REGION Network 2: PREMIXING VESSEL BOTTOM STERROR RUN
   RUNG wire#powerrail
      I_Contact( "AlwaysTRUE" )
      { S7_Templates := "SrcType := Int" } EQ_Contact(in1 := "MODE SELECTION DB"."MODE BUFF", in2 := 2)
      I_Contact( "RECIRCULATION DB".PREMIXING.PAUSE )
      Coil( "TRANSFER DB".OUTPUT."PREMIXING VESSEL BOTTOM STERROR RUN" )
   END_RUNG
   // the same network as SCL:
   "TRANSFER DB".OUTPUT."PREMIXING VESSEL BOTTOM STERROR RUN" := NOT "AlwaysTRUE" AND ("MODE SELECTION DB"."MODE BUFF" = 2) AND NOT "RECIRCULATION DB".PREMIXING.PAUSE;
END_REGION

REGION Network 3: INLINE 1 HOMOGENIZER MOTOR1 RUN
   RUNG wire#powerrail
      Contact( "AlwaysTRUE" )
      wire#w1
      { S7_Templates := "SrcType := Int" } NE_Contact(in1 := "MODE SELECTION DB"."MODE BUFF", in2 := 0)
      wire#w2
      Contact( "TRANSFER DB".BIT."MFG TO STORAGE-1 WITH INLINE HOMO"."INLINE 1 HOMOGENIZER MOTOR1 RUN" )
      wire#w3
      Contact( "DO MAPING"."PAV-56 INLINE HOMO. SEAL COOLING INLET" )
      { S7_Templates := "time_type := Time" } "IEC_Timer_0_DB_80".TON(pt := T#3S, et =>)
      Coil( "TRANSFER DB".OUTPUT."INLINE 1 HOMOGENIZER MOTOR1 RUN" )
   END_RUNG
   RUNG wire#w2
      Contact( "TRANSFER DB".BIT."MFG TO STORAGE-2 WITH INLINE HOMO"."INLINE 1 HOMOGENIZER MOTOR1 RUN" )
   END_RUNG wire#w3
   RUNG wire#w2
      Contact( "TRANSFER DB".BIT."MFG TO STORAGE-3 WITH INLINE HOMO"."INLINE 1 HOMOGENIZER MOTOR1 RUN" )
   END_RUNG wire#w3
   RUNG wire#w1
      { S7_Templates := "SrcType := Int" } EQ_Contact(in1 := "MODE SELECTION DB"."MODE BUFF", in2 := 2)
      { S7_Templates := "SrcType := Int" } EQ_Contact(in1 := "RECIRCULATION DB".MFG.BUFF, in2 := 2)
      I_Contact( "RECIRCULATION DB".MFG.PAUSE )
   END_RUNG wire#w3
   // the same network as SCL:
   "IEC_Timer_0_DB_80".TON(IN := "AlwaysTRUE" AND ((("MODE SELECTION DB"."MODE BUFF" <> 0) AND ("TRANSFER DB".BIT."MFG TO STORAGE-1 WITH INLINE HOMO"."INLINE 1 HOMOGENIZER MOTOR1 RUN" OR "TRANSFER DB".BIT."MFG TO STORAGE-2 WITH INLINE HOMO"."INLINE 1 HOMOGENIZER MOTOR1 RUN" OR "TRANSFER DB".BIT."MFG TO STORAGE-3 WITH INLINE HOMO"."INLINE 1 HOMOGENIZER MOTOR1 RUN")) OR (("MODE SELECTION DB"."MODE BUFF" = 2) AND ("RECIRCULATION DB".MFG.BUFF = 2) AND NOT "RECIRCULATION DB".MFG.PAUSE)) AND "DO MAPING"."PAV-56 INLINE HOMO. SEAL COOLING INLET",
                           PT := T#3S);
   "TRANSFER DB".OUTPUT."INLINE 1 HOMOGENIZER MOTOR1 RUN" := "IEC_Timer_0_DB_80".Q;
END_REGION

REGION Network 4: INLINE 2 HOMOGENIZER MOTOR 2 RUN
   RUNG wire#powerrail
      Contact( "AlwaysTRUE" )
      wire#w1
      { S7_Templates := "SrcType := Int" } NE_Contact(in1 := "MODE SELECTION DB"."MODE BUFF", in2 := 0)
      wire#w2
      Contact( "TRANSFER DB".BIT."PREMIXING TO MFG WITH INLINE HOMO"."INLINE 2 HOMOGENIZER MOTOR 2 RUN" )
      wire#w3
      Contact( "DO MAPING"."PAV-99 INLINE HOMOGENIZER SEAL COOLING" )
      { S7_Templates := "time_type := Time" } "IEC_Timer_0_DB_65".TON(pt := T#3S, et =>)
      Coil( "TRANSFER DB".OUTPUT."INLINE 2 HOMOGENIZER MOTOR 2 RUN" )
   END_RUNG
   RUNG wire#w2
      Contact( "TRANSFER DB".BIT."PREMIXING TO STORAGE-4 WITH INLINE HOMO"."INLINE 2 HOMOGENIZER MOTOR 2 RUN" )
   END_RUNG wire#w3
   RUNG wire#w1
      { S7_Templates := "SrcType := Int" } EQ_Contact(in1 := "MODE SELECTION DB"."MODE BUFF", in2 := 2)
      { S7_Templates := "SrcType := Int" } EQ_Contact(in1 := "RECIRCULATION DB".PREMIXING.BUFF, in2 := 2)
      I_Contact( "RECIRCULATION DB".PREMIXING.PAUSE )
   END_RUNG wire#w3
   // the same network as SCL:
   "IEC_Timer_0_DB_65".TON(IN := "AlwaysTRUE" AND ((("MODE SELECTION DB"."MODE BUFF" <> 0) AND ("TRANSFER DB".BIT."PREMIXING TO MFG WITH INLINE HOMO"."INLINE 2 HOMOGENIZER MOTOR 2 RUN" OR "TRANSFER DB".BIT."PREMIXING TO STORAGE-4 WITH INLINE HOMO"."INLINE 2 HOMOGENIZER MOTOR 2 RUN")) OR (("MODE SELECTION DB"."MODE BUFF" = 2) AND ("RECIRCULATION DB".PREMIXING.BUFF = 2) AND NOT "RECIRCULATION DB".PREMIXING.PAUSE)) AND "DO MAPING"."PAV-99 INLINE HOMOGENIZER SEAL COOLING",
                           PT := T#3S);
   "TRANSFER DB".OUTPUT."INLINE 2 HOMOGENIZER MOTOR 2 RUN" := "IEC_Timer_0_DB_65".Q;
END_REGION

REGION Network 5: FILTER PRESS MOTOR 1 RUN
   RUNG wire#powerrail
      Contact( "AlwaysTRUE" )
      { S7_Templates := "SrcType := Int" } NE_Contact(in1 := "MODE SELECTION DB"."MODE BUFF", in2 := 0)
      wire#w1
      Contact( "TRANSFER DB".BIT."MFG TO STORAGE-1 WITH INLINE FILTER PRES"."FILTER PRESS MOTOR 1 RUN" )
      wire#w2
      Coil( "TRANSFER DB".OUTPUT."FILTER PRESS MOTOR 1 RUN" )
   END_RUNG
   RUNG wire#w1
      Contact( "TRANSFER DB".BIT."MFG TO STORAGE-2 WITH INLINE FILTER PRES"."FILTER PRESS MOTOR 1 RUN" )
   END_RUNG wire#w2
   RUNG wire#w1
      Contact( "TRANSFER DB".BIT."MFG TO STORAGE-3 WITH INLINE FILTER PRES"."FILTER PRESS MOTOR 1 RUN" )
   END_RUNG wire#w2
   // the same network as SCL:
   "TRANSFER DB".OUTPUT."FILTER PRESS MOTOR 1 RUN" := "AlwaysTRUE" AND ("MODE SELECTION DB"."MODE BUFF" <> 0) AND ("TRANSFER DB".BIT."MFG TO STORAGE-1 WITH INLINE FILTER PRES"."FILTER PRESS MOTOR 1 RUN" OR "TRANSFER DB".BIT."MFG TO STORAGE-2 WITH INLINE FILTER PRES"."FILTER PRESS MOTOR 1 RUN" OR "TRANSFER DB".BIT."MFG TO STORAGE-3 WITH INLINE FILTER PRES"."FILTER PRESS MOTOR 1 RUN");
END_REGION

REGION Network 6: FILTER PRESS MOTOR 2 RUN
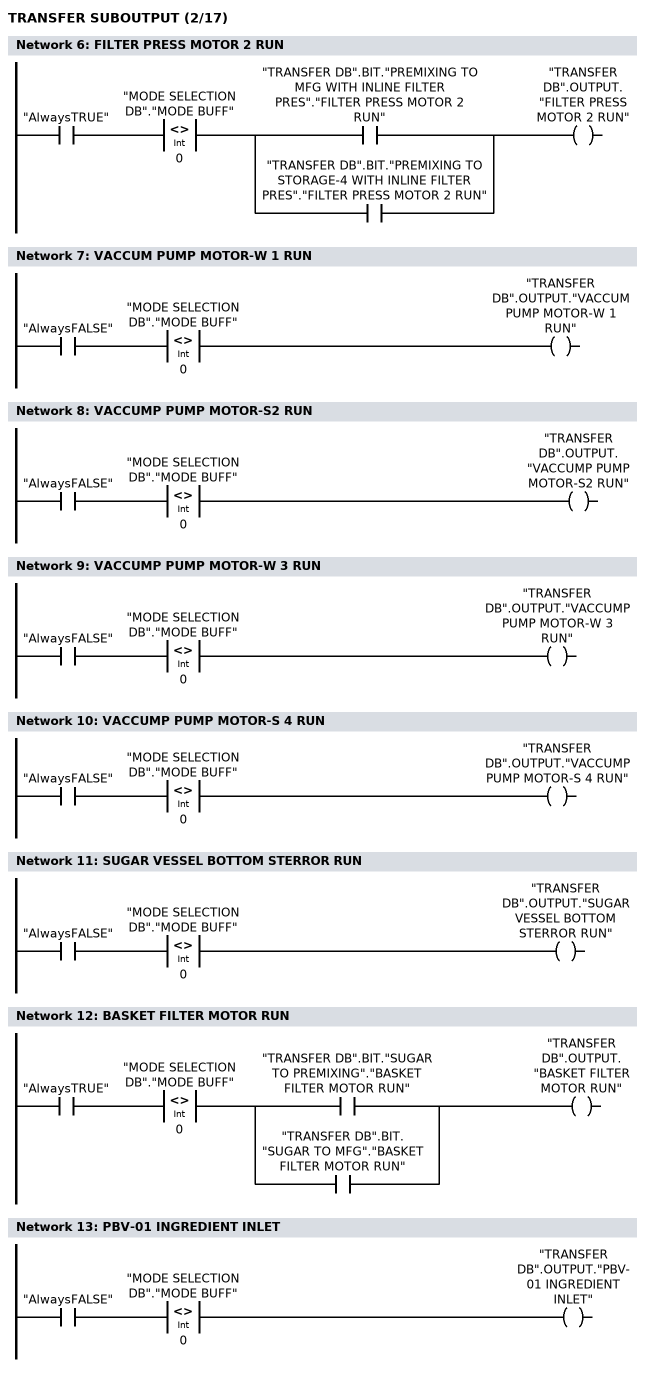
   RUNG wire#powerrail
      Contact( "AlwaysTRUE" )
      { S7_Templates := "SrcType := Int" } NE_Contact(in1 := "MODE SELECTION DB"."MODE BUFF", in2 := 0)
      wire#w1
      Contact( "TRANSFER DB".BIT."PREMIXING TO MFG WITH INLINE FILTER PRES"."FILTER PRESS MOTOR 2 RUN" )
      wire#w2
      Coil( "TRANSFER DB".OUTPUT."FILTER PRESS MOTOR 2 RUN" )
   END_RUNG
   RUNG wire#w1
      Contact( "TRANSFER DB".BIT."PREMIXING TO STORAGE-4 WITH INLINE FILTER PRES"."FILTER PRESS MOTOR 2 RUN" )
   END_RUNG wire#w2
   // the same network as SCL:
   "TRANSFER DB".OUTPUT."FILTER PRESS MOTOR 2 RUN" := "AlwaysTRUE" AND ("MODE SELECTION DB"."MODE BUFF" <> 0) AND ("TRANSFER DB".BIT."PREMIXING TO MFG WITH INLINE FILTER PRES"."FILTER PRESS MOTOR 2 RUN" OR "TRANSFER DB".BIT."PREMIXING TO STORAGE-4 WITH INLINE FILTER PRES"."FILTER PRESS MOTOR 2 RUN");
END_REGION

REGION Network 7: VACCUM PUMP MOTOR-W 1 RUN
   RUNG wire#powerrail
      Contact( "AlwaysFALSE" )
      { S7_Templates := "SrcType := Int" } NE_Contact(in1 := "MODE SELECTION DB"."MODE BUFF", in2 := 0)
      Coil( "TRANSFER DB".OUTPUT."VACCUM PUMP MOTOR-W 1 RUN" )
   END_RUNG
   // the same network as SCL:
   "TRANSFER DB".OUTPUT."VACCUM PUMP MOTOR-W 1 RUN" := "AlwaysFALSE" AND ("MODE SELECTION DB"."MODE BUFF" <> 0);
END_REGION

REGION Network 8: VACCUMP PUMP MOTOR-S2 RUN
   RUNG wire#powerrail
      Contact( "AlwaysFALSE" )
      { S7_Templates := "SrcType := Int" } NE_Contact(in1 := "MODE SELECTION DB"."MODE BUFF", in2 := 0)
      Coil( "TRANSFER DB".OUTPUT."VACCUMP PUMP MOTOR-S2 RUN" )
   END_RUNG
   // the same network as SCL:
   "TRANSFER DB".OUTPUT."VACCUMP PUMP MOTOR-S2 RUN" := "AlwaysFALSE" AND ("MODE SELECTION DB"."MODE BUFF" <> 0);
END_REGION

REGION Network 9: VACCUMP PUMP MOTOR-W 3 RUN
   RUNG wire#powerrail
      Contact( "AlwaysFALSE" )
      { S7_Templates := "SrcType := Int" } NE_Contact(in1 := "MODE SELECTION DB"."MODE BUFF", in2 := 0)
      Coil( "TRANSFER DB".OUTPUT."VACCUMP PUMP MOTOR-W 3 RUN" )
   END_RUNG
   // the same network as SCL:
   "TRANSFER DB".OUTPUT."VACCUMP PUMP MOTOR-W 3 RUN" := "AlwaysFALSE" AND ("MODE SELECTION DB"."MODE BUFF" <> 0);
END_REGION

REGION Network 10: VACCUMP PUMP MOTOR-S 4 RUN
   RUNG wire#powerrail
      Contact( "AlwaysFALSE" )
      { S7_Templates := "SrcType := Int" } NE_Contact(in1 := "MODE SELECTION DB"."MODE BUFF", in2 := 0)
      Coil( "TRANSFER DB".OUTPUT."VACCUMP PUMP MOTOR-S 4 RUN" )
   END_RUNG
   // the same network as SCL:
   "TRANSFER DB".OUTPUT."VACCUMP PUMP MOTOR-S 4 RUN" := "AlwaysFALSE" AND ("MODE SELECTION DB"."MODE BUFF" <> 0);
END_REGION

REGION Network 11: SUGAR VESSEL BOTTOM STERROR RUN
   RUNG wire#powerrail
      Contact( "AlwaysFALSE" )
      { S7_Templates := "SrcType := Int" } NE_Contact(in1 := "MODE SELECTION DB"."MODE BUFF", in2 := 0)
      Coil( "TRANSFER DB".OUTPUT."SUGAR VESSEL BOTTOM STERROR RUN" )
   END_RUNG
   // the same network as SCL:
   "TRANSFER DB".OUTPUT."SUGAR VESSEL BOTTOM STERROR RUN" := "AlwaysFALSE" AND ("MODE SELECTION DB"."MODE BUFF" <> 0);
END_REGION

REGION Network 12: BASKET FILTER MOTOR RUN
   RUNG wire#powerrail
      Contact( "AlwaysTRUE" )
      { S7_Templates := "SrcType := Int" } NE_Contact(in1 := "MODE SELECTION DB"."MODE BUFF", in2 := 0)
      wire#w1
      Contact( "TRANSFER DB".BIT."SUGAR TO PREMIXING"."BASKET FILTER MOTOR RUN" )
      wire#w2
      Coil( "TRANSFER DB".OUTPUT."BASKET FILTER MOTOR RUN" )
   END_RUNG
   RUNG wire#w1
      Contact( "TRANSFER DB".BIT."SUGAR TO MFG"."BASKET FILTER MOTOR RUN" )
   END_RUNG wire#w2
   // the same network as SCL:
   "TRANSFER DB".OUTPUT."BASKET FILTER MOTOR RUN" := "AlwaysTRUE" AND ("MODE SELECTION DB"."MODE BUFF" <> 0) AND ("TRANSFER DB".BIT."SUGAR TO PREMIXING"."BASKET FILTER MOTOR RUN" OR "TRANSFER DB".BIT."SUGAR TO MFG"."BASKET FILTER MOTOR RUN");
END_REGION

REGION Network 13: PBV-01 INGREDIENT INLET
   RUNG wire#powerrail
      Contact( "AlwaysFALSE" )
      { S7_Templates := "SrcType := Int" } NE_Contact(in1 := "MODE SELECTION DB"."MODE BUFF", in2 := 0)
      Coil( "TRANSFER DB".OUTPUT."PBV-01 INGREDIENT INLET" )
   END_RUNG
   // the same network as SCL:
   "TRANSFER DB".OUTPUT."PBV-01 INGREDIENT INLET" := "AlwaysFALSE" AND ("MODE SELECTION DB"."MODE BUFF" <> 0);
END_REGION

REGION Network 14: PBV-02 CIP INLET (SPRAY BALL)
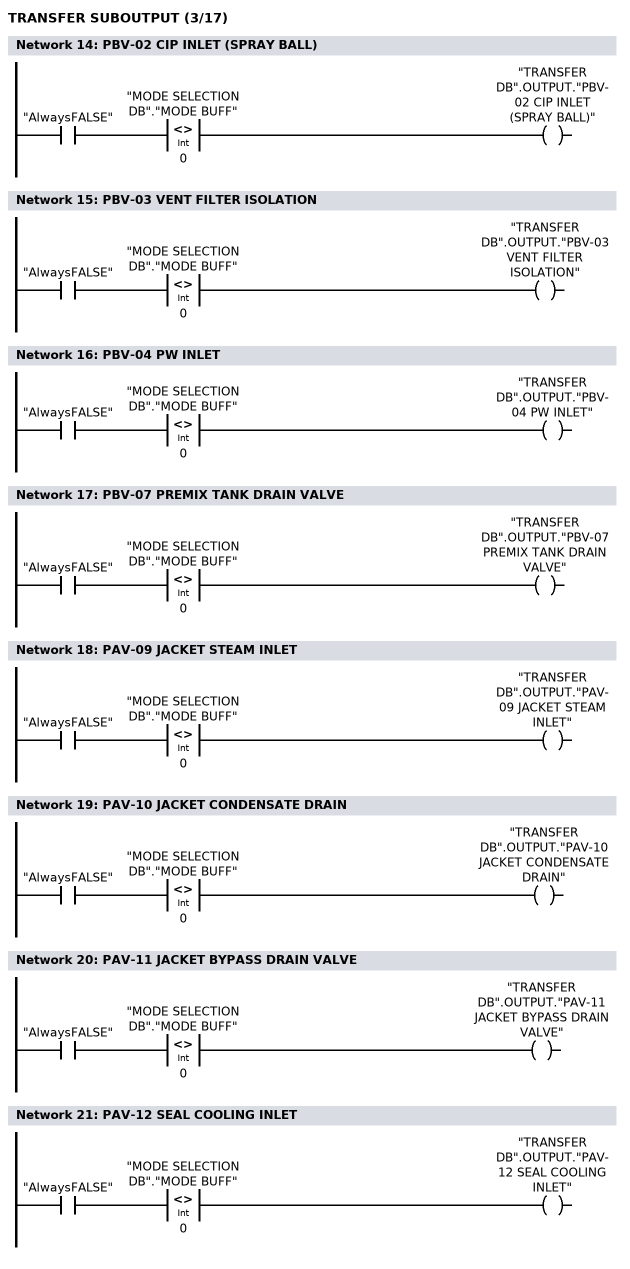
   RUNG wire#powerrail
      Contact( "AlwaysFALSE" )
      { S7_Templates := "SrcType := Int" } NE_Contact(in1 := "MODE SELECTION DB"."MODE BUFF", in2 := 0)
      Coil( "TRANSFER DB".OUTPUT."PBV-02 CIP INLET (SPRAY BALL)" )
   END_RUNG
   // the same network as SCL:
   "TRANSFER DB".OUTPUT."PBV-02 CIP INLET (SPRAY BALL)" := "AlwaysFALSE" AND ("MODE SELECTION DB"."MODE BUFF" <> 0);
END_REGION

REGION Network 15: PBV-03 VENT FILTER ISOLATION
   RUNG wire#powerrail
      Contact( "AlwaysFALSE" )
      { S7_Templates := "SrcType := Int" } NE_Contact(in1 := "MODE SELECTION DB"."MODE BUFF", in2 := 0)
      Coil( "TRANSFER DB".OUTPUT."PBV-03 VENT FILTER ISOLATION" )
   END_RUNG
   // the same network as SCL:
   "TRANSFER DB".OUTPUT."PBV-03 VENT FILTER ISOLATION" := "AlwaysFALSE" AND ("MODE SELECTION DB"."MODE BUFF" <> 0);
END_REGION

REGION Network 16: PBV-04 PW INLET
   RUNG wire#powerrail
      Contact( "AlwaysFALSE" )
      { S7_Templates := "SrcType := Int" } NE_Contact(in1 := "MODE SELECTION DB"."MODE BUFF", in2 := 0)
      Coil( "TRANSFER DB".OUTPUT."PBV-04 PW INLET" )
   END_RUNG
   // the same network as SCL:
   "TRANSFER DB".OUTPUT."PBV-04 PW INLET" := "AlwaysFALSE" AND ("MODE SELECTION DB"."MODE BUFF" <> 0);
END_REGION

REGION Network 17: PBV-07 PREMIX TANK DRAIN VALVE
   RUNG wire#powerrail
      Contact( "AlwaysFALSE" )
      { S7_Templates := "SrcType := Int" } NE_Contact(in1 := "MODE SELECTION DB"."MODE BUFF", in2 := 0)
      Coil( "TRANSFER DB".OUTPUT."PBV-07 PREMIX TANK DRAIN VALVE" )
   END_RUNG
   // the same network as SCL:
   "TRANSFER DB".OUTPUT."PBV-07 PREMIX TANK DRAIN VALVE" := "AlwaysFALSE" AND ("MODE SELECTION DB"."MODE BUFF" <> 0);
END_REGION

REGION Network 18: PAV-09 JACKET STEAM INLET
   RUNG wire#powerrail
      Contact( "AlwaysFALSE" )
      { S7_Templates := "SrcType := Int" } NE_Contact(in1 := "MODE SELECTION DB"."MODE BUFF", in2 := 0)
      Coil( "TRANSFER DB".OUTPUT."PAV-09 JACKET STEAM INLET" )
   END_RUNG
   // the same network as SCL:
   "TRANSFER DB".OUTPUT."PAV-09 JACKET STEAM INLET" := "AlwaysFALSE" AND ("MODE SELECTION DB"."MODE BUFF" <> 0);
END_REGION

REGION Network 19: PAV-10 JACKET CONDENSATE DRAIN
   RUNG wire#powerrail
      Contact( "AlwaysFALSE" )
      { S7_Templates := "SrcType := Int" } NE_Contact(in1 := "MODE SELECTION DB"."MODE BUFF", in2 := 0)
      Coil( "TRANSFER DB".OUTPUT."PAV-10 JACKET CONDENSATE DRAIN" )
   END_RUNG
   // the same network as SCL:
   "TRANSFER DB".OUTPUT."PAV-10 JACKET CONDENSATE DRAIN" := "AlwaysFALSE" AND ("MODE SELECTION DB"."MODE BUFF" <> 0);
END_REGION

REGION Network 20: PAV-11 JACKET BYPASS DRAIN VALVE
   RUNG wire#powerrail
      Contact( "AlwaysFALSE" )
      { S7_Templates := "SrcType := Int" } NE_Contact(in1 := "MODE SELECTION DB"."MODE BUFF", in2 := 0)
      Coil( "TRANSFER DB".OUTPUT."PAV-11 JACKET BYPASS DRAIN VALVE" )
   END_RUNG
   // the same network as SCL:
   "TRANSFER DB".OUTPUT."PAV-11 JACKET BYPASS DRAIN VALVE" := "AlwaysFALSE" AND ("MODE SELECTION DB"."MODE BUFF" <> 0);
END_REGION

REGION Network 21: PAV-12 SEAL COOLING INLET
   RUNG wire#powerrail
      Contact( "AlwaysFALSE" )
      { S7_Templates := "SrcType := Int" } NE_Contact(in1 := "MODE SELECTION DB"."MODE BUFF", in2 := 0)
      Coil( "TRANSFER DB".OUTPUT."PAV-12 SEAL COOLING INLET" )
   END_RUNG
   // the same network as SCL:
   "TRANSFER DB".OUTPUT."PAV-12 SEAL COOLING INLET" := "AlwaysFALSE" AND ("MODE SELECTION DB"."MODE BUFF" <> 0);
END_REGION

REGION Network 22: PAV-13 WATER COOLING INLET
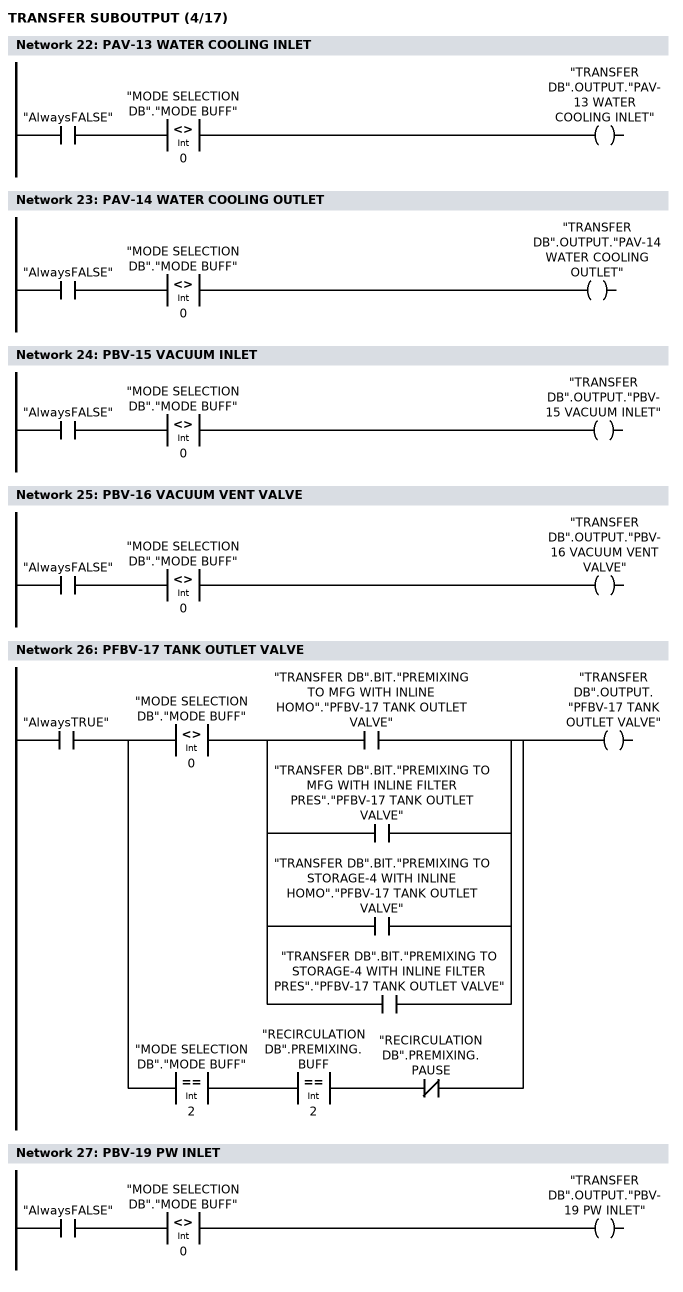
   RUNG wire#powerrail
      Contact( "AlwaysFALSE" )
      { S7_Templates := "SrcType := Int" } NE_Contact(in1 := "MODE SELECTION DB"."MODE BUFF", in2 := 0)
      Coil( "TRANSFER DB".OUTPUT."PAV-13 WATER COOLING INLET" )
   END_RUNG
   // the same network as SCL:
   "TRANSFER DB".OUTPUT."PAV-13 WATER COOLING INLET" := "AlwaysFALSE" AND ("MODE SELECTION DB"."MODE BUFF" <> 0);
END_REGION

REGION Network 23: PAV-14 WATER COOLING OUTLET
   RUNG wire#powerrail
      Contact( "AlwaysFALSE" )
      { S7_Templates := "SrcType := Int" } NE_Contact(in1 := "MODE SELECTION DB"."MODE BUFF", in2 := 0)
      Coil( "TRANSFER DB".OUTPUT."PAV-14 WATER COOLING OUTLET" )
   END_RUNG
   // the same network as SCL:
   "TRANSFER DB".OUTPUT."PAV-14 WATER COOLING OUTLET" := "AlwaysFALSE" AND ("MODE SELECTION DB"."MODE BUFF" <> 0);
END_REGION

REGION Network 24: PBV-15 VACUUM INLET
   RUNG wire#powerrail
      Contact( "AlwaysFALSE" )
      { S7_Templates := "SrcType := Int" } NE_Contact(in1 := "MODE SELECTION DB"."MODE BUFF", in2 := 0)
      Coil( "TRANSFER DB".OUTPUT."PBV-15 VACUUM INLET" )
   END_RUNG
   // the same network as SCL:
   "TRANSFER DB".OUTPUT."PBV-15 VACUUM INLET" := "AlwaysFALSE" AND ("MODE SELECTION DB"."MODE BUFF" <> 0);
END_REGION

REGION Network 25: PBV-16 VACUUM VENT VALVE
   RUNG wire#powerrail
      Contact( "AlwaysFALSE" )
      { S7_Templates := "SrcType := Int" } NE_Contact(in1 := "MODE SELECTION DB"."MODE BUFF", in2 := 0)
      Coil( "TRANSFER DB".OUTPUT."PBV-16 VACUUM VENT VALVE" )
   END_RUNG
   // the same network as SCL:
   "TRANSFER DB".OUTPUT."PBV-16 VACUUM VENT VALVE" := "AlwaysFALSE" AND ("MODE SELECTION DB"."MODE BUFF" <> 0);
END_REGION

REGION Network 26: PFBV-17 TANK OUTLET VALVE
   RUNG wire#powerrail
      Contact( "AlwaysTRUE" )
      wire#w1
      { S7_Templates := "SrcType := Int" } NE_Contact(in1 := "MODE SELECTION DB"."MODE BUFF", in2 := 0)
      wire#w2
      Contact( "TRANSFER DB".BIT."PREMIXING TO MFG WITH INLINE HOMO"."PFBV-17 TANK OUTLET VALVE" )
      wire#w3
      Coil( "TRANSFER DB".OUTPUT."PFBV-17 TANK OUTLET VALVE" )
   END_RUNG
   RUNG wire#w2
      Contact( "TRANSFER DB".BIT."PREMIXING TO MFG WITH INLINE FILTER PRES"."PFBV-17 TANK OUTLET VALVE" )
   END_RUNG wire#w3
   RUNG wire#w2
      Contact( "TRANSFER DB".BIT."PREMIXING TO STORAGE-4 WITH INLINE HOMO"."PFBV-17 TANK OUTLET VALVE" )
   END_RUNG wire#w3
   RUNG wire#w2
      Contact( "TRANSFER DB".BIT."PREMIXING TO STORAGE-4 WITH INLINE FILTER PRES"."PFBV-17 TANK OUTLET VALVE" )
   END_RUNG wire#w3
   RUNG wire#w1
      { S7_Templates := "SrcType := Int" } EQ_Contact(in1 := "MODE SELECTION DB"."MODE BUFF", in2 := 2)
      { S7_Templates := "SrcType := Int" } EQ_Contact(in1 := "RECIRCULATION DB".PREMIXING.BUFF, in2 := 2)
      I_Contact( "RECIRCULATION DB".PREMIXING.PAUSE )
   END_RUNG wire#w3
   // the same network as SCL:
   "TRANSFER DB".OUTPUT."PFBV-17 TANK OUTLET VALVE" := "AlwaysTRUE" AND ((("MODE SELECTION DB"."MODE BUFF" <> 0) AND ("TRANSFER DB".BIT."PREMIXING TO MFG WITH INLINE HOMO"."PFBV-17 TANK OUTLET VALVE" OR "TRANSFER DB".BIT."PREMIXING TO MFG WITH INLINE FILTER PRES"."PFBV-17 TANK OUTLET VALVE" OR "TRANSFER DB".BIT."PREMIXING TO STORAGE-4 WITH INLINE HOMO"."PFBV-17 TANK OUTLET VALVE" OR "TRANSFER DB".BIT."PREMIXING TO STORAGE-4 WITH INLINE FILTER PRES"."PFBV-17 TANK OUTLET VALVE")) OR (("MODE SELECTION DB"."MODE BUFF" = 2) AND ("RECIRCULATION DB".PREMIXING.BUFF = 2) AND NOT "RECIRCULATION DB".PREMIXING.PAUSE));
END_REGION

REGION Network 27: PBV-19 PW INLET
   RUNG wire#powerrail
      Contact( "AlwaysFALSE" )
      { S7_Templates := "SrcType := Int" } NE_Contact(in1 := "MODE SELECTION DB"."MODE BUFF", in2 := 0)
      Coil( "TRANSFER DB".OUTPUT."PBV-19 PW INLET" )
   END_RUNG
   // the same network as SCL:
   "TRANSFER DB".OUTPUT."PBV-19 PW INLET" := "AlwaysFALSE" AND ("MODE SELECTION DB"."MODE BUFF" <> 0);
END_REGION

REGION Network 28: PBV-20 CIP INLET (SPRAY BALL)
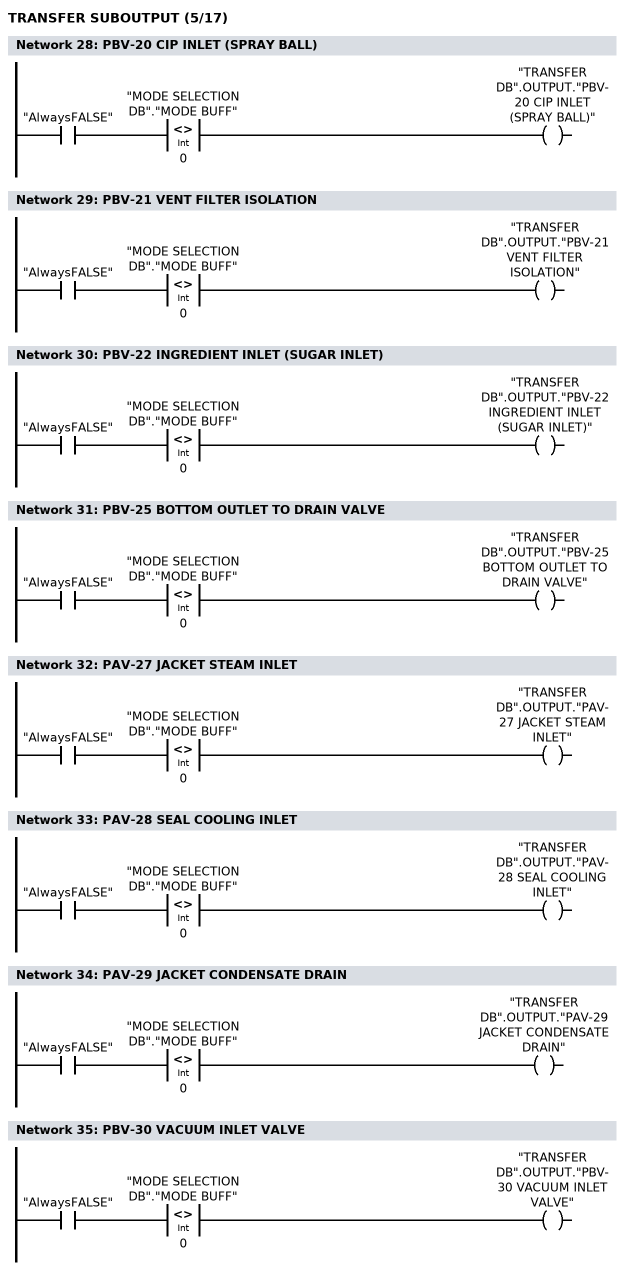
   RUNG wire#powerrail
      Contact( "AlwaysFALSE" )
      { S7_Templates := "SrcType := Int" } NE_Contact(in1 := "MODE SELECTION DB"."MODE BUFF", in2 := 0)
      Coil( "TRANSFER DB".OUTPUT."PBV-20 CIP INLET (SPRAY BALL)" )
   END_RUNG
   // the same network as SCL:
   "TRANSFER DB".OUTPUT."PBV-20 CIP INLET (SPRAY BALL)" := "AlwaysFALSE" AND ("MODE SELECTION DB"."MODE BUFF" <> 0);
END_REGION

REGION Network 29: PBV-21 VENT FILTER ISOLATION
   RUNG wire#powerrail
      Contact( "AlwaysFALSE" )
      { S7_Templates := "SrcType := Int" } NE_Contact(in1 := "MODE SELECTION DB"."MODE BUFF", in2 := 0)
      Coil( "TRANSFER DB".OUTPUT."PBV-21 VENT FILTER ISOLATION" )
   END_RUNG
   // the same network as SCL:
   "TRANSFER DB".OUTPUT."PBV-21 VENT FILTER ISOLATION" := "AlwaysFALSE" AND ("MODE SELECTION DB"."MODE BUFF" <> 0);
END_REGION

REGION Network 30: PBV-22 INGREDIENT INLET (SUGAR INLET)
   RUNG wire#powerrail
      Contact( "AlwaysFALSE" )
      { S7_Templates := "SrcType := Int" } NE_Contact(in1 := "MODE SELECTION DB"."MODE BUFF", in2 := 0)
      Coil( "TRANSFER DB".OUTPUT."PBV-22 INGREDIENT INLET (SUGAR INLET)" )
   END_RUNG
   // the same network as SCL:
   "TRANSFER DB".OUTPUT."PBV-22 INGREDIENT INLET (SUGAR INLET)" := "AlwaysFALSE" AND ("MODE SELECTION DB"."MODE BUFF" <> 0);
END_REGION

REGION Network 31: PBV-25 BOTTOM OUTLET TO DRAIN VALVE
   RUNG wire#powerrail
      Contact( "AlwaysFALSE" )
      { S7_Templates := "SrcType := Int" } NE_Contact(in1 := "MODE SELECTION DB"."MODE BUFF", in2 := 0)
      Coil( "TRANSFER DB".OUTPUT."PBV-25 BOTTOM OUTLET TO DRAIN VALVE" )
   END_RUNG
   // the same network as SCL:
   "TRANSFER DB".OUTPUT."PBV-25 BOTTOM OUTLET TO DRAIN VALVE" := "AlwaysFALSE" AND ("MODE SELECTION DB"."MODE BUFF" <> 0);
END_REGION

REGION Network 32: PAV-27 JACKET STEAM INLET
   RUNG wire#powerrail
      Contact( "AlwaysFALSE" )
      { S7_Templates := "SrcType := Int" } NE_Contact(in1 := "MODE SELECTION DB"."MODE BUFF", in2 := 0)
      Coil( "TRANSFER DB".OUTPUT."PAV-27 JACKET STEAM INLET" )
   END_RUNG
   // the same network as SCL:
   "TRANSFER DB".OUTPUT."PAV-27 JACKET STEAM INLET" := "AlwaysFALSE" AND ("MODE SELECTION DB"."MODE BUFF" <> 0);
END_REGION

REGION Network 33: PAV-28 SEAL COOLING INLET
   RUNG wire#powerrail
      Contact( "AlwaysFALSE" )
      { S7_Templates := "SrcType := Int" } NE_Contact(in1 := "MODE SELECTION DB"."MODE BUFF", in2 := 0)
      Coil( "TRANSFER DB".OUTPUT."PAV-28 SEAL COOLING INLET" )
   END_RUNG
   // the same network as SCL:
   "TRANSFER DB".OUTPUT."PAV-28 SEAL COOLING INLET" := "AlwaysFALSE" AND ("MODE SELECTION DB"."MODE BUFF" <> 0);
END_REGION

REGION Network 34: PAV-29 JACKET CONDENSATE DRAIN
   RUNG wire#powerrail
      Contact( "AlwaysFALSE" )
      { S7_Templates := "SrcType := Int" } NE_Contact(in1 := "MODE SELECTION DB"."MODE BUFF", in2 := 0)
      Coil( "TRANSFER DB".OUTPUT."PAV-29 JACKET CONDENSATE DRAIN" )
   END_RUNG
   // the same network as SCL:
   "TRANSFER DB".OUTPUT."PAV-29 JACKET CONDENSATE DRAIN" := "AlwaysFALSE" AND ("MODE SELECTION DB"."MODE BUFF" <> 0);
END_REGION

REGION Network 35: PBV-30 VACUUM INLET VALVE
   RUNG wire#powerrail
      Contact( "AlwaysFALSE" )
      { S7_Templates := "SrcType := Int" } NE_Contact(in1 := "MODE SELECTION DB"."MODE BUFF", in2 := 0)
      Coil( "TRANSFER DB".OUTPUT."PBV-30 VACUUM INLET VALVE" )
   END_RUNG
   // the same network as SCL:
   "TRANSFER DB".OUTPUT."PBV-30 VACUUM INLET VALVE" := "AlwaysFALSE" AND ("MODE SELECTION DB"."MODE BUFF" <> 0);
END_REGION

REGION Network 36: PBV-31 VACUUM VENT VALVE
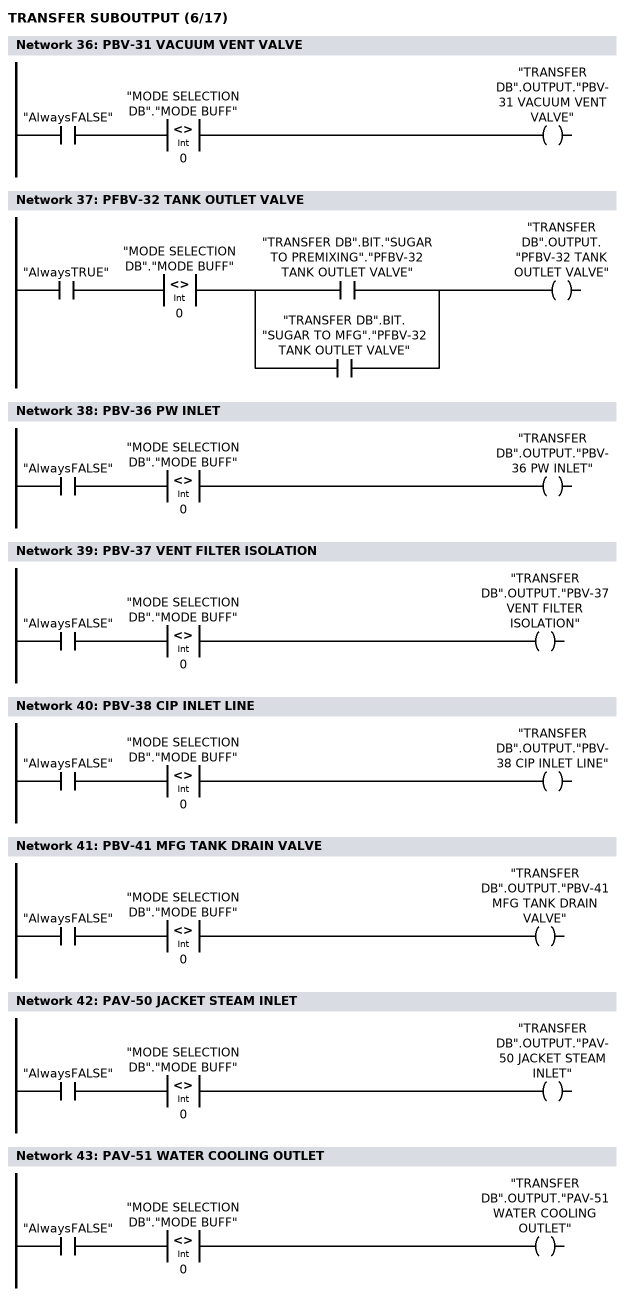
   RUNG wire#powerrail
      Contact( "AlwaysFALSE" )
      { S7_Templates := "SrcType := Int" } NE_Contact(in1 := "MODE SELECTION DB"."MODE BUFF", in2 := 0)
      Coil( "TRANSFER DB".OUTPUT."PBV-31 VACUUM VENT VALVE" )
   END_RUNG
   // the same network as SCL:
   "TRANSFER DB".OUTPUT."PBV-31 VACUUM VENT VALVE" := "AlwaysFALSE" AND ("MODE SELECTION DB"."MODE BUFF" <> 0);
END_REGION

REGION Network 37: PFBV-32 TANK OUTLET VALVE
   RUNG wire#powerrail
      Contact( "AlwaysTRUE" )
      { S7_Templates := "SrcType := Int" } NE_Contact(in1 := "MODE SELECTION DB"."MODE BUFF", in2 := 0)
      wire#w1
      Contact( "TRANSFER DB".BIT."SUGAR TO PREMIXING"."PFBV-32 TANK OUTLET VALVE" )
      wire#w2
      Coil( "TRANSFER DB".OUTPUT."PFBV-32 TANK OUTLET VALVE" )
   END_RUNG
   RUNG wire#w1
      Contact( "TRANSFER DB".BIT."SUGAR TO MFG"."PFBV-32 TANK OUTLET VALVE" )
   END_RUNG wire#w2
   // the same network as SCL:
   "TRANSFER DB".OUTPUT."PFBV-32 TANK OUTLET VALVE" := "AlwaysTRUE" AND ("MODE SELECTION DB"."MODE BUFF" <> 0) AND ("TRANSFER DB".BIT."SUGAR TO PREMIXING"."PFBV-32 TANK OUTLET VALVE" OR "TRANSFER DB".BIT."SUGAR TO MFG"."PFBV-32 TANK OUTLET VALVE");
END_REGION

REGION Network 38: PBV-36 PW INLET
   RUNG wire#powerrail
      Contact( "AlwaysFALSE" )
      { S7_Templates := "SrcType := Int" } NE_Contact(in1 := "MODE SELECTION DB"."MODE BUFF", in2 := 0)
      Coil( "TRANSFER DB".OUTPUT."PBV-36 PW INLET" )
   END_RUNG
   // the same network as SCL:
   "TRANSFER DB".OUTPUT."PBV-36 PW INLET" := "AlwaysFALSE" AND ("MODE SELECTION DB"."MODE BUFF" <> 0);
END_REGION

REGION Network 39: PBV-37 VENT FILTER ISOLATION
   RUNG wire#powerrail
      Contact( "AlwaysFALSE" )
      { S7_Templates := "SrcType := Int" } NE_Contact(in1 := "MODE SELECTION DB"."MODE BUFF", in2 := 0)
      Coil( "TRANSFER DB".OUTPUT."PBV-37 VENT FILTER ISOLATION" )
   END_RUNG
   // the same network as SCL:
   "TRANSFER DB".OUTPUT."PBV-37 VENT FILTER ISOLATION" := "AlwaysFALSE" AND ("MODE SELECTION DB"."MODE BUFF" <> 0);
END_REGION

REGION Network 40: PBV-38 CIP INLET LINE
   RUNG wire#powerrail
      Contact( "AlwaysFALSE" )
      { S7_Templates := "SrcType := Int" } NE_Contact(in1 := "MODE SELECTION DB"."MODE BUFF", in2 := 0)
      Coil( "TRANSFER DB".OUTPUT."PBV-38 CIP INLET LINE" )
   END_RUNG
   // the same network as SCL:
   "TRANSFER DB".OUTPUT."PBV-38 CIP INLET LINE" := "AlwaysFALSE" AND ("MODE SELECTION DB"."MODE BUFF" <> 0);
END_REGION

REGION Network 41: PBV-41 MFG TANK DRAIN VALVE
   RUNG wire#powerrail
      Contact( "AlwaysFALSE" )
      { S7_Templates := "SrcType := Int" } NE_Contact(in1 := "MODE SELECTION DB"."MODE BUFF", in2 := 0)
      Coil( "TRANSFER DB".OUTPUT."PBV-41 MFG TANK DRAIN VALVE" )
   END_RUNG
   // the same network as SCL:
   "TRANSFER DB".OUTPUT."PBV-41 MFG TANK DRAIN VALVE" := "AlwaysFALSE" AND ("MODE SELECTION DB"."MODE BUFF" <> 0);
END_REGION

REGION Network 42: PAV-50 JACKET STEAM INLET
   RUNG wire#powerrail
      Contact( "AlwaysFALSE" )
      { S7_Templates := "SrcType := Int" } NE_Contact(in1 := "MODE SELECTION DB"."MODE BUFF", in2 := 0)
      Coil( "TRANSFER DB".OUTPUT."PAV-50 JACKET STEAM INLET" )
   END_RUNG
   // the same network as SCL:
   "TRANSFER DB".OUTPUT."PAV-50 JACKET STEAM INLET" := "AlwaysFALSE" AND ("MODE SELECTION DB"."MODE BUFF" <> 0);
END_REGION

REGION Network 43: PAV-51 WATER COOLING OUTLET
   RUNG wire#powerrail
      Contact( "AlwaysFALSE" )
      { S7_Templates := "SrcType := Int" } NE_Contact(in1 := "MODE SELECTION DB"."MODE BUFF", in2 := 0)
      Coil( "TRANSFER DB".OUTPUT."PAV-51 WATER COOLING OUTLET" )
   END_RUNG
   // the same network as SCL:
   "TRANSFER DB".OUTPUT."PAV-51 WATER COOLING OUTLET" := "AlwaysFALSE" AND ("MODE SELECTION DB"."MODE BUFF" <> 0);
END_REGION

REGION Network 44: PAV-52 WATER COOLING INLET
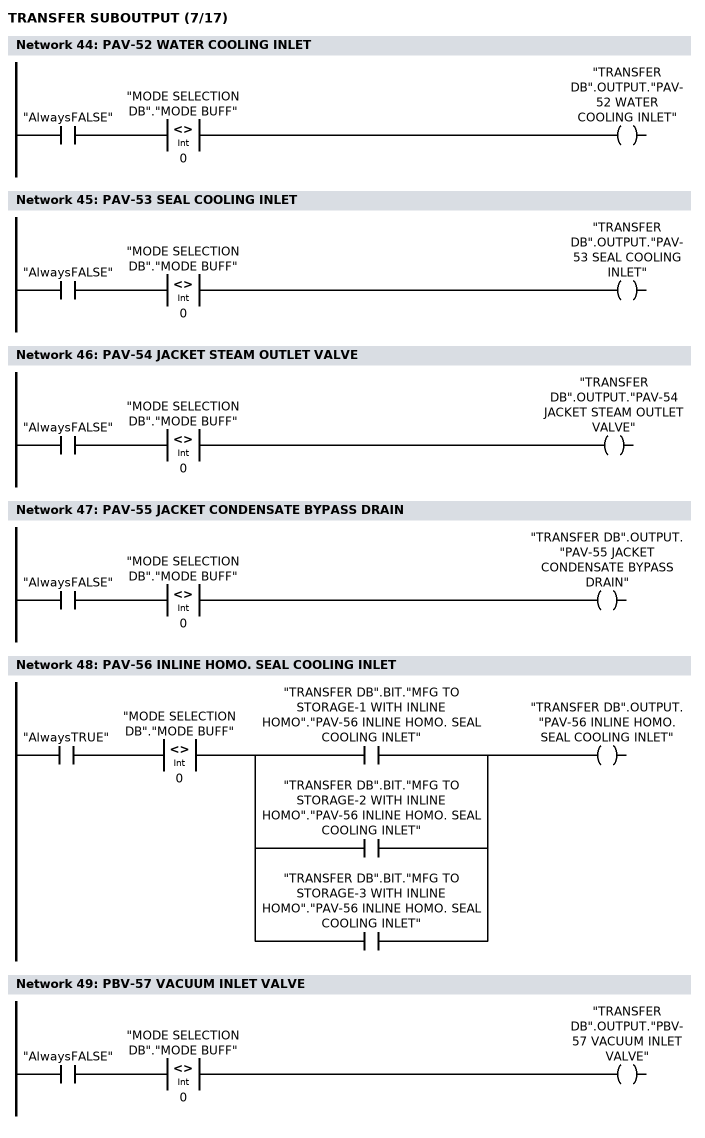
   RUNG wire#powerrail
      Contact( "AlwaysFALSE" )
      { S7_Templates := "SrcType := Int" } NE_Contact(in1 := "MODE SELECTION DB"."MODE BUFF", in2 := 0)
      Coil( "TRANSFER DB".OUTPUT."PAV-52 WATER COOLING INLET" )
   END_RUNG
   // the same network as SCL:
   "TRANSFER DB".OUTPUT."PAV-52 WATER COOLING INLET" := "AlwaysFALSE" AND ("MODE SELECTION DB"."MODE BUFF" <> 0);
END_REGION

REGION Network 45: PAV-53 SEAL COOLING INLET
   RUNG wire#powerrail
      Contact( "AlwaysFALSE" )
      { S7_Templates := "SrcType := Int" } NE_Contact(in1 := "MODE SELECTION DB"."MODE BUFF", in2 := 0)
      Coil( "TRANSFER DB".OUTPUT."PAV-53 SEAL COOLING INLET" )
   END_RUNG
   // the same network as SCL:
   "TRANSFER DB".OUTPUT."PAV-53 SEAL COOLING INLET" := "AlwaysFALSE" AND ("MODE SELECTION DB"."MODE BUFF" <> 0);
END_REGION

REGION Network 46: PAV-54 JACKET STEAM OUTLET VALVE
   RUNG wire#powerrail
      Contact( "AlwaysFALSE" )
      { S7_Templates := "SrcType := Int" } NE_Contact(in1 := "MODE SELECTION DB"."MODE BUFF", in2 := 0)
      Coil( "TRANSFER DB".OUTPUT."PAV-54 JACKET STEAM OUTLET VALVE" )
   END_RUNG
   // the same network as SCL:
   "TRANSFER DB".OUTPUT."PAV-54 JACKET STEAM OUTLET VALVE" := "AlwaysFALSE" AND ("MODE SELECTION DB"."MODE BUFF" <> 0);
END_REGION

REGION Network 47: PAV-55 JACKET CONDENSATE BYPASS DRAIN
   RUNG wire#powerrail
      Contact( "AlwaysFALSE" )
      { S7_Templates := "SrcType := Int" } NE_Contact(in1 := "MODE SELECTION DB"."MODE BUFF", in2 := 0)
      Coil( "TRANSFER DB".OUTPUT."PAV-55 JACKET CONDENSATE BYPASS DRAIN" )
   END_RUNG
   // the same network as SCL:
   "TRANSFER DB".OUTPUT."PAV-55 JACKET CONDENSATE BYPASS DRAIN" := "AlwaysFALSE" AND ("MODE SELECTION DB"."MODE BUFF" <> 0);
END_REGION

REGION Network 48: PAV-56 INLINE HOMO. SEAL COOLING INLET
   RUNG wire#powerrail
      Contact( "AlwaysTRUE" )
      { S7_Templates := "SrcType := Int" } NE_Contact(in1 := "MODE SELECTION DB"."MODE BUFF", in2 := 0)
      wire#w1
      Contact( "TRANSFER DB".BIT."MFG TO STORAGE-1 WITH INLINE HOMO"."PAV-56 INLINE HOMO. SEAL COOLING INLET" )
      wire#w2
      Coil( "TRANSFER DB".OUTPUT."PAV-56 INLINE HOMO. SEAL COOLING INLET" )
   END_RUNG
   RUNG wire#w1
      Contact( "TRANSFER DB".BIT."MFG TO STORAGE-2 WITH INLINE HOMO"."PAV-56 INLINE HOMO. SEAL COOLING INLET" )
   END_RUNG wire#w2
   RUNG wire#w1
      Contact( "TRANSFER DB".BIT."MFG TO STORAGE-3 WITH INLINE HOMO"."PAV-56 INLINE HOMO. SEAL COOLING INLET" )
   END_RUNG wire#w2
   // the same network as SCL:
   "TRANSFER DB".OUTPUT."PAV-56 INLINE HOMO. SEAL COOLING INLET" := "AlwaysTRUE" AND ("MODE SELECTION DB"."MODE BUFF" <> 0) AND ("TRANSFER DB".BIT."MFG TO STORAGE-1 WITH INLINE HOMO"."PAV-56 INLINE HOMO. SEAL COOLING INLET" OR "TRANSFER DB".BIT."MFG TO STORAGE-2 WITH INLINE HOMO"."PAV-56 INLINE HOMO. SEAL COOLING INLET" OR "TRANSFER DB".BIT."MFG TO STORAGE-3 WITH INLINE HOMO"."PAV-56 INLINE HOMO. SEAL COOLING INLET");
END_REGION

REGION Network 49: PBV-57 VACUUM INLET VALVE
   RUNG wire#powerrail
      Contact( "AlwaysFALSE" )
      { S7_Templates := "SrcType := Int" } NE_Contact(in1 := "MODE SELECTION DB"."MODE BUFF", in2 := 0)
      Coil( "TRANSFER DB".OUTPUT."PBV-57 VACUUM INLET VALVE" )
   END_RUNG
   // the same network as SCL:
   "TRANSFER DB".OUTPUT."PBV-57 VACUUM INLET VALVE" := "AlwaysFALSE" AND ("MODE SELECTION DB"."MODE BUFF" <> 0);
END_REGION

REGION Network 50: PFBV-59 TANK OUTLET VALVE
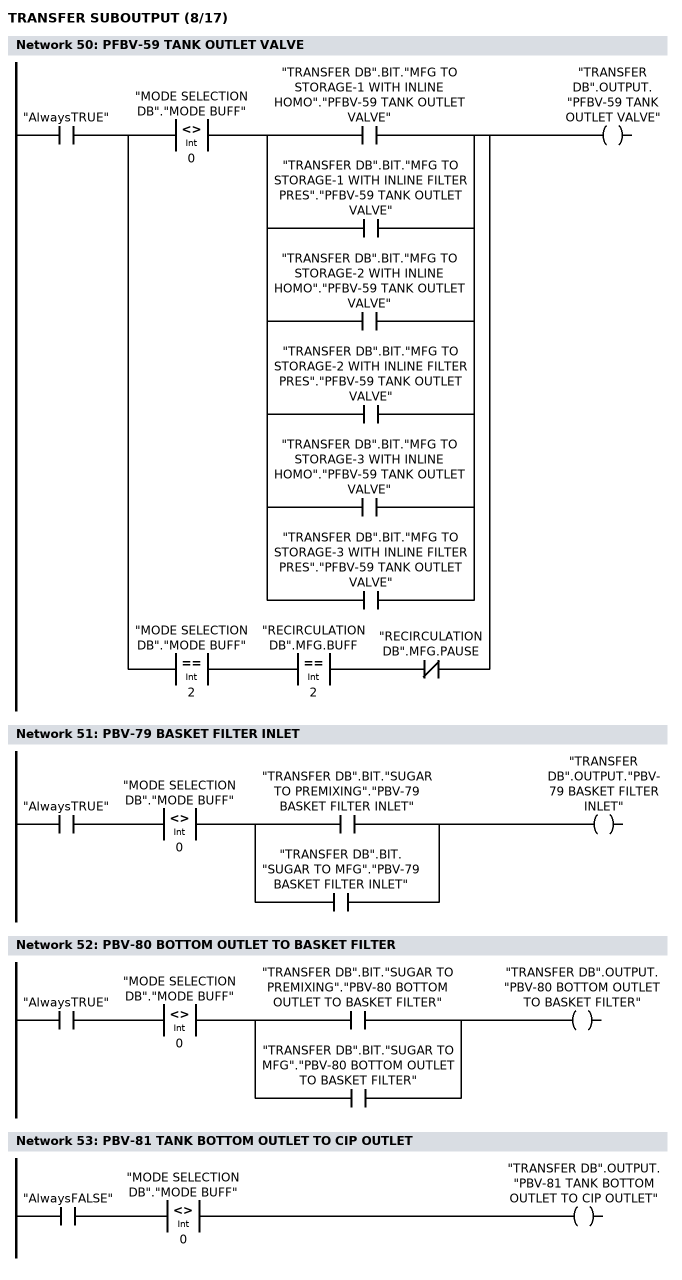
   RUNG wire#powerrail
      Contact( "AlwaysTRUE" )
      wire#w1
      { S7_Templates := "SrcType := Int" } NE_Contact(in1 := "MODE SELECTION DB"."MODE BUFF", in2 := 0)
      wire#w2
      Contact( "TRANSFER DB".BIT."MFG TO STORAGE-1 WITH INLINE HOMO"."PFBV-59 TANK OUTLET VALVE" )
      wire#w3
      Coil( "TRANSFER DB".OUTPUT."PFBV-59 TANK OUTLET VALVE" )
   END_RUNG
   RUNG wire#w2
      Contact( "TRANSFER DB".BIT."MFG TO STORAGE-1 WITH INLINE FILTER PRES"."PFBV-59 TANK OUTLET VALVE" )
   END_RUNG wire#w3
   RUNG wire#w2
      Contact( "TRANSFER DB".BIT."MFG TO STORAGE-2 WITH INLINE HOMO"."PFBV-59 TANK OUTLET VALVE" )
   END_RUNG wire#w3
   RUNG wire#w2
      Contact( "TRANSFER DB".BIT."MFG TO STORAGE-2 WITH INLINE FILTER PRES"."PFBV-59 TANK OUTLET VALVE" )
   END_RUNG wire#w3
   RUNG wire#w2
      Contact( "TRANSFER DB".BIT."MFG TO STORAGE-3 WITH INLINE HOMO"."PFBV-59 TANK OUTLET VALVE" )
   END_RUNG wire#w3
   RUNG wire#w2
      Contact( "TRANSFER DB".BIT."MFG TO STORAGE-3 WITH INLINE FILTER PRES"."PFBV-59 TANK OUTLET VALVE" )
   END_RUNG wire#w3
   RUNG wire#w1
      { S7_Templates := "SrcType := Int" } EQ_Contact(in1 := "MODE SELECTION DB"."MODE BUFF", in2 := 2)
      { S7_Templates := "SrcType := Int" } EQ_Contact(in1 := "RECIRCULATION DB".MFG.BUFF, in2 := 2)
      I_Contact( "RECIRCULATION DB".MFG.PAUSE )
   END_RUNG wire#w3
   // the same network as SCL:
   "TRANSFER DB".OUTPUT."PFBV-59 TANK OUTLET VALVE" := "AlwaysTRUE" AND ((("MODE SELECTION DB"."MODE BUFF" <> 0) AND ("TRANSFER DB".BIT."MFG TO STORAGE-1 WITH INLINE HOMO"."PFBV-59 TANK OUTLET VALVE" OR "TRANSFER DB".BIT."MFG TO STORAGE-1 WITH INLINE FILTER PRES"."PFBV-59 TANK OUTLET VALVE" OR "TRANSFER DB".BIT."MFG TO STORAGE-2 WITH INLINE HOMO"."PFBV-59 TANK OUTLET VALVE" OR "TRANSFER DB".BIT."MFG TO STORAGE-2 WITH INLINE FILTER PRES"."PFBV-59 TANK OUTLET VALVE" OR "TRANSFER DB".BIT."MFG TO STORAGE-3 WITH INLINE HOMO"."PFBV-59 TANK OUTLET VALVE" OR "TRANSFER DB".BIT."MFG TO STORAGE-3 WITH INLINE FILTER PRES"."PFBV-59 TANK OUTLET VALVE")) OR (("MODE SELECTION DB"."MODE BUFF" = 2) AND ("RECIRCULATION DB".MFG.BUFF = 2) AND NOT "RECIRCULATION DB".MFG.PAUSE));
END_REGION

REGION Network 51: PBV-79 BASKET FILTER INLET
   RUNG wire#powerrail
      Contact( "AlwaysTRUE" )
      { S7_Templates := "SrcType := Int" } NE_Contact(in1 := "MODE SELECTION DB"."MODE BUFF", in2 := 0)
      wire#w1
      Contact( "TRANSFER DB".BIT."SUGAR TO PREMIXING"."PBV-79 BASKET FILTER INLET" )
      wire#w2
      Coil( "TRANSFER DB".OUTPUT."PBV-79 BASKET FILTER INLET" )
   END_RUNG
   RUNG wire#w1
      Contact( "TRANSFER DB".BIT."SUGAR TO MFG"."PBV-79 BASKET FILTER INLET" )
   END_RUNG wire#w2
   // the same network as SCL:
   "TRANSFER DB".OUTPUT."PBV-79 BASKET FILTER INLET" := "AlwaysTRUE" AND ("MODE SELECTION DB"."MODE BUFF" <> 0) AND ("TRANSFER DB".BIT."SUGAR TO PREMIXING"."PBV-79 BASKET FILTER INLET" OR "TRANSFER DB".BIT."SUGAR TO MFG"."PBV-79 BASKET FILTER INLET");
END_REGION

REGION Network 52: PBV-80 BOTTOM OUTLET TO BASKET FILTER
   RUNG wire#powerrail
      Contact( "AlwaysTRUE" )
      { S7_Templates := "SrcType := Int" } NE_Contact(in1 := "MODE SELECTION DB"."MODE BUFF", in2 := 0)
      wire#w1
      Contact( "TRANSFER DB".BIT."SUGAR TO PREMIXING"."PBV-80 BOTTOM OUTLET TO BASKET FILTER" )
      wire#w2
      Coil( "TRANSFER DB".OUTPUT."PBV-80 BOTTOM OUTLET TO BASKET FILTER" )
   END_RUNG
   RUNG wire#w1
      Contact( "TRANSFER DB".BIT."SUGAR TO MFG"."PBV-80 BOTTOM OUTLET TO BASKET FILTER" )
   END_RUNG wire#w2
   // the same network as SCL:
   "TRANSFER DB".OUTPUT."PBV-80 BOTTOM OUTLET TO BASKET FILTER" := "AlwaysTRUE" AND ("MODE SELECTION DB"."MODE BUFF" <> 0) AND ("TRANSFER DB".BIT."SUGAR TO PREMIXING"."PBV-80 BOTTOM OUTLET TO BASKET FILTER" OR "TRANSFER DB".BIT."SUGAR TO MFG"."PBV-80 BOTTOM OUTLET TO BASKET FILTER");
END_REGION

REGION Network 53: PBV-81 TANK BOTTOM OUTLET TO CIP OUTLET
   RUNG wire#powerrail
      Contact( "AlwaysFALSE" )
      { S7_Templates := "SrcType := Int" } NE_Contact(in1 := "MODE SELECTION DB"."MODE BUFF", in2 := 0)
      Coil( "TRANSFER DB".OUTPUT."PBV-81 TANK BOTTOM OUTLET TO CIP OUTLET" )
   END_RUNG
   // the same network as SCL:
   "TRANSFER DB".OUTPUT."PBV-81 TANK BOTTOM OUTLET TO CIP OUTLET" := "AlwaysFALSE" AND ("MODE SELECTION DB"."MODE BUFF" <> 0);
END_REGION

REGION Network 54: PBV-82 CIP ISOLATION
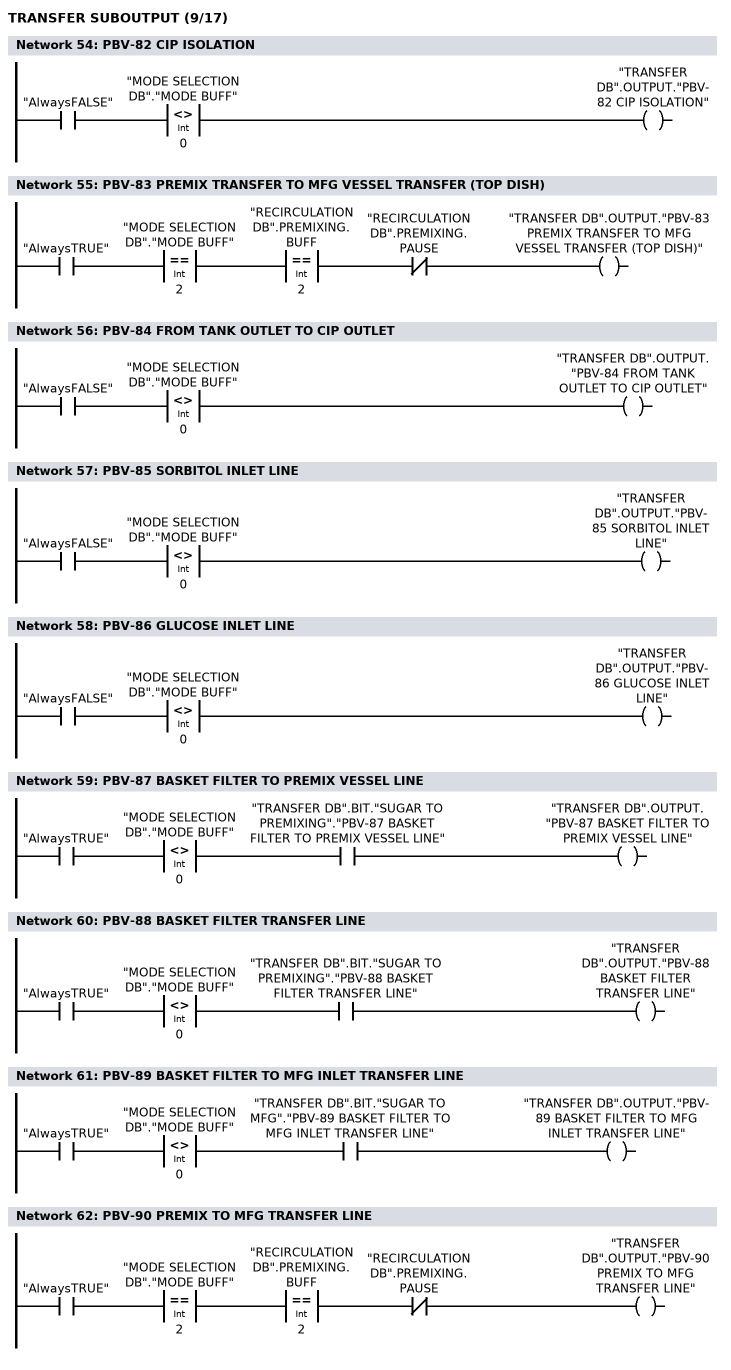
   RUNG wire#powerrail
      Contact( "AlwaysFALSE" )
      { S7_Templates := "SrcType := Int" } NE_Contact(in1 := "MODE SELECTION DB"."MODE BUFF", in2 := 0)
      Coil( "TRANSFER DB".OUTPUT."PBV-82 CIP ISOLATION" )
   END_RUNG
   // the same network as SCL:
   "TRANSFER DB".OUTPUT."PBV-82 CIP ISOLATION" := "AlwaysFALSE" AND ("MODE SELECTION DB"."MODE BUFF" <> 0);
END_REGION

REGION Network 55: PBV-83 PREMIX TRANSFER TO MFG VESSEL TRANSFER (TOP DISH)
   RUNG wire#powerrail
      Contact( "AlwaysTRUE" )
      { S7_Templates := "SrcType := Int" } EQ_Contact(in1 := "MODE SELECTION DB"."MODE BUFF", in2 := 2)
      { S7_Templates := "SrcType := Int" } EQ_Contact(in1 := "RECIRCULATION DB".PREMIXING.BUFF, in2 := 2)
      I_Contact( "RECIRCULATION DB".PREMIXING.PAUSE )
      Coil( "TRANSFER DB".OUTPUT."PBV-83 PREMIX TRANSFER TO MFG VESSEL TRANSFER (TOP DISH)" )
   END_RUNG
   // the same network as SCL:
   "TRANSFER DB".OUTPUT."PBV-83 PREMIX TRANSFER TO MFG VESSEL TRANSFER (TOP DISH)" := "AlwaysTRUE" AND ("MODE SELECTION DB"."MODE BUFF" = 2) AND ("RECIRCULATION DB".PREMIXING.BUFF = 2) AND NOT "RECIRCULATION DB".PREMIXING.PAUSE;
END_REGION

REGION Network 56: PBV-84 FROM TANK OUTLET TO CIP OUTLET
   RUNG wire#powerrail
      Contact( "AlwaysFALSE" )
      { S7_Templates := "SrcType := Int" } NE_Contact(in1 := "MODE SELECTION DB"."MODE BUFF", in2 := 0)
      Coil( "TRANSFER DB".OUTPUT."PBV-84 FROM TANK OUTLET TO CIP OUTLET" )
   END_RUNG
   // the same network as SCL:
   "TRANSFER DB".OUTPUT."PBV-84 FROM TANK OUTLET TO CIP OUTLET" := "AlwaysFALSE" AND ("MODE SELECTION DB"."MODE BUFF" <> 0);
END_REGION

REGION Network 57: PBV-85 SORBITOL INLET LINE
   RUNG wire#powerrail
      Contact( "AlwaysFALSE" )
      { S7_Templates := "SrcType := Int" } NE_Contact(in1 := "MODE SELECTION DB"."MODE BUFF", in2 := 0)
      Coil( "TRANSFER DB".OUTPUT."PBV-85 SORBITOL INLET LINE" )
   END_RUNG
   // the same network as SCL:
   "TRANSFER DB".OUTPUT."PBV-85 SORBITOL INLET LINE" := "AlwaysFALSE" AND ("MODE SELECTION DB"."MODE BUFF" <> 0);
END_REGION

REGION Network 58: PBV-86 GLUCOSE INLET LINE
   RUNG wire#powerrail
      Contact( "AlwaysFALSE" )
      { S7_Templates := "SrcType := Int" } NE_Contact(in1 := "MODE SELECTION DB"."MODE BUFF", in2 := 0)
      Coil( "TRANSFER DB".OUTPUT."PBV-86 GLUCOSE INLET LINE" )
   END_RUNG
   // the same network as SCL:
   "TRANSFER DB".OUTPUT."PBV-86 GLUCOSE INLET LINE" := "AlwaysFALSE" AND ("MODE SELECTION DB"."MODE BUFF" <> 0);
END_REGION

REGION Network 59: PBV-87 BASKET FILTER TO PREMIX VESSEL LINE
   RUNG wire#powerrail
      Contact( "AlwaysTRUE" )
      { S7_Templates := "SrcType := Int" } NE_Contact(in1 := "MODE SELECTION DB"."MODE BUFF", in2 := 0)
      Contact( "TRANSFER DB".BIT."SUGAR TO PREMIXING"."PBV-87 BASKET FILTER TO PREMIX VESSEL LINE" )
      Coil( "TRANSFER DB".OUTPUT."PBV-87 BASKET FILTER TO PREMIX VESSEL LINE" )
   END_RUNG
   // the same network as SCL:
   "TRANSFER DB".OUTPUT."PBV-87 BASKET FILTER TO PREMIX VESSEL LINE" := "AlwaysTRUE" AND ("MODE SELECTION DB"."MODE BUFF" <> 0) AND "TRANSFER DB".BIT."SUGAR TO PREMIXING"."PBV-87 BASKET FILTER TO PREMIX VESSEL LINE";
END_REGION

REGION Network 60: PBV-88 BASKET FILTER TRANSFER LINE
   RUNG wire#powerrail
      Contact( "AlwaysTRUE" )
      { S7_Templates := "SrcType := Int" } NE_Contact(in1 := "MODE SELECTION DB"."MODE BUFF", in2 := 0)
      Contact( "TRANSFER DB".BIT."SUGAR TO PREMIXING"."PBV-88 BASKET FILTER TRANSFER LINE" )
      Coil( "TRANSFER DB".OUTPUT."PBV-88 BASKET FILTER TRANSFER LINE" )
   END_RUNG
   // the same network as SCL:
   "TRANSFER DB".OUTPUT."PBV-88 BASKET FILTER TRANSFER LINE" := "AlwaysTRUE" AND ("MODE SELECTION DB"."MODE BUFF" <> 0) AND "TRANSFER DB".BIT."SUGAR TO PREMIXING"."PBV-88 BASKET FILTER TRANSFER LINE";
END_REGION

REGION Network 61: PBV-89 BASKET FILTER TO MFG INLET TRANSFER LINE
   RUNG wire#powerrail
      Contact( "AlwaysTRUE" )
      { S7_Templates := "SrcType := Int" } NE_Contact(in1 := "MODE SELECTION DB"."MODE BUFF", in2 := 0)
      Contact( "TRANSFER DB".BIT."SUGAR TO MFG"."PBV-89 BASKET FILTER TO MFG INLET TRANSFER LINE" )
      Coil( "TRANSFER DB".OUTPUT."PBV-89 BASKET FILTER TO MFG INLET TRANSFER LINE" )
   END_RUNG
   // the same network as SCL:
   "TRANSFER DB".OUTPUT."PBV-89 BASKET FILTER TO MFG INLET TRANSFER LINE" := "AlwaysTRUE" AND ("MODE SELECTION DB"."MODE BUFF" <> 0) AND "TRANSFER DB".BIT."SUGAR TO MFG"."PBV-89 BASKET FILTER TO MFG INLET TRANSFER LINE";
END_REGION

REGION Network 62: PBV-90 PREMIX TO MFG TRANSFER LINE
   RUNG wire#powerrail
      Contact( "AlwaysTRUE" )
      { S7_Templates := "SrcType := Int" } EQ_Contact(in1 := "MODE SELECTION DB"."MODE BUFF", in2 := 2)
      { S7_Templates := "SrcType := Int" } EQ_Contact(in1 := "RECIRCULATION DB".PREMIXING.BUFF, in2 := 2)
      I_Contact( "RECIRCULATION DB".PREMIXING.PAUSE )
      Coil( "TRANSFER DB".OUTPUT."PBV-90 PREMIX TO MFG TRANSFER LINE" )
   END_RUNG
   // the same network as SCL:
   "TRANSFER DB".OUTPUT."PBV-90 PREMIX TO MFG TRANSFER LINE" := "AlwaysTRUE" AND ("MODE SELECTION DB"."MODE BUFF" = 2) AND ("RECIRCULATION DB".PREMIXING.BUFF = 2) AND NOT "RECIRCULATION DB".PREMIXING.PAUSE;
END_REGION

REGION Network 63: PBV-91 PREMIX TO MFG TRANSFER LINE
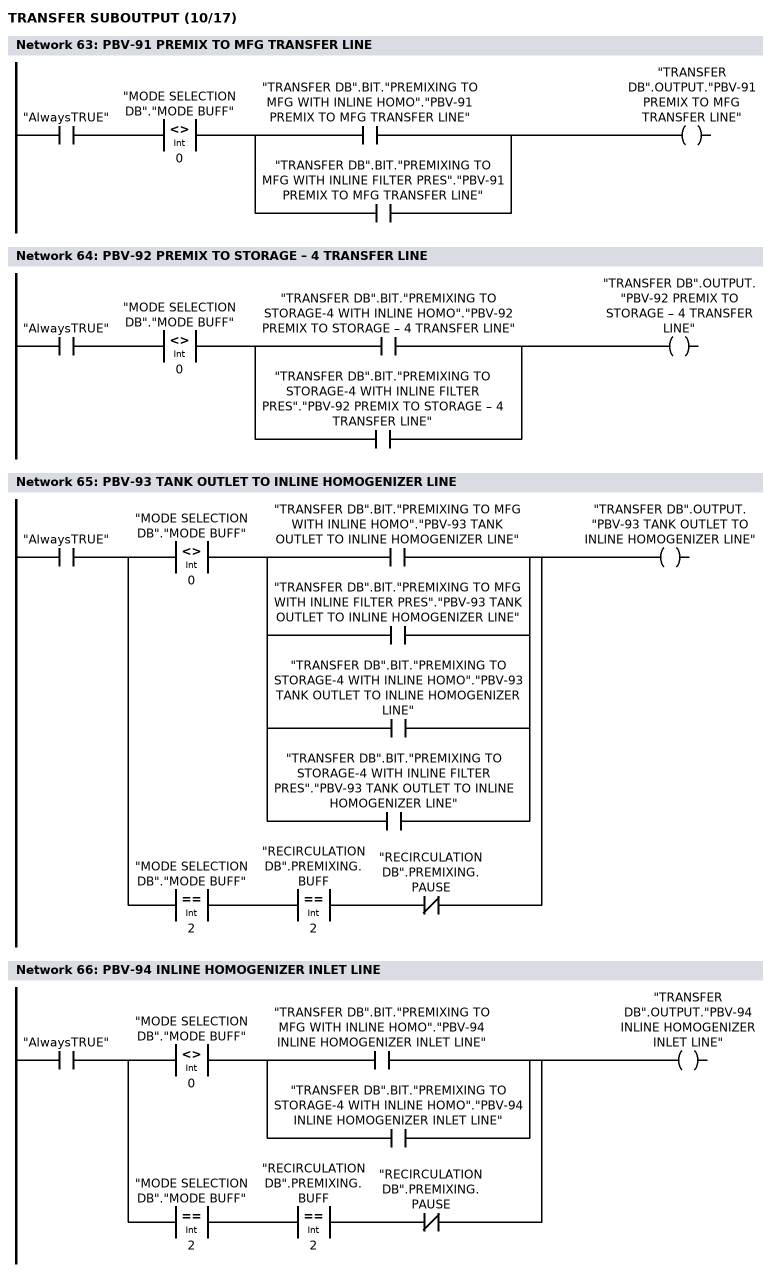
   RUNG wire#powerrail
      Contact( "AlwaysTRUE" )
      { S7_Templates := "SrcType := Int" } NE_Contact(in1 := "MODE SELECTION DB"."MODE BUFF", in2 := 0)
      wire#w1
      Contact( "TRANSFER DB".BIT."PREMIXING TO MFG WITH INLINE HOMO"."PBV-91 PREMIX TO MFG TRANSFER LINE" )
      wire#w2
      Coil( "TRANSFER DB".OUTPUT."PBV-91 PREMIX TO MFG TRANSFER LINE" )
   END_RUNG
   RUNG wire#w1
      Contact( "TRANSFER DB".BIT."PREMIXING TO MFG WITH INLINE FILTER PRES"."PBV-91 PREMIX TO MFG TRANSFER LINE" )
   END_RUNG wire#w2
   // the same network as SCL:
   "TRANSFER DB".OUTPUT."PBV-91 PREMIX TO MFG TRANSFER LINE" := "AlwaysTRUE" AND ("MODE SELECTION DB"."MODE BUFF" <> 0) AND ("TRANSFER DB".BIT."PREMIXING TO MFG WITH INLINE HOMO"."PBV-91 PREMIX TO MFG TRANSFER LINE" OR "TRANSFER DB".BIT."PREMIXING TO MFG WITH INLINE FILTER PRES"."PBV-91 PREMIX TO MFG TRANSFER LINE");
END_REGION

REGION Network 64: PBV-92 PREMIX TO STORAGE – 4 TRANSFER LINE
   RUNG wire#powerrail
      Contact( "AlwaysTRUE" )
      { S7_Templates := "SrcType := Int" } NE_Contact(in1 := "MODE SELECTION DB"."MODE BUFF", in2 := 0)
      wire#w1
      Contact( "TRANSFER DB".BIT."PREMIXING TO STORAGE-4 WITH INLINE HOMO"."PBV-92 PREMIX TO STORAGE – 4 TRANSFER LINE" )
      wire#w2
      Coil( "TRANSFER DB".OUTPUT."PBV-92 PREMIX TO STORAGE – 4 TRANSFER LINE" )
   END_RUNG
   RUNG wire#w1
      Contact( "TRANSFER DB".BIT."PREMIXING TO STORAGE-4 WITH INLINE FILTER PRES"."PBV-92 PREMIX TO STORAGE – 4 TRANSFER LINE" )
   END_RUNG wire#w2
   // the same network as SCL:
   "TRANSFER DB".OUTPUT."PBV-92 PREMIX TO STORAGE – 4 TRANSFER LINE" := "AlwaysTRUE" AND ("MODE SELECTION DB"."MODE BUFF" <> 0) AND ("TRANSFER DB".BIT."PREMIXING TO STORAGE-4 WITH INLINE HOMO"."PBV-92 PREMIX TO STORAGE – 4 TRANSFER LINE" OR "TRANSFER DB".BIT."PREMIXING TO STORAGE-4 WITH INLINE FILTER PRES"."PBV-92 PREMIX TO STORAGE – 4 TRANSFER LINE");
END_REGION

REGION Network 65: PBV-93 TANK OUTLET TO INLINE HOMOGENIZER LINE
   RUNG wire#powerrail
      Contact( "AlwaysTRUE" )
      wire#w1
      { S7_Templates := "SrcType := Int" } NE_Contact(in1 := "MODE SELECTION DB"."MODE BUFF", in2 := 0)
      wire#w2
      Contact( "TRANSFER DB".BIT."PREMIXING TO MFG WITH INLINE HOMO"."PBV-93 TANK OUTLET TO INLINE HOMOGENIZER LINE" )
      wire#w3
      Coil( "TRANSFER DB".OUTPUT."PBV-93 TANK OUTLET TO INLINE HOMOGENIZER LINE" )
   END_RUNG
   RUNG wire#w2
      Contact( "TRANSFER DB".BIT."PREMIXING TO MFG WITH INLINE FILTER PRES"."PBV-93 TANK OUTLET TO INLINE HOMOGENIZER LINE" )
   END_RUNG wire#w3
   RUNG wire#w2
      Contact( "TRANSFER DB".BIT."PREMIXING TO STORAGE-4 WITH INLINE HOMO"."PBV-93 TANK OUTLET TO INLINE HOMOGENIZER LINE" )
   END_RUNG wire#w3
   RUNG wire#w2
      Contact( "TRANSFER DB".BIT."PREMIXING TO STORAGE-4 WITH INLINE FILTER PRES"."PBV-93 TANK OUTLET TO INLINE HOMOGENIZER LINE" )
   END_RUNG wire#w3
   RUNG wire#w1
      { S7_Templates := "SrcType := Int" } EQ_Contact(in1 := "MODE SELECTION DB"."MODE BUFF", in2 := 2)
      { S7_Templates := "SrcType := Int" } EQ_Contact(in1 := "RECIRCULATION DB".PREMIXING.BUFF, in2 := 2)
      I_Contact( "RECIRCULATION DB".PREMIXING.PAUSE )
   END_RUNG wire#w3
   // the same network as SCL:
   "TRANSFER DB".OUTPUT."PBV-93 TANK OUTLET TO INLINE HOMOGENIZER LINE" := "AlwaysTRUE" AND ((("MODE SELECTION DB"."MODE BUFF" <> 0) AND ("TRANSFER DB".BIT."PREMIXING TO MFG WITH INLINE HOMO"."PBV-93 TANK OUTLET TO INLINE HOMOGENIZER LINE" OR "TRANSFER DB".BIT."PREMIXING TO MFG WITH INLINE FILTER PRES"."PBV-93 TANK OUTLET TO INLINE HOMOGENIZER LINE" OR "TRANSFER DB".BIT."PREMIXING TO STORAGE-4 WITH INLINE HOMO"."PBV-93 TANK OUTLET TO INLINE HOMOGENIZER LINE" OR "TRANSFER DB".BIT."PREMIXING TO STORAGE-4 WITH INLINE FILTER PRES"."PBV-93 TANK OUTLET TO INLINE HOMOGENIZER LINE")) OR (("MODE SELECTION DB"."MODE BUFF" = 2) AND ("RECIRCULATION DB".PREMIXING.BUFF = 2) AND NOT "RECIRCULATION DB".PREMIXING.PAUSE));
END_REGION

REGION Network 66: PBV-94 INLINE HOMOGENIZER INLET LINE
   RUNG wire#powerrail
      Contact( "AlwaysTRUE" )
      wire#w1
      { S7_Templates := "SrcType := Int" } NE_Contact(in1 := "MODE SELECTION DB"."MODE BUFF", in2 := 0)
      wire#w2
      Contact( "TRANSFER DB".BIT."PREMIXING TO MFG WITH INLINE HOMO"."PBV-94 INLINE HOMOGENIZER INLET LINE" )
      wire#w3
      Coil( "TRANSFER DB".OUTPUT."PBV-94 INLINE HOMOGENIZER INLET LINE" )
   END_RUNG
   RUNG wire#w2
      Contact( "TRANSFER DB".BIT."PREMIXING TO STORAGE-4 WITH INLINE HOMO"."PBV-94 INLINE HOMOGENIZER INLET LINE" )
   END_RUNG wire#w3
   RUNG wire#w1
      { S7_Templates := "SrcType := Int" } EQ_Contact(in1 := "MODE SELECTION DB"."MODE BUFF", in2 := 2)
      { S7_Templates := "SrcType := Int" } EQ_Contact(in1 := "RECIRCULATION DB".PREMIXING.BUFF, in2 := 2)
      I_Contact( "RECIRCULATION DB".PREMIXING.PAUSE )
   END_RUNG wire#w3
   // the same network as SCL:
   "TRANSFER DB".OUTPUT."PBV-94 INLINE HOMOGENIZER INLET LINE" := "AlwaysTRUE" AND ((("MODE SELECTION DB"."MODE BUFF" <> 0) AND ("TRANSFER DB".BIT."PREMIXING TO MFG WITH INLINE HOMO"."PBV-94 INLINE HOMOGENIZER INLET LINE" OR "TRANSFER DB".BIT."PREMIXING TO STORAGE-4 WITH INLINE HOMO"."PBV-94 INLINE HOMOGENIZER INLET LINE")) OR (("MODE SELECTION DB"."MODE BUFF" = 2) AND ("RECIRCULATION DB".PREMIXING.BUFF = 2) AND NOT "RECIRCULATION DB".PREMIXING.PAUSE));
END_REGION

REGION Network 67: PBV-95 TANK OUTLET TO FILTER PRESS LINE
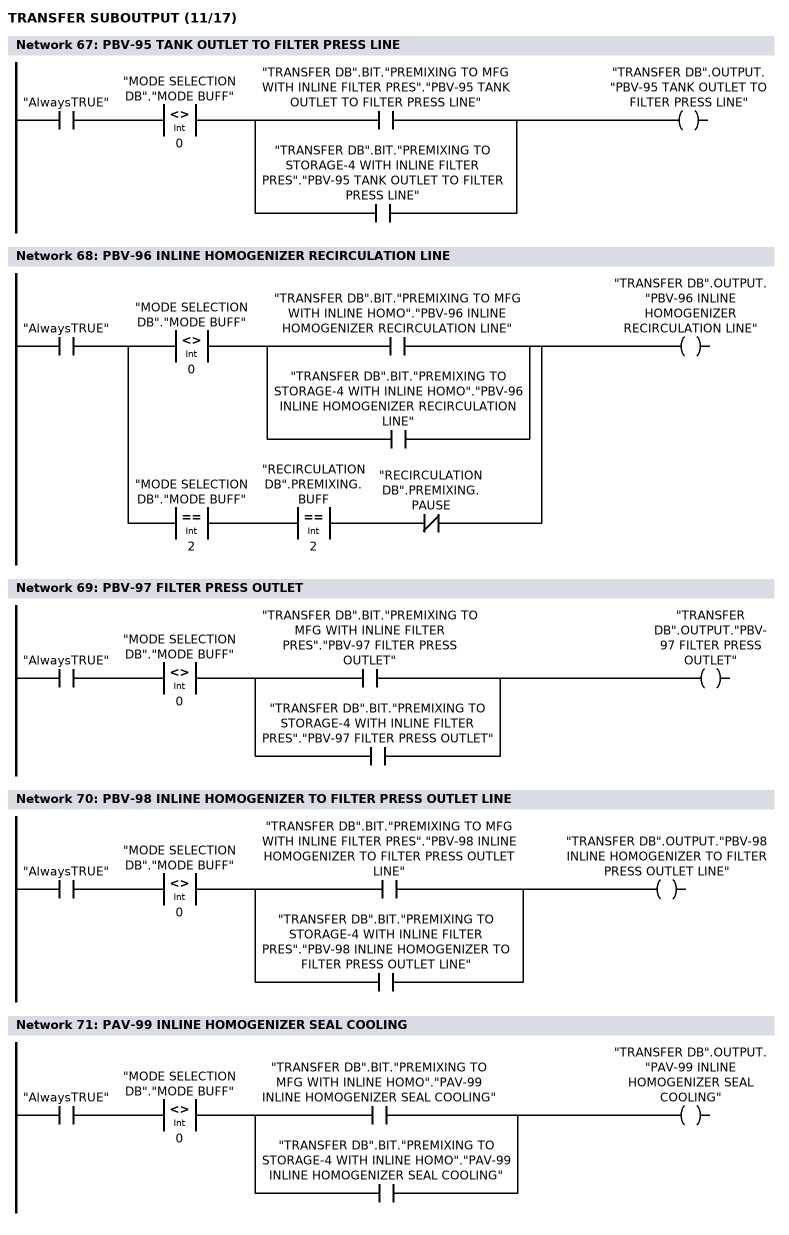
   RUNG wire#powerrail
      Contact( "AlwaysTRUE" )
      { S7_Templates := "SrcType := Int" } NE_Contact(in1 := "MODE SELECTION DB"."MODE BUFF", in2 := 0)
      wire#w1
      Contact( "TRANSFER DB".BIT."PREMIXING TO MFG WITH INLINE FILTER PRES"."PBV-95 TANK OUTLET TO FILTER PRESS LINE" )
      wire#w2
      Coil( "TRANSFER DB".OUTPUT."PBV-95 TANK OUTLET TO FILTER PRESS LINE" )
   END_RUNG
   RUNG wire#w1
      Contact( "TRANSFER DB".BIT."PREMIXING TO STORAGE-4 WITH INLINE FILTER PRES"."PBV-95 TANK OUTLET TO FILTER PRESS LINE" )
   END_RUNG wire#w2
   // the same network as SCL:
   "TRANSFER DB".OUTPUT."PBV-95 TANK OUTLET TO FILTER PRESS LINE" := "AlwaysTRUE" AND ("MODE SELECTION DB"."MODE BUFF" <> 0) AND ("TRANSFER DB".BIT."PREMIXING TO MFG WITH INLINE FILTER PRES"."PBV-95 TANK OUTLET TO FILTER PRESS LINE" OR "TRANSFER DB".BIT."PREMIXING TO STORAGE-4 WITH INLINE FILTER PRES"."PBV-95 TANK OUTLET TO FILTER PRESS LINE");
END_REGION

REGION Network 68: PBV-96 INLINE HOMOGENIZER RECIRCULATION LINE
   RUNG wire#powerrail
      Contact( "AlwaysTRUE" )
      wire#w1
      { S7_Templates := "SrcType := Int" } NE_Contact(in1 := "MODE SELECTION DB"."MODE BUFF", in2 := 0)
      wire#w2
      Contact( "TRANSFER DB".BIT."PREMIXING TO MFG WITH INLINE HOMO"."PBV-96 INLINE HOMOGENIZER RECIRCULATION LINE" )
      wire#w3
      Coil( "TRANSFER DB".OUTPUT."PBV-96 INLINE HOMOGENIZER RECIRCULATION LINE" )
   END_RUNG
   RUNG wire#w2
      Contact( "TRANSFER DB".BIT."PREMIXING TO STORAGE-4 WITH INLINE HOMO"."PBV-96 INLINE HOMOGENIZER RECIRCULATION LINE" )
   END_RUNG wire#w3
   RUNG wire#w1
      { S7_Templates := "SrcType := Int" } EQ_Contact(in1 := "MODE SELECTION DB"."MODE BUFF", in2 := 2)
      { S7_Templates := "SrcType := Int" } EQ_Contact(in1 := "RECIRCULATION DB".PREMIXING.BUFF, in2 := 2)
      I_Contact( "RECIRCULATION DB".PREMIXING.PAUSE )
   END_RUNG wire#w3
   // the same network as SCL:
   "TRANSFER DB".OUTPUT."PBV-96 INLINE HOMOGENIZER RECIRCULATION LINE" := "AlwaysTRUE" AND ((("MODE SELECTION DB"."MODE BUFF" <> 0) AND ("TRANSFER DB".BIT."PREMIXING TO MFG WITH INLINE HOMO"."PBV-96 INLINE HOMOGENIZER RECIRCULATION LINE" OR "TRANSFER DB".BIT."PREMIXING TO STORAGE-4 WITH INLINE HOMO"."PBV-96 INLINE HOMOGENIZER RECIRCULATION LINE")) OR (("MODE SELECTION DB"."MODE BUFF" = 2) AND ("RECIRCULATION DB".PREMIXING.BUFF = 2) AND NOT "RECIRCULATION DB".PREMIXING.PAUSE));
END_REGION

REGION Network 69: PBV-97 FILTER PRESS OUTLET
   RUNG wire#powerrail
      Contact( "AlwaysTRUE" )
      { S7_Templates := "SrcType := Int" } NE_Contact(in1 := "MODE SELECTION DB"."MODE BUFF", in2 := 0)
      wire#w1
      Contact( "TRANSFER DB".BIT."PREMIXING TO MFG WITH INLINE FILTER PRES"."PBV-97 FILTER PRESS OUTLET" )
      wire#w2
      Coil( "TRANSFER DB".OUTPUT."PBV-97 FILTER PRESS OUTLET" )
   END_RUNG
   RUNG wire#w1
      Contact( "TRANSFER DB".BIT."PREMIXING TO STORAGE-4 WITH INLINE FILTER PRES"."PBV-97 FILTER PRESS OUTLET" )
   END_RUNG wire#w2
   // the same network as SCL:
   "TRANSFER DB".OUTPUT."PBV-97 FILTER PRESS OUTLET" := "AlwaysTRUE" AND ("MODE SELECTION DB"."MODE BUFF" <> 0) AND ("TRANSFER DB".BIT."PREMIXING TO MFG WITH INLINE FILTER PRES"."PBV-97 FILTER PRESS OUTLET" OR "TRANSFER DB".BIT."PREMIXING TO STORAGE-4 WITH INLINE FILTER PRES"."PBV-97 FILTER PRESS OUTLET");
END_REGION

REGION Network 70: PBV-98 INLINE HOMOGENIZER TO FILTER PRESS OUTLET LINE
   RUNG wire#powerrail
      Contact( "AlwaysTRUE" )
      { S7_Templates := "SrcType := Int" } NE_Contact(in1 := "MODE SELECTION DB"."MODE BUFF", in2 := 0)
      wire#w1
      Contact( "TRANSFER DB".BIT."PREMIXING TO MFG WITH INLINE FILTER PRES"."PBV-98 INLINE HOMOGENIZER TO FILTER PRESS OUTLET LINE" )
      wire#w2
      Coil( "TRANSFER DB".OUTPUT."PBV-98 INLINE HOMOGENIZER TO FILTER PRESS OUTLET LINE" )
   END_RUNG
   RUNG wire#w1
      Contact( "TRANSFER DB".BIT."PREMIXING TO STORAGE-4 WITH INLINE FILTER PRES"."PBV-98 INLINE HOMOGENIZER TO FILTER PRESS OUTLET LINE" )
   END_RUNG wire#w2
   // the same network as SCL:
   "TRANSFER DB".OUTPUT."PBV-98 INLINE HOMOGENIZER TO FILTER PRESS OUTLET LINE" := "AlwaysTRUE" AND ("MODE SELECTION DB"."MODE BUFF" <> 0) AND ("TRANSFER DB".BIT."PREMIXING TO MFG WITH INLINE FILTER PRES"."PBV-98 INLINE HOMOGENIZER TO FILTER PRESS OUTLET LINE" OR "TRANSFER DB".BIT."PREMIXING TO STORAGE-4 WITH INLINE FILTER PRES"."PBV-98 INLINE HOMOGENIZER TO FILTER PRESS OUTLET LINE");
END_REGION

REGION Network 71: PAV-99 INLINE HOMOGENIZER SEAL COOLING
   RUNG wire#powerrail
      Contact( "AlwaysTRUE" )
      { S7_Templates := "SrcType := Int" } NE_Contact(in1 := "MODE SELECTION DB"."MODE BUFF", in2 := 0)
      wire#w1
      Contact( "TRANSFER DB".BIT."PREMIXING TO MFG WITH INLINE HOMO"."PAV-99 INLINE HOMOGENIZER SEAL COOLING" )
      wire#w2
      Coil( "TRANSFER DB".OUTPUT."PAV-99 INLINE HOMOGENIZER SEAL COOLING" )
   END_RUNG
   RUNG wire#w1
      Contact( "TRANSFER DB".BIT."PREMIXING TO STORAGE-4 WITH INLINE HOMO"."PAV-99 INLINE HOMOGENIZER SEAL COOLING" )
   END_RUNG wire#w2
   // the same network as SCL:
   "TRANSFER DB".OUTPUT."PAV-99 INLINE HOMOGENIZER SEAL COOLING" := "AlwaysTRUE" AND ("MODE SELECTION DB"."MODE BUFF" <> 0) AND ("TRANSFER DB".BIT."PREMIXING TO MFG WITH INLINE HOMO"."PAV-99 INLINE HOMOGENIZER SEAL COOLING" OR "TRANSFER DB".BIT."PREMIXING TO STORAGE-4 WITH INLINE HOMO"."PAV-99 INLINE HOMOGENIZER SEAL COOLING");
END_REGION

REGION Network 72: PBV-100 FILTER PRESS INLET
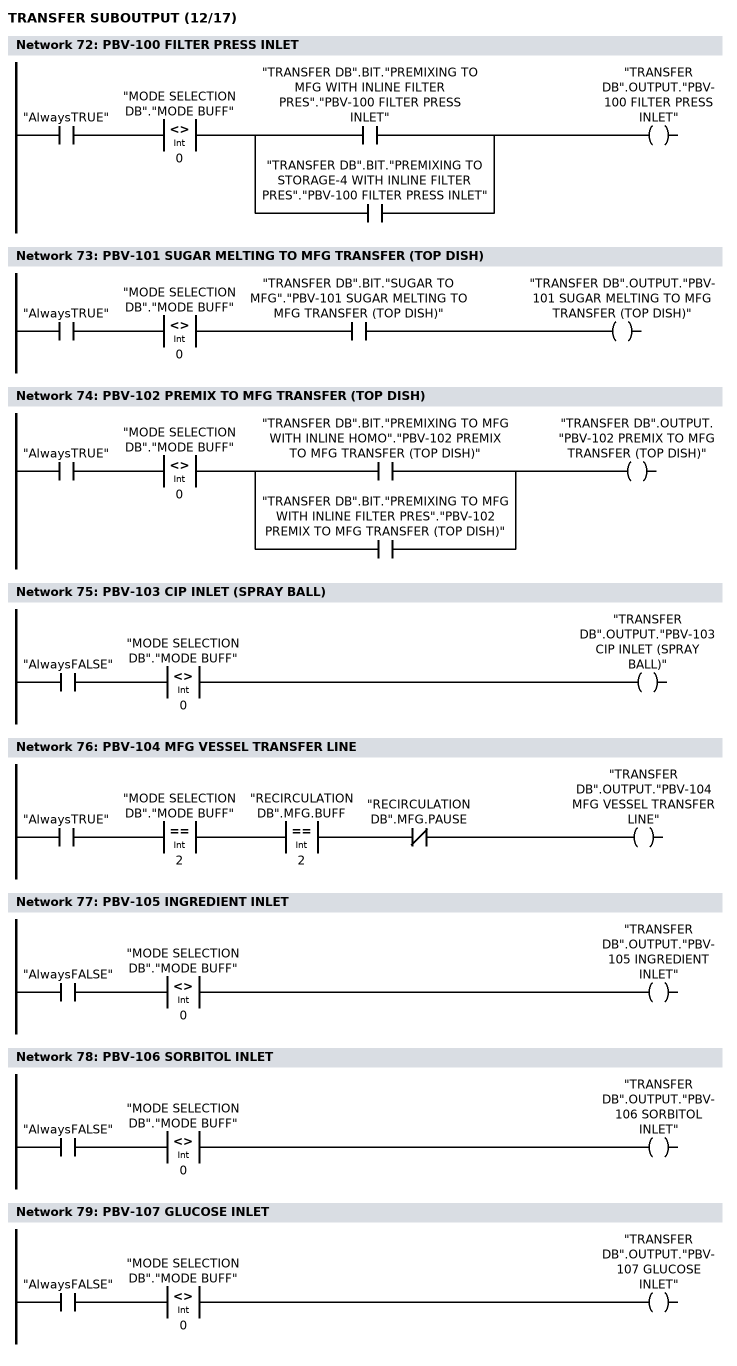
   RUNG wire#powerrail
      Contact( "AlwaysTRUE" )
      { S7_Templates := "SrcType := Int" } NE_Contact(in1 := "MODE SELECTION DB"."MODE BUFF", in2 := 0)
      wire#w1
      Contact( "TRANSFER DB".BIT."PREMIXING TO MFG WITH INLINE FILTER PRES"."PBV-100 FILTER PRESS INLET" )
      wire#w2
      Coil( "TRANSFER DB".OUTPUT."PBV-100 FILTER PRESS INLET" )
   END_RUNG
   RUNG wire#w1
      Contact( "TRANSFER DB".BIT."PREMIXING TO STORAGE-4 WITH INLINE FILTER PRES"."PBV-100 FILTER PRESS INLET" )
   END_RUNG wire#w2
   // the same network as SCL:
   "TRANSFER DB".OUTPUT."PBV-100 FILTER PRESS INLET" := "AlwaysTRUE" AND ("MODE SELECTION DB"."MODE BUFF" <> 0) AND ("TRANSFER DB".BIT."PREMIXING TO MFG WITH INLINE FILTER PRES"."PBV-100 FILTER PRESS INLET" OR "TRANSFER DB".BIT."PREMIXING TO STORAGE-4 WITH INLINE FILTER PRES"."PBV-100 FILTER PRESS INLET");
END_REGION

REGION Network 73: PBV-101 SUGAR MELTING TO MFG TRANSFER (TOP DISH)
   RUNG wire#powerrail
      Contact( "AlwaysTRUE" )
      { S7_Templates := "SrcType := Int" } NE_Contact(in1 := "MODE SELECTION DB"."MODE BUFF", in2 := 0)
      Contact( "TRANSFER DB".BIT."SUGAR TO MFG"."PBV-101 SUGAR MELTING TO MFG TRANSFER (TOP DISH)" )
      Coil( "TRANSFER DB".OUTPUT."PBV-101 SUGAR MELTING TO MFG TRANSFER (TOP DISH)" )
   END_RUNG
   // the same network as SCL:
   "TRANSFER DB".OUTPUT."PBV-101 SUGAR MELTING TO MFG TRANSFER (TOP DISH)" := "AlwaysTRUE" AND ("MODE SELECTION DB"."MODE BUFF" <> 0) AND "TRANSFER DB".BIT."SUGAR TO MFG"."PBV-101 SUGAR MELTING TO MFG TRANSFER (TOP DISH)";
END_REGION

REGION Network 74: PBV-102 PREMIX TO MFG TRANSFER (TOP DISH)
   RUNG wire#powerrail
      Contact( "AlwaysTRUE" )
      { S7_Templates := "SrcType := Int" } NE_Contact(in1 := "MODE SELECTION DB"."MODE BUFF", in2 := 0)
      wire#w1
      Contact( "TRANSFER DB".BIT."PREMIXING TO MFG WITH INLINE HOMO"."PBV-102 PREMIX TO MFG TRANSFER (TOP DISH)" )
      wire#w2
      Coil( "TRANSFER DB".OUTPUT."PBV-102 PREMIX TO MFG TRANSFER (TOP DISH)" )
   END_RUNG
   RUNG wire#w1
      Contact( "TRANSFER DB".BIT."PREMIXING TO MFG WITH INLINE FILTER PRES"."PBV-102 PREMIX TO MFG TRANSFER (TOP DISH)" )
   END_RUNG wire#w2
   // the same network as SCL:
   "TRANSFER DB".OUTPUT."PBV-102 PREMIX TO MFG TRANSFER (TOP DISH)" := "AlwaysTRUE" AND ("MODE SELECTION DB"."MODE BUFF" <> 0) AND ("TRANSFER DB".BIT."PREMIXING TO MFG WITH INLINE HOMO"."PBV-102 PREMIX TO MFG TRANSFER (TOP DISH)" OR "TRANSFER DB".BIT."PREMIXING TO MFG WITH INLINE FILTER PRES"."PBV-102 PREMIX TO MFG TRANSFER (TOP DISH)");
END_REGION

REGION Network 75: PBV-103 CIP INLET (SPRAY BALL)
   RUNG wire#powerrail
      Contact( "AlwaysFALSE" )
      { S7_Templates := "SrcType := Int" } NE_Contact(in1 := "MODE SELECTION DB"."MODE BUFF", in2 := 0)
      Coil( "TRANSFER DB".OUTPUT."PBV-103 CIP INLET (SPRAY BALL)" )
   END_RUNG
   // the same network as SCL:
   "TRANSFER DB".OUTPUT."PBV-103 CIP INLET (SPRAY BALL)" := "AlwaysFALSE" AND ("MODE SELECTION DB"."MODE BUFF" <> 0);
END_REGION

REGION Network 76: PBV-104 MFG VESSEL TRANSFER LINE
   RUNG wire#powerrail
      Contact( "AlwaysTRUE" )
      { S7_Templates := "SrcType := Int" } EQ_Contact(in1 := "MODE SELECTION DB"."MODE BUFF", in2 := 2)
      { S7_Templates := "SrcType := Int" } EQ_Contact(in1 := "RECIRCULATION DB".MFG.BUFF, in2 := 2)
      I_Contact( "RECIRCULATION DB".MFG.PAUSE )
      Coil( "TRANSFER DB".OUTPUT."PBV-104 MFG VESSEL TRANSFER LINE" )
   END_RUNG
   // the same network as SCL:
   "TRANSFER DB".OUTPUT."PBV-104 MFG VESSEL TRANSFER LINE" := "AlwaysTRUE" AND ("MODE SELECTION DB"."MODE BUFF" = 2) AND ("RECIRCULATION DB".MFG.BUFF = 2) AND NOT "RECIRCULATION DB".MFG.PAUSE;
END_REGION

REGION Network 77: PBV-105 INGREDIENT INLET
   RUNG wire#powerrail
      Contact( "AlwaysFALSE" )
      { S7_Templates := "SrcType := Int" } NE_Contact(in1 := "MODE SELECTION DB"."MODE BUFF", in2 := 0)
      Coil( "TRANSFER DB".OUTPUT."PBV-105 INGREDIENT INLET" )
   END_RUNG
   // the same network as SCL:
   "TRANSFER DB".OUTPUT."PBV-105 INGREDIENT INLET" := "AlwaysFALSE" AND ("MODE SELECTION DB"."MODE BUFF" <> 0);
END_REGION

REGION Network 78: PBV-106 SORBITOL INLET
   RUNG wire#powerrail
      Contact( "AlwaysFALSE" )
      { S7_Templates := "SrcType := Int" } NE_Contact(in1 := "MODE SELECTION DB"."MODE BUFF", in2 := 0)
      Coil( "TRANSFER DB".OUTPUT."PBV-106 SORBITOL INLET" )
   END_RUNG
   // the same network as SCL:
   "TRANSFER DB".OUTPUT."PBV-106 SORBITOL INLET" := "AlwaysFALSE" AND ("MODE SELECTION DB"."MODE BUFF" <> 0);
END_REGION

REGION Network 79: PBV-107 GLUCOSE INLET
   RUNG wire#powerrail
      Contact( "AlwaysFALSE" )
      { S7_Templates := "SrcType := Int" } NE_Contact(in1 := "MODE SELECTION DB"."MODE BUFF", in2 := 0)
      Coil( "TRANSFER DB".OUTPUT."PBV-107 GLUCOSE INLET" )
   END_RUNG
   // the same network as SCL:
   "TRANSFER DB".OUTPUT."PBV-107 GLUCOSE INLET" := "AlwaysFALSE" AND ("MODE SELECTION DB"."MODE BUFF" <> 0);
END_REGION

REGION Network 80: PBV-108 INLINE HOMOGENIZER TO FILTER PRESS INLET LINE
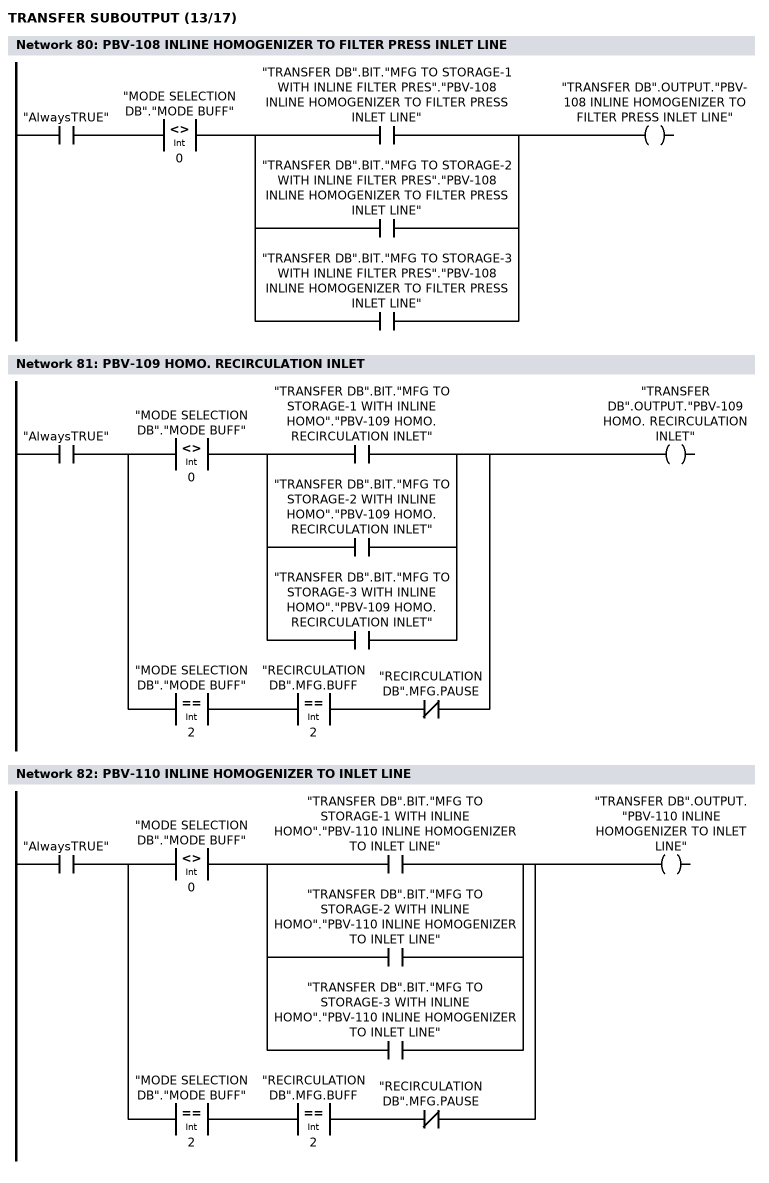
   RUNG wire#powerrail
      Contact( "AlwaysTRUE" )
      { S7_Templates := "SrcType := Int" } NE_Contact(in1 := "MODE SELECTION DB"."MODE BUFF", in2 := 0)
      wire#w1
      Contact( "TRANSFER DB".BIT."MFG TO STORAGE-1 WITH INLINE FILTER PRES"."PBV-108 INLINE HOMOGENIZER TO FILTER PRESS INLET LINE" )
      wire#w2
      Coil( "TRANSFER DB".OUTPUT."PBV-108 INLINE HOMOGENIZER TO FILTER PRESS INLET LINE" )
   END_RUNG
   RUNG wire#w1
      Contact( "TRANSFER DB".BIT."MFG TO STORAGE-2 WITH INLINE FILTER PRES"."PBV-108 INLINE HOMOGENIZER TO FILTER PRESS INLET LINE" )
   END_RUNG wire#w2
   RUNG wire#w1
      Contact( "TRANSFER DB".BIT."MFG TO STORAGE-3 WITH INLINE FILTER PRES"."PBV-108 INLINE HOMOGENIZER TO FILTER PRESS INLET LINE" )
   END_RUNG wire#w2
   // the same network as SCL:
   "TRANSFER DB".OUTPUT."PBV-108 INLINE HOMOGENIZER TO FILTER PRESS INLET LINE" := "AlwaysTRUE" AND ("MODE SELECTION DB"."MODE BUFF" <> 0) AND ("TRANSFER DB".BIT."MFG TO STORAGE-1 WITH INLINE FILTER PRES"."PBV-108 INLINE HOMOGENIZER TO FILTER PRESS INLET LINE" OR "TRANSFER DB".BIT."MFG TO STORAGE-2 WITH INLINE FILTER PRES"."PBV-108 INLINE HOMOGENIZER TO FILTER PRESS INLET LINE" OR "TRANSFER DB".BIT."MFG TO STORAGE-3 WITH INLINE FILTER PRES"."PBV-108 INLINE HOMOGENIZER TO FILTER PRESS INLET LINE");
END_REGION

REGION Network 81: PBV-109 HOMO. RECIRCULATION INLET
   RUNG wire#powerrail
      Contact( "AlwaysTRUE" )
      wire#w1
      { S7_Templates := "SrcType := Int" } NE_Contact(in1 := "MODE SELECTION DB"."MODE BUFF", in2 := 0)
      wire#w2
      Contact( "TRANSFER DB".BIT."MFG TO STORAGE-1 WITH INLINE HOMO"."PBV-109 HOMO. RECIRCULATION INLET" )
      wire#w3
      Coil( "TRANSFER DB".OUTPUT."PBV-109 HOMO. RECIRCULATION INLET" )
   END_RUNG
   RUNG wire#w2
      Contact( "TRANSFER DB".BIT."MFG TO STORAGE-2 WITH INLINE HOMO"."PBV-109 HOMO. RECIRCULATION INLET" )
   END_RUNG wire#w3
   RUNG wire#w2
      Contact( "TRANSFER DB".BIT."MFG TO STORAGE-3 WITH INLINE HOMO"."PBV-109 HOMO. RECIRCULATION INLET" )
   END_RUNG wire#w3
   RUNG wire#w1
      { S7_Templates := "SrcType := Int" } EQ_Contact(in1 := "MODE SELECTION DB"."MODE BUFF", in2 := 2)
      { S7_Templates := "SrcType := Int" } EQ_Contact(in1 := "RECIRCULATION DB".MFG.BUFF, in2 := 2)
      I_Contact( "RECIRCULATION DB".MFG.PAUSE )
   END_RUNG wire#w3
   // the same network as SCL:
   "TRANSFER DB".OUTPUT."PBV-109 HOMO. RECIRCULATION INLET" := "AlwaysTRUE" AND ((("MODE SELECTION DB"."MODE BUFF" <> 0) AND ("TRANSFER DB".BIT."MFG TO STORAGE-1 WITH INLINE HOMO"."PBV-109 HOMO. RECIRCULATION INLET" OR "TRANSFER DB".BIT."MFG TO STORAGE-2 WITH INLINE HOMO"."PBV-109 HOMO. RECIRCULATION INLET" OR "TRANSFER DB".BIT."MFG TO STORAGE-3 WITH INLINE HOMO"."PBV-109 HOMO. RECIRCULATION INLET")) OR (("MODE SELECTION DB"."MODE BUFF" = 2) AND ("RECIRCULATION DB".MFG.BUFF = 2) AND NOT "RECIRCULATION DB".MFG.PAUSE));
END_REGION

REGION Network 82: PBV-110 INLINE HOMOGENIZER TO INLET LINE
   RUNG wire#powerrail
      Contact( "AlwaysTRUE" )
      wire#w1
      { S7_Templates := "SrcType := Int" } NE_Contact(in1 := "MODE SELECTION DB"."MODE BUFF", in2 := 0)
      wire#w2
      Contact( "TRANSFER DB".BIT."MFG TO STORAGE-1 WITH INLINE HOMO"."PBV-110 INLINE HOMOGENIZER TO INLET LINE" )
      wire#w3
      Coil( "TRANSFER DB".OUTPUT."PBV-110 INLINE HOMOGENIZER TO INLET LINE" )
   END_RUNG
   RUNG wire#w2
      Contact( "TRANSFER DB".BIT."MFG TO STORAGE-2 WITH INLINE HOMO"."PBV-110 INLINE HOMOGENIZER TO INLET LINE" )
   END_RUNG wire#w3
   RUNG wire#w2
      Contact( "TRANSFER DB".BIT."MFG TO STORAGE-3 WITH INLINE HOMO"."PBV-110 INLINE HOMOGENIZER TO INLET LINE" )
   END_RUNG wire#w3
   RUNG wire#w1
      { S7_Templates := "SrcType := Int" } EQ_Contact(in1 := "MODE SELECTION DB"."MODE BUFF", in2 := 2)
      { S7_Templates := "SrcType := Int" } EQ_Contact(in1 := "RECIRCULATION DB".MFG.BUFF, in2 := 2)
      I_Contact( "RECIRCULATION DB".MFG.PAUSE )
   END_RUNG wire#w3
   // the same network as SCL:
   "TRANSFER DB".OUTPUT."PBV-110 INLINE HOMOGENIZER TO INLET LINE" := "AlwaysTRUE" AND ((("MODE SELECTION DB"."MODE BUFF" <> 0) AND ("TRANSFER DB".BIT."MFG TO STORAGE-1 WITH INLINE HOMO"."PBV-110 INLINE HOMOGENIZER TO INLET LINE" OR "TRANSFER DB".BIT."MFG TO STORAGE-2 WITH INLINE HOMO"."PBV-110 INLINE HOMOGENIZER TO INLET LINE" OR "TRANSFER DB".BIT."MFG TO STORAGE-3 WITH INLINE HOMO"."PBV-110 INLINE HOMOGENIZER TO INLET LINE")) OR (("MODE SELECTION DB"."MODE BUFF" = 2) AND ("RECIRCULATION DB".MFG.BUFF = 2) AND NOT "RECIRCULATION DB".MFG.PAUSE));
END_REGION

REGION Network 83: PBV-111 FILTER PRESS OUTLER VALVE
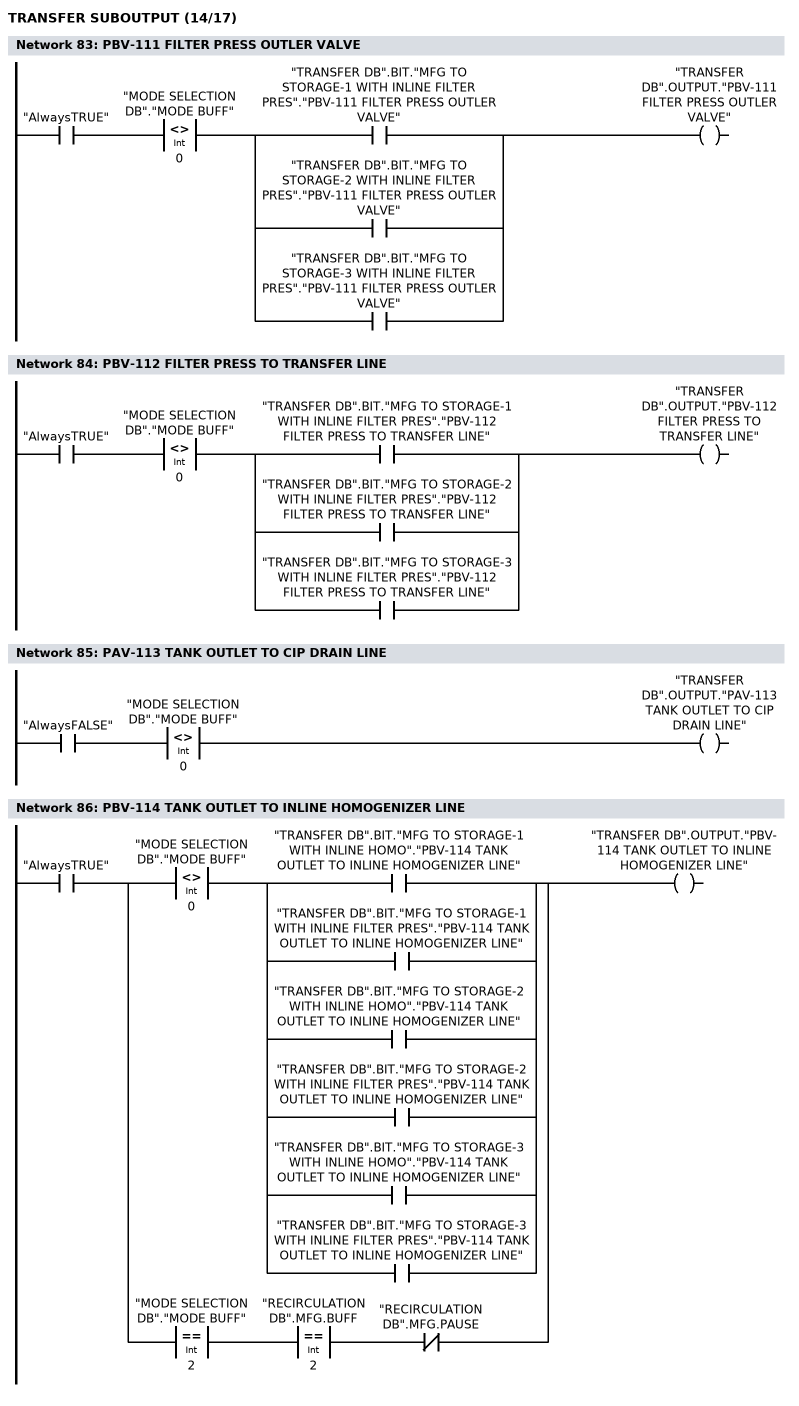
   RUNG wire#powerrail
      Contact( "AlwaysTRUE" )
      { S7_Templates := "SrcType := Int" } NE_Contact(in1 := "MODE SELECTION DB"."MODE BUFF", in2 := 0)
      wire#w1
      Contact( "TRANSFER DB".BIT."MFG TO STORAGE-1 WITH INLINE FILTER PRES"."PBV-111 FILTER PRESS OUTLER VALVE" )
      wire#w2
      Coil( "TRANSFER DB".OUTPUT."PBV-111 FILTER PRESS OUTLER VALVE" )
   END_RUNG
   RUNG wire#w1
      Contact( "TRANSFER DB".BIT."MFG TO STORAGE-2 WITH INLINE FILTER PRES"."PBV-111 FILTER PRESS OUTLER VALVE" )
   END_RUNG wire#w2
   RUNG wire#w1
      Contact( "TRANSFER DB".BIT."MFG TO STORAGE-3 WITH INLINE FILTER PRES"."PBV-111 FILTER PRESS OUTLER VALVE" )
   END_RUNG wire#w2
   // the same network as SCL:
   "TRANSFER DB".OUTPUT."PBV-111 FILTER PRESS OUTLER VALVE" := "AlwaysTRUE" AND ("MODE SELECTION DB"."MODE BUFF" <> 0) AND ("TRANSFER DB".BIT."MFG TO STORAGE-1 WITH INLINE FILTER PRES"."PBV-111 FILTER PRESS OUTLER VALVE" OR "TRANSFER DB".BIT."MFG TO STORAGE-2 WITH INLINE FILTER PRES"."PBV-111 FILTER PRESS OUTLER VALVE" OR "TRANSFER DB".BIT."MFG TO STORAGE-3 WITH INLINE FILTER PRES"."PBV-111 FILTER PRESS OUTLER VALVE");
END_REGION

REGION Network 84: PBV-112 FILTER PRESS TO TRANSFER LINE
   RUNG wire#powerrail
      Contact( "AlwaysTRUE" )
      { S7_Templates := "SrcType := Int" } NE_Contact(in1 := "MODE SELECTION DB"."MODE BUFF", in2 := 0)
      wire#w1
      Contact( "TRANSFER DB".BIT."MFG TO STORAGE-1 WITH INLINE FILTER PRES"."PBV-112 FILTER PRESS TO TRANSFER LINE" )
      wire#w2
      Coil( "TRANSFER DB".OUTPUT."PBV-112 FILTER PRESS TO TRANSFER LINE" )
   END_RUNG
   RUNG wire#w1
      Contact( "TRANSFER DB".BIT."MFG TO STORAGE-2 WITH INLINE FILTER PRES"."PBV-112 FILTER PRESS TO TRANSFER LINE" )
   END_RUNG wire#w2
   RUNG wire#w1
      Contact( "TRANSFER DB".BIT."MFG TO STORAGE-3 WITH INLINE FILTER PRES"."PBV-112 FILTER PRESS TO TRANSFER LINE" )
   END_RUNG wire#w2
   // the same network as SCL:
   "TRANSFER DB".OUTPUT."PBV-112 FILTER PRESS TO TRANSFER LINE" := "AlwaysTRUE" AND ("MODE SELECTION DB"."MODE BUFF" <> 0) AND ("TRANSFER DB".BIT."MFG TO STORAGE-1 WITH INLINE FILTER PRES"."PBV-112 FILTER PRESS TO TRANSFER LINE" OR "TRANSFER DB".BIT."MFG TO STORAGE-2 WITH INLINE FILTER PRES"."PBV-112 FILTER PRESS TO TRANSFER LINE" OR "TRANSFER DB".BIT."MFG TO STORAGE-3 WITH INLINE FILTER PRES"."PBV-112 FILTER PRESS TO TRANSFER LINE");
END_REGION

REGION Network 85: PAV-113 TANK OUTLET TO CIP DRAIN LINE
   RUNG wire#powerrail
      Contact( "AlwaysFALSE" )
      { S7_Templates := "SrcType := Int" } NE_Contact(in1 := "MODE SELECTION DB"."MODE BUFF", in2 := 0)
      Coil( "TRANSFER DB".OUTPUT."PAV-113 TANK OUTLET TO CIP DRAIN LINE" )
   END_RUNG
   // the same network as SCL:
   "TRANSFER DB".OUTPUT."PAV-113 TANK OUTLET TO CIP DRAIN LINE" := "AlwaysFALSE" AND ("MODE SELECTION DB"."MODE BUFF" <> 0);
END_REGION

REGION Network 86: PBV-114 TANK OUTLET TO INLINE HOMOGENIZER LINE
   RUNG wire#powerrail
      Contact( "AlwaysTRUE" )
      wire#w1
      { S7_Templates := "SrcType := Int" } NE_Contact(in1 := "MODE SELECTION DB"."MODE BUFF", in2 := 0)
      wire#w2
      Contact( "TRANSFER DB".BIT."MFG TO STORAGE-1 WITH INLINE HOMO"."PBV-114 TANK OUTLET TO INLINE HOMOGENIZER LINE" )
      wire#w3
      Coil( "TRANSFER DB".OUTPUT."PBV-114 TANK OUTLET TO INLINE HOMOGENIZER LINE" )
   END_RUNG
   RUNG wire#w2
      Contact( "TRANSFER DB".BIT."MFG TO STORAGE-1 WITH INLINE FILTER PRES"."PBV-114 TANK OUTLET TO INLINE HOMOGENIZER LINE" )
   END_RUNG wire#w3
   RUNG wire#w2
      Contact( "TRANSFER DB".BIT."MFG TO STORAGE-2 WITH INLINE HOMO"."PBV-114 TANK OUTLET TO INLINE HOMOGENIZER LINE" )
   END_RUNG wire#w3
   RUNG wire#w2
      Contact( "TRANSFER DB".BIT."MFG TO STORAGE-2 WITH INLINE FILTER PRES"."PBV-114 TANK OUTLET TO INLINE HOMOGENIZER LINE" )
   END_RUNG wire#w3
   RUNG wire#w2
      Contact( "TRANSFER DB".BIT."MFG TO STORAGE-3 WITH INLINE HOMO"."PBV-114 TANK OUTLET TO INLINE HOMOGENIZER LINE" )
   END_RUNG wire#w3
   RUNG wire#w2
      Contact( "TRANSFER DB".BIT."MFG TO STORAGE-3 WITH INLINE FILTER PRES"."PBV-114 TANK OUTLET TO INLINE HOMOGENIZER LINE" )
   END_RUNG wire#w3
   RUNG wire#w1
      { S7_Templates := "SrcType := Int" } EQ_Contact(in1 := "MODE SELECTION DB"."MODE BUFF", in2 := 2)
      { S7_Templates := "SrcType := Int" } EQ_Contact(in1 := "RECIRCULATION DB".MFG.BUFF, in2 := 2)
      I_Contact( "RECIRCULATION DB".MFG.PAUSE )
   END_RUNG wire#w3
   // the same network as SCL:
   "TRANSFER DB".OUTPUT."PBV-114 TANK OUTLET TO INLINE HOMOGENIZER LINE" := "AlwaysTRUE" AND ((("MODE SELECTION DB"."MODE BUFF" <> 0) AND ("TRANSFER DB".BIT."MFG TO STORAGE-1 WITH INLINE HOMO"."PBV-114 TANK OUTLET TO INLINE HOMOGENIZER LINE" OR "TRANSFER DB".BIT."MFG TO STORAGE-1 WITH INLINE FILTER PRES"."PBV-114 TANK OUTLET TO INLINE HOMOGENIZER LINE" OR "TRANSFER DB".BIT."MFG TO STORAGE-2 WITH INLINE HOMO"."PBV-114 TANK OUTLET TO INLINE HOMOGENIZER LINE" OR "TRANSFER DB".BIT."MFG TO STORAGE-2 WITH INLINE FILTER PRES"."PBV-114 TANK OUTLET TO INLINE HOMOGENIZER LINE" OR "TRANSFER DB".BIT."MFG TO STORAGE-3 WITH INLINE HOMO"."PBV-114 TANK OUTLET TO INLINE HOMOGENIZER LINE" OR "TRANSFER DB".BIT."MFG TO STORAGE-3 WITH INLINE FILTER PRES"."PBV-114 TANK OUTLET TO INLINE HOMOGENIZER LINE")) OR (("MODE SELECTION DB"."MODE BUFF" = 2) AND ("RECIRCULATION DB".MFG.BUFF = 2) AND NOT "RECIRCULATION DB".MFG.PAUSE));
END_REGION

REGION Network 87: PBV-115 MFG TO STORAGE – 1 TRANSFER LINE
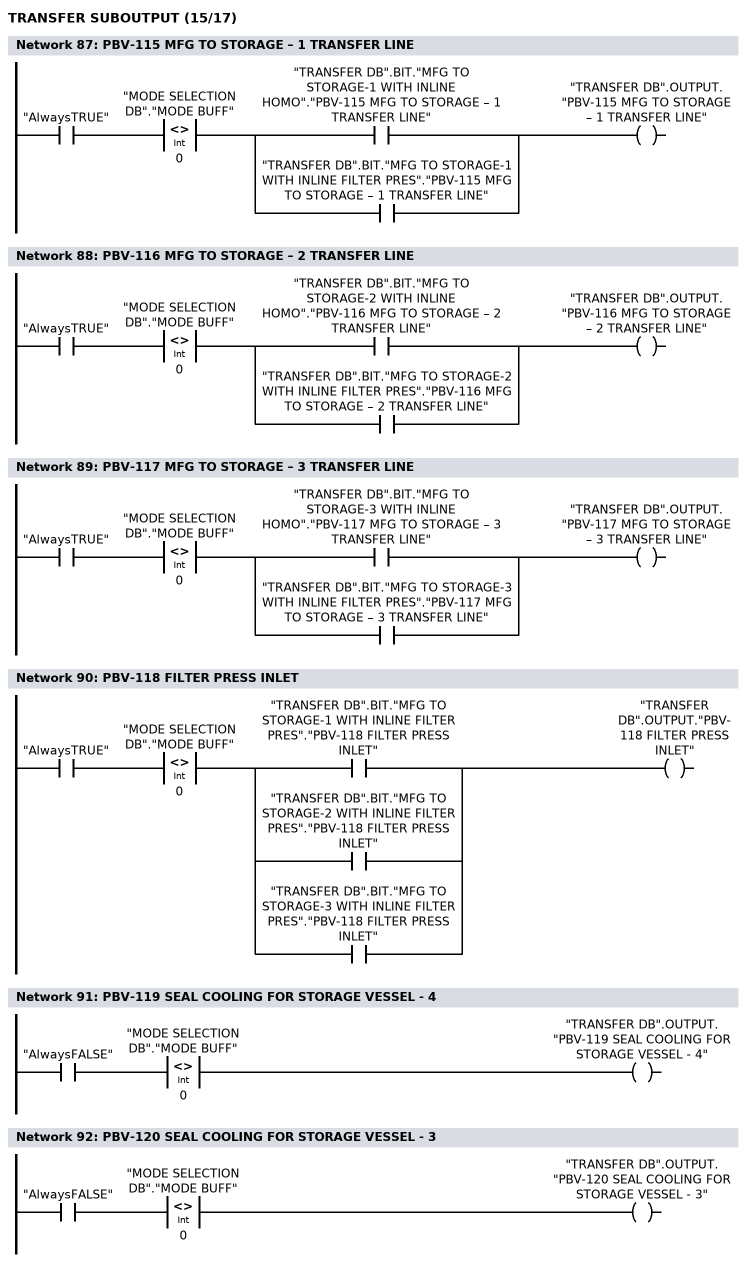
   RUNG wire#powerrail
      Contact( "AlwaysTRUE" )
      { S7_Templates := "SrcType := Int" } NE_Contact(in1 := "MODE SELECTION DB"."MODE BUFF", in2 := 0)
      wire#w1
      Contact( "TRANSFER DB".BIT."MFG TO STORAGE-1 WITH INLINE HOMO"."PBV-115 MFG TO STORAGE – 1 TRANSFER LINE" )
      wire#w2
      Coil( "TRANSFER DB".OUTPUT."PBV-115 MFG TO STORAGE – 1 TRANSFER LINE" )
   END_RUNG
   RUNG wire#w1
      Contact( "TRANSFER DB".BIT."MFG TO STORAGE-1 WITH INLINE FILTER PRES"."PBV-115 MFG TO STORAGE – 1 TRANSFER LINE" )
   END_RUNG wire#w2
   // the same network as SCL:
   "TRANSFER DB".OUTPUT."PBV-115 MFG TO STORAGE – 1 TRANSFER LINE" := "AlwaysTRUE" AND ("MODE SELECTION DB"."MODE BUFF" <> 0) AND ("TRANSFER DB".BIT."MFG TO STORAGE-1 WITH INLINE HOMO"."PBV-115 MFG TO STORAGE – 1 TRANSFER LINE" OR "TRANSFER DB".BIT."MFG TO STORAGE-1 WITH INLINE FILTER PRES"."PBV-115 MFG TO STORAGE – 1 TRANSFER LINE");
END_REGION

REGION Network 88: PBV-116 MFG TO STORAGE – 2 TRANSFER LINE
   RUNG wire#powerrail
      Contact( "AlwaysTRUE" )
      { S7_Templates := "SrcType := Int" } NE_Contact(in1 := "MODE SELECTION DB"."MODE BUFF", in2 := 0)
      wire#w1
      Contact( "TRANSFER DB".BIT."MFG TO STORAGE-2 WITH INLINE HOMO"."PBV-116 MFG TO STORAGE – 2 TRANSFER LINE" )
      wire#w2
      Coil( "TRANSFER DB".OUTPUT."PBV-116 MFG TO STORAGE – 2 TRANSFER LINE" )
   END_RUNG
   RUNG wire#w1
      Contact( "TRANSFER DB".BIT."MFG TO STORAGE-2 WITH INLINE FILTER PRES"."PBV-116 MFG TO STORAGE – 2 TRANSFER LINE" )
   END_RUNG wire#w2
   // the same network as SCL:
   "TRANSFER DB".OUTPUT."PBV-116 MFG TO STORAGE – 2 TRANSFER LINE" := "AlwaysTRUE" AND ("MODE SELECTION DB"."MODE BUFF" <> 0) AND ("TRANSFER DB".BIT."MFG TO STORAGE-2 WITH INLINE HOMO"."PBV-116 MFG TO STORAGE – 2 TRANSFER LINE" OR "TRANSFER DB".BIT."MFG TO STORAGE-2 WITH INLINE FILTER PRES"."PBV-116 MFG TO STORAGE – 2 TRANSFER LINE");
END_REGION

REGION Network 89: PBV-117 MFG TO STORAGE – 3 TRANSFER LINE
   RUNG wire#powerrail
      Contact( "AlwaysTRUE" )
      { S7_Templates := "SrcType := Int" } NE_Contact(in1 := "MODE SELECTION DB"."MODE BUFF", in2 := 0)
      wire#w1
      Contact( "TRANSFER DB".BIT."MFG TO STORAGE-3 WITH INLINE HOMO"."PBV-117 MFG TO STORAGE – 3 TRANSFER LINE" )
      wire#w2
      Coil( "TRANSFER DB".OUTPUT."PBV-117 MFG TO STORAGE – 3 TRANSFER LINE" )
   END_RUNG
   RUNG wire#w1
      Contact( "TRANSFER DB".BIT."MFG TO STORAGE-3 WITH INLINE FILTER PRES"."PBV-117 MFG TO STORAGE – 3 TRANSFER LINE" )
   END_RUNG wire#w2
   // the same network as SCL:
   "TRANSFER DB".OUTPUT."PBV-117 MFG TO STORAGE – 3 TRANSFER LINE" := "AlwaysTRUE" AND ("MODE SELECTION DB"."MODE BUFF" <> 0) AND ("TRANSFER DB".BIT."MFG TO STORAGE-3 WITH INLINE HOMO"."PBV-117 MFG TO STORAGE – 3 TRANSFER LINE" OR "TRANSFER DB".BIT."MFG TO STORAGE-3 WITH INLINE FILTER PRES"."PBV-117 MFG TO STORAGE – 3 TRANSFER LINE");
END_REGION

REGION Network 90: PBV-118 FILTER PRESS INLET
   RUNG wire#powerrail
      Contact( "AlwaysTRUE" )
      { S7_Templates := "SrcType := Int" } NE_Contact(in1 := "MODE SELECTION DB"."MODE BUFF", in2 := 0)
      wire#w1
      Contact( "TRANSFER DB".BIT."MFG TO STORAGE-1 WITH INLINE FILTER PRES"."PBV-118 FILTER PRESS INLET" )
      wire#w2
      Coil( "TRANSFER DB".OUTPUT."PBV-118 FILTER PRESS INLET" )
   END_RUNG
   RUNG wire#w1
      Contact( "TRANSFER DB".BIT."MFG TO STORAGE-2 WITH INLINE FILTER PRES"."PBV-118 FILTER PRESS INLET" )
   END_RUNG wire#w2
   RUNG wire#w1
      Contact( "TRANSFER DB".BIT."MFG TO STORAGE-3 WITH INLINE FILTER PRES"."PBV-118 FILTER PRESS INLET" )
   END_RUNG wire#w2
   // the same network as SCL:
   "TRANSFER DB".OUTPUT."PBV-118 FILTER PRESS INLET" := "AlwaysTRUE" AND ("MODE SELECTION DB"."MODE BUFF" <> 0) AND ("TRANSFER DB".BIT."MFG TO STORAGE-1 WITH INLINE FILTER PRES"."PBV-118 FILTER PRESS INLET" OR "TRANSFER DB".BIT."MFG TO STORAGE-2 WITH INLINE FILTER PRES"."PBV-118 FILTER PRESS INLET" OR "TRANSFER DB".BIT."MFG TO STORAGE-3 WITH INLINE FILTER PRES"."PBV-118 FILTER PRESS INLET");
END_REGION

REGION Network 91: PBV-119 SEAL COOLING FOR STORAGE VESSEL - 4
   RUNG wire#powerrail
      Contact( "AlwaysFALSE" )
      { S7_Templates := "SrcType := Int" } NE_Contact(in1 := "MODE SELECTION DB"."MODE BUFF", in2 := 0)
      Coil( "TRANSFER DB".OUTPUT."PBV-119 SEAL COOLING FOR STORAGE VESSEL - 4" )
   END_RUNG
   // the same network as SCL:
   "TRANSFER DB".OUTPUT."PBV-119 SEAL COOLING FOR STORAGE VESSEL - 4" := "AlwaysFALSE" AND ("MODE SELECTION DB"."MODE BUFF" <> 0);
END_REGION

REGION Network 92: PBV-120 SEAL COOLING FOR STORAGE VESSEL - 3
   RUNG wire#powerrail
      Contact( "AlwaysFALSE" )
      { S7_Templates := "SrcType := Int" } NE_Contact(in1 := "MODE SELECTION DB"."MODE BUFF", in2 := 0)
      Coil( "TRANSFER DB".OUTPUT."PBV-120 SEAL COOLING FOR STORAGE VESSEL - 3" )
   END_RUNG
   // the same network as SCL:
   "TRANSFER DB".OUTPUT."PBV-120 SEAL COOLING FOR STORAGE VESSEL - 3" := "AlwaysFALSE" AND ("MODE SELECTION DB"."MODE BUFF" <> 0);
END_REGION

REGION Network 93: PBV-121 SEAL COOLING FOR STORAGE VESSEL - 2
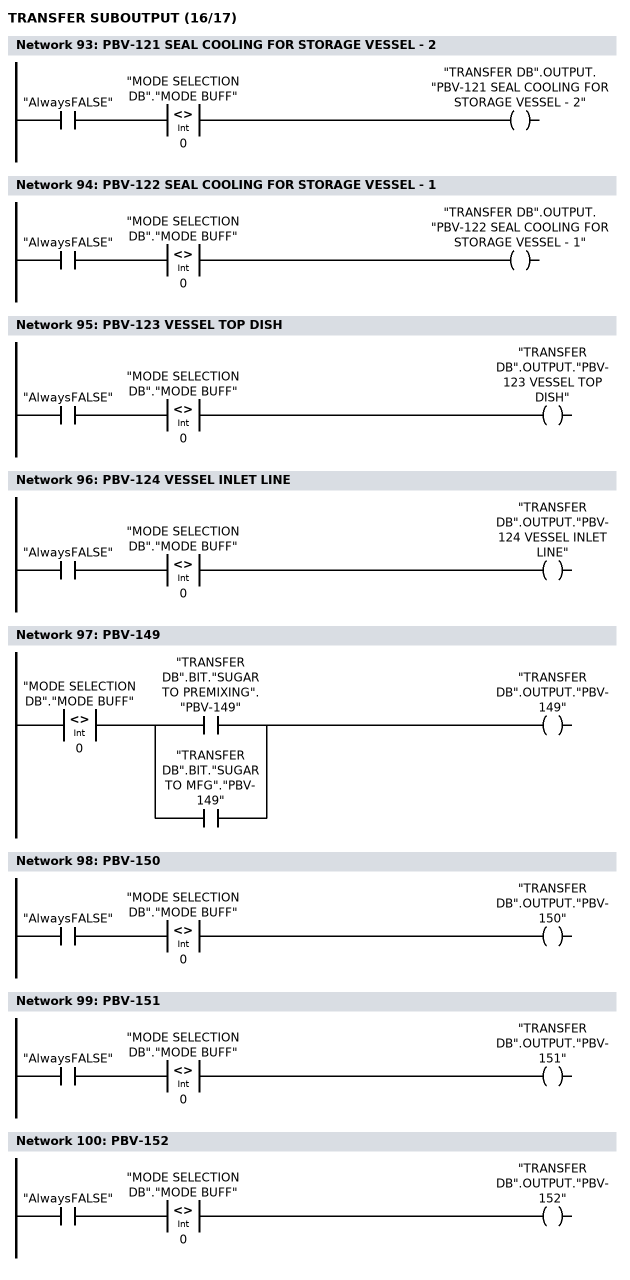
   RUNG wire#powerrail
      Contact( "AlwaysFALSE" )
      { S7_Templates := "SrcType := Int" } NE_Contact(in1 := "MODE SELECTION DB"."MODE BUFF", in2 := 0)
      Coil( "TRANSFER DB".OUTPUT."PBV-121 SEAL COOLING FOR STORAGE VESSEL - 2" )
   END_RUNG
   // the same network as SCL:
   "TRANSFER DB".OUTPUT."PBV-121 SEAL COOLING FOR STORAGE VESSEL - 2" := "AlwaysFALSE" AND ("MODE SELECTION DB"."MODE BUFF" <> 0);
END_REGION

REGION Network 94: PBV-122 SEAL COOLING FOR STORAGE VESSEL - 1
   RUNG wire#powerrail
      Contact( "AlwaysFALSE" )
      { S7_Templates := "SrcType := Int" } NE_Contact(in1 := "MODE SELECTION DB"."MODE BUFF", in2 := 0)
      Coil( "TRANSFER DB".OUTPUT."PBV-122 SEAL COOLING FOR STORAGE VESSEL - 1" )
   END_RUNG
   // the same network as SCL:
   "TRANSFER DB".OUTPUT."PBV-122 SEAL COOLING FOR STORAGE VESSEL - 1" := "AlwaysFALSE" AND ("MODE SELECTION DB"."MODE BUFF" <> 0);
END_REGION

REGION Network 95: PBV-123 VESSEL TOP DISH
   RUNG wire#powerrail
      Contact( "AlwaysFALSE" )
      { S7_Templates := "SrcType := Int" } NE_Contact(in1 := "MODE SELECTION DB"."MODE BUFF", in2 := 0)
      Coil( "TRANSFER DB".OUTPUT."PBV-123 VESSEL TOP DISH" )
   END_RUNG
   // the same network as SCL:
   "TRANSFER DB".OUTPUT."PBV-123 VESSEL TOP DISH" := "AlwaysFALSE" AND ("MODE SELECTION DB"."MODE BUFF" <> 0);
END_REGION

REGION Network 96: PBV-124 VESSEL INLET LINE
   RUNG wire#powerrail
      Contact( "AlwaysFALSE" )
      { S7_Templates := "SrcType := Int" } NE_Contact(in1 := "MODE SELECTION DB"."MODE BUFF", in2 := 0)
      Coil( "TRANSFER DB".OUTPUT."PBV-124 VESSEL INLET LINE" )
   END_RUNG
   // the same network as SCL:
   "TRANSFER DB".OUTPUT."PBV-124 VESSEL INLET LINE" := "AlwaysFALSE" AND ("MODE SELECTION DB"."MODE BUFF" <> 0);
END_REGION

REGION Network 97: PBV-149
   RUNG wire#powerrail
      { S7_Templates := "SrcType := Int" } NE_Contact(in1 := "MODE SELECTION DB"."MODE BUFF", in2 := 0)
      wire#w1
      Contact( "TRANSFER DB".BIT."SUGAR TO PREMIXING"."PBV-149" )
      wire#w2
      Coil( "TRANSFER DB".OUTPUT."PBV-149" )
   END_RUNG
   RUNG wire#w1
      Contact( "TRANSFER DB".BIT."SUGAR TO MFG"."PBV-149" )
   END_RUNG wire#w2
   // the same network as SCL:
   "TRANSFER DB".OUTPUT."PBV-149" := ("MODE SELECTION DB"."MODE BUFF" <> 0) AND ("TRANSFER DB".BIT."SUGAR TO PREMIXING"."PBV-149" OR "TRANSFER DB".BIT."SUGAR TO MFG"."PBV-149");
END_REGION

REGION Network 98: PBV-150
   RUNG wire#powerrail
      Contact( "AlwaysFALSE" )
      { S7_Templates := "SrcType := Int" } NE_Contact(in1 := "MODE SELECTION DB"."MODE BUFF", in2 := 0)
      Coil( "TRANSFER DB".OUTPUT."PBV-150" )
   END_RUNG
   // the same network as SCL:
   "TRANSFER DB".OUTPUT."PBV-150" := "AlwaysFALSE" AND ("MODE SELECTION DB"."MODE BUFF" <> 0);
END_REGION

REGION Network 99: PBV-151
   RUNG wire#powerrail
      Contact( "AlwaysFALSE" )
      { S7_Templates := "SrcType := Int" } NE_Contact(in1 := "MODE SELECTION DB"."MODE BUFF", in2 := 0)
      Coil( "TRANSFER DB".OUTPUT."PBV-151" )
   END_RUNG
   // the same network as SCL:
   "TRANSFER DB".OUTPUT."PBV-151" := "AlwaysFALSE" AND ("MODE SELECTION DB"."MODE BUFF" <> 0);
END_REGION

REGION Network 100: PBV-152
   RUNG wire#powerrail
      Contact( "AlwaysFALSE" )
      { S7_Templates := "SrcType := Int" } NE_Contact(in1 := "MODE SELECTION DB"."MODE BUFF", in2 := 0)
      Coil( "TRANSFER DB".OUTPUT."PBV-152" )
   END_RUNG
   // the same network as SCL:
   "TRANSFER DB".OUTPUT."PBV-152" := "AlwaysFALSE" AND ("MODE SELECTION DB"."MODE BUFF" <> 0);
END_REGION

REGION Network 101: PBV-153
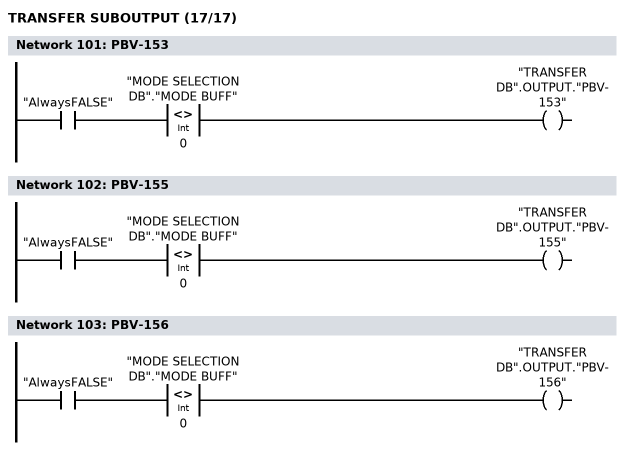
   RUNG wire#powerrail
      Contact( "AlwaysFALSE" )
      { S7_Templates := "SrcType := Int" } NE_Contact(in1 := "MODE SELECTION DB"."MODE BUFF", in2 := 0)
      Coil( "TRANSFER DB".OUTPUT."PBV-153" )
   END_RUNG
   // the same network as SCL:
   "TRANSFER DB".OUTPUT."PBV-153" := "AlwaysFALSE" AND ("MODE SELECTION DB"."MODE BUFF" <> 0);
END_REGION

REGION Network 102: PBV-155
   RUNG wire#powerrail
      Contact( "AlwaysFALSE" )
      { S7_Templates := "SrcType := Int" } NE_Contact(in1 := "MODE SELECTION DB"."MODE BUFF", in2 := 0)
      Coil( "TRANSFER DB".OUTPUT."PBV-155" )
   END_RUNG
   // the same network as SCL:
   "TRANSFER DB".OUTPUT."PBV-155" := "AlwaysFALSE" AND ("MODE SELECTION DB"."MODE BUFF" <> 0);
END_REGION

REGION Network 103: PBV-156
   RUNG wire#powerrail
      Contact( "AlwaysFALSE" )
      { S7_Templates := "SrcType := Int" } NE_Contact(in1 := "MODE SELECTION DB"."MODE BUFF", in2 := 0)
      Coil( "TRANSFER DB".OUTPUT."PBV-156" )
   END_RUNG
   // the same network as SCL:
   "TRANSFER DB".OUTPUT."PBV-156" := "AlwaysFALSE" AND ("MODE SELECTION DB"."MODE BUFF" <> 0);
END_REGION
END_FUNCTION

FUNCTION "MODE SELECTION" : Void   // FC2, LAD
{ S7_Optimized_Access := 'TRUE' }
// stored: SetENOAutomatically false
   VAR_TEMP   // added for the SCL form of the ladder/FBD networks
      _w1 : Bool;
   END_VAR
BEGIN

REGION Network 1: STANDBY
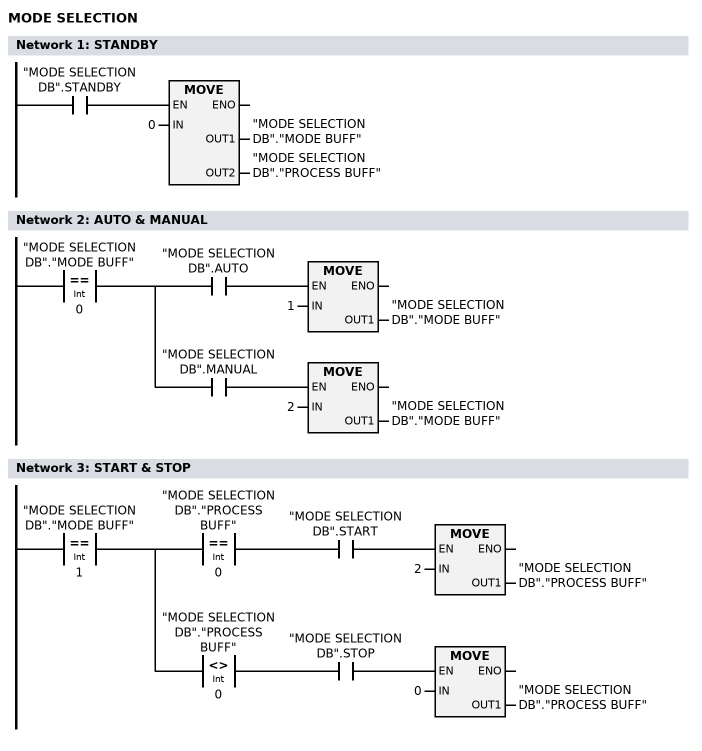
   RUNG wire#powerrail
      Contact( "MODE SELECTION DB".STANDBY )
      Move(in := 0, out1 => "MODE SELECTION DB"."MODE BUFF", out2 => "MODE SELECTION DB"."PROCESS BUFF")
   END_RUNG
   // the same network as SCL:
   IF "MODE SELECTION DB".STANDBY THEN
       "MODE SELECTION DB"."MODE BUFF" := 0;
       "MODE SELECTION DB"."PROCESS BUFF" := 0;
   END_IF;
END_REGION

REGION Network 2: AUTO & MANUAL
   RUNG wire#powerrail
      { S7_Templates := "SrcType := Int" } EQ_Contact(in1 := "MODE SELECTION DB"."MODE BUFF", in2 := 0)
      wire#w1
      Contact( "MODE SELECTION DB".AUTO )
      Move(in := 1, out1 => "MODE SELECTION DB"."MODE BUFF")
   END_RUNG
   RUNG wire#w1
      Contact( "MODE SELECTION DB".MANUAL )
      Move(in := 2, out1 => "MODE SELECTION DB"."MODE BUFF")
   END_RUNG
   // the same network as SCL:
   #_w1 := "MODE SELECTION DB"."MODE BUFF" = 0;
   IF #_w1 AND "MODE SELECTION DB".AUTO THEN "MODE SELECTION DB"."MODE BUFF" := 1; END_IF;
   IF #_w1 AND "MODE SELECTION DB".MANUAL THEN "MODE SELECTION DB"."MODE BUFF" := 2; END_IF;
END_REGION

REGION Network 3: START & STOP
   RUNG wire#powerrail
      { S7_Templates := "SrcType := Int" } EQ_Contact(in1 := "MODE SELECTION DB"."MODE BUFF", in2 := 1)
      wire#w1
      { S7_Templates := "SrcType := Int" } EQ_Contact(in1 := "MODE SELECTION DB"."PROCESS BUFF", in2 := 0)
      Contact( "MODE SELECTION DB".START )
      Move(in := 2, out1 => "MODE SELECTION DB"."PROCESS BUFF")
   END_RUNG
   RUNG wire#w1
      { S7_Templates := "SrcType := Int" } NE_Contact(in1 := "MODE SELECTION DB"."PROCESS BUFF", in2 := 0)
      Contact( "MODE SELECTION DB".STOP )
      Move(in := 0, out1 => "MODE SELECTION DB"."PROCESS BUFF")
   END_RUNG
   // the same network as SCL:
   #_w1 := "MODE SELECTION DB"."MODE BUFF" = 1;
   IF #_w1 AND ("MODE SELECTION DB"."PROCESS BUFF" = 0) AND "MODE SELECTION DB".START THEN
       "MODE SELECTION DB"."PROCESS BUFF" := 2;
   END_IF;
   IF #_w1 AND ("MODE SELECTION DB"."PROCESS BUFF" <> 0) AND "MODE SELECTION DB".STOP THEN
       "MODE SELECTION DB"."PROCESS BUFF" := 0;
   END_IF;
END_REGION
END_FUNCTION

FUNCTION "ALARM" : Void   // FC10, LAD
{ S7_Optimized_Access := 'TRUE' }
// stored: SetENOAutomatically false
   VAR_TEMP   // added for the SCL form of the ladder/FBD networks
      _w1 : Bool;
   END_VAR
BEGIN

REGION Network 1: HOOTER RESET
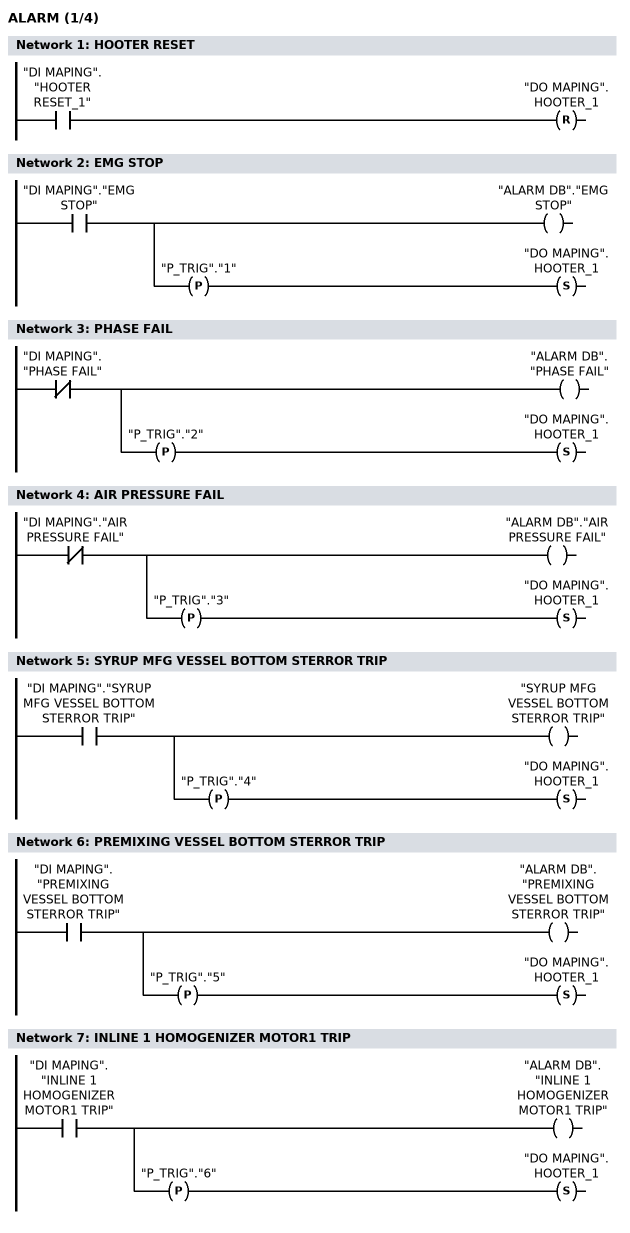
   RUNG wire#powerrail
      Contact( "DI MAPING"."HOOTER RESET_1" )
      R_Coil( "DO MAPING".HOOTER_1 )
   END_RUNG
   // the same network as SCL:
   IF "DI MAPING"."HOOTER RESET_1" THEN "DO MAPING".HOOTER_1 := FALSE; END_IF;
END_REGION

REGION Network 2: EMG STOP
   RUNG wire#powerrail
      Contact( "DI MAPING"."EMG STOP" )
      wire#w1
      Coil( "ALARM DB"."EMG STOP" )
   END_RUNG
   RUNG wire#w1
      P_Trig( "P_TRIG"."1" )
      S_Coil( "DO MAPING".HOOTER_1 )
   END_RUNG
   // the same network as SCL:
   "ALARM DB"."EMG STOP" := "DI MAPING"."EMG STOP";
   #_w1 := "DI MAPING"."EMG STOP" AND NOT "P_TRIG"."1";   // rising edge
   "P_TRIG"."1" := "DI MAPING"."EMG STOP";
   IF #_w1 THEN "DO MAPING".HOOTER_1 := TRUE; END_IF;
END_REGION

REGION Network 3: PHASE FAIL
   RUNG wire#powerrail
      I_Contact( "DI MAPING"."PHASE FAIL" )
      wire#w1
      Coil( "ALARM DB"."PHASE FAIL" )
   END_RUNG
   RUNG wire#w1
      P_Trig( "P_TRIG"."2" )
      S_Coil( "DO MAPING".HOOTER_1 )
   END_RUNG
   // the same network as SCL:
   "ALARM DB"."PHASE FAIL" := NOT "DI MAPING"."PHASE FAIL";
   #_w1 := NOT "DI MAPING"."PHASE FAIL" AND NOT "P_TRIG"."2";   // rising edge
   "P_TRIG"."2" := NOT "DI MAPING"."PHASE FAIL";
   IF #_w1 THEN "DO MAPING".HOOTER_1 := TRUE; END_IF;
END_REGION

REGION Network 4: AIR PRESSURE FAIL
   RUNG wire#powerrail
      I_Contact( "DI MAPING"."AIR PRESSURE FAIL" )
      wire#w1
      Coil( "ALARM DB"."AIR PRESSURE FAIL" )
   END_RUNG
   RUNG wire#w1
      P_Trig( "P_TRIG"."3" )
      S_Coil( "DO MAPING".HOOTER_1 )
   END_RUNG
   // the same network as SCL:
   "ALARM DB"."AIR PRESSURE FAIL" := NOT "DI MAPING"."AIR PRESSURE FAIL";
   #_w1 := NOT "DI MAPING"."AIR PRESSURE FAIL" AND NOT "P_TRIG"."3";   // rising edge
   "P_TRIG"."3" := NOT "DI MAPING"."AIR PRESSURE FAIL";
   IF #_w1 THEN "DO MAPING".HOOTER_1 := TRUE; END_IF;
END_REGION

REGION Network 5: SYRUP MFG VESSEL BOTTOM STERROR TRIP
   RUNG wire#powerrail
      Contact( "DI MAPING"."SYRUP MFG VESSEL BOTTOM STERROR TRIP" )
      wire#w1
      Coil( "SYRUP MFG VESSEL BOTTOM STERROR TRIP" )
   END_RUNG
   RUNG wire#w1
      P_Trig( "P_TRIG"."4" )
      S_Coil( "DO MAPING".HOOTER_1 )
   END_RUNG
   // the same network as SCL:
   "SYRUP MFG VESSEL BOTTOM STERROR TRIP" := "DI MAPING"."SYRUP MFG VESSEL BOTTOM STERROR TRIP";
   #_w1 := "DI MAPING"."SYRUP MFG VESSEL BOTTOM STERROR TRIP" AND NOT "P_TRIG"."4";   // rising edge
   "P_TRIG"."4" := "DI MAPING"."SYRUP MFG VESSEL BOTTOM STERROR TRIP";
   IF #_w1 THEN "DO MAPING".HOOTER_1 := TRUE; END_IF;
END_REGION

REGION Network 6: PREMIXING VESSEL BOTTOM STERROR TRIP
   RUNG wire#powerrail
      Contact( "DI MAPING"."PREMIXING VESSEL BOTTOM STERROR TRIP" )
      wire#w1
      Coil( "ALARM DB"."PREMIXING VESSEL BOTTOM STERROR TRIP" )
   END_RUNG
   RUNG wire#w1
      P_Trig( "P_TRIG"."5" )
      S_Coil( "DO MAPING".HOOTER_1 )
   END_RUNG
   // the same network as SCL:
   "ALARM DB"."PREMIXING VESSEL BOTTOM STERROR TRIP" := "DI MAPING"."PREMIXING VESSEL BOTTOM STERROR TRIP";
   #_w1 := "DI MAPING"."PREMIXING VESSEL BOTTOM STERROR TRIP" AND NOT "P_TRIG"."5";   // rising edge
   "P_TRIG"."5" := "DI MAPING"."PREMIXING VESSEL BOTTOM STERROR TRIP";
   IF #_w1 THEN "DO MAPING".HOOTER_1 := TRUE; END_IF;
END_REGION

REGION Network 7: INLINE 1 HOMOGENIZER MOTOR1 TRIP
   RUNG wire#powerrail
      Contact( "DI MAPING"."INLINE 1 HOMOGENIZER MOTOR1 TRIP" )
      wire#w1
      Coil( "ALARM DB"."INLINE 1 HOMOGENIZER MOTOR1 TRIP" )
   END_RUNG
   RUNG wire#w1
      P_Trig( "P_TRIG"."6" )
      S_Coil( "DO MAPING".HOOTER_1 )
   END_RUNG
   // the same network as SCL:
   "ALARM DB"."INLINE 1 HOMOGENIZER MOTOR1 TRIP" := "DI MAPING"."INLINE 1 HOMOGENIZER MOTOR1 TRIP";
   #_w1 := "DI MAPING"."INLINE 1 HOMOGENIZER MOTOR1 TRIP" AND NOT "P_TRIG"."6";   // rising edge
   "P_TRIG"."6" := "DI MAPING"."INLINE 1 HOMOGENIZER MOTOR1 TRIP";
   IF #_w1 THEN "DO MAPING".HOOTER_1 := TRUE; END_IF;
END_REGION

REGION Network 8: INLINE 2 HOMOGENIZER MOTOR 2 TRIP
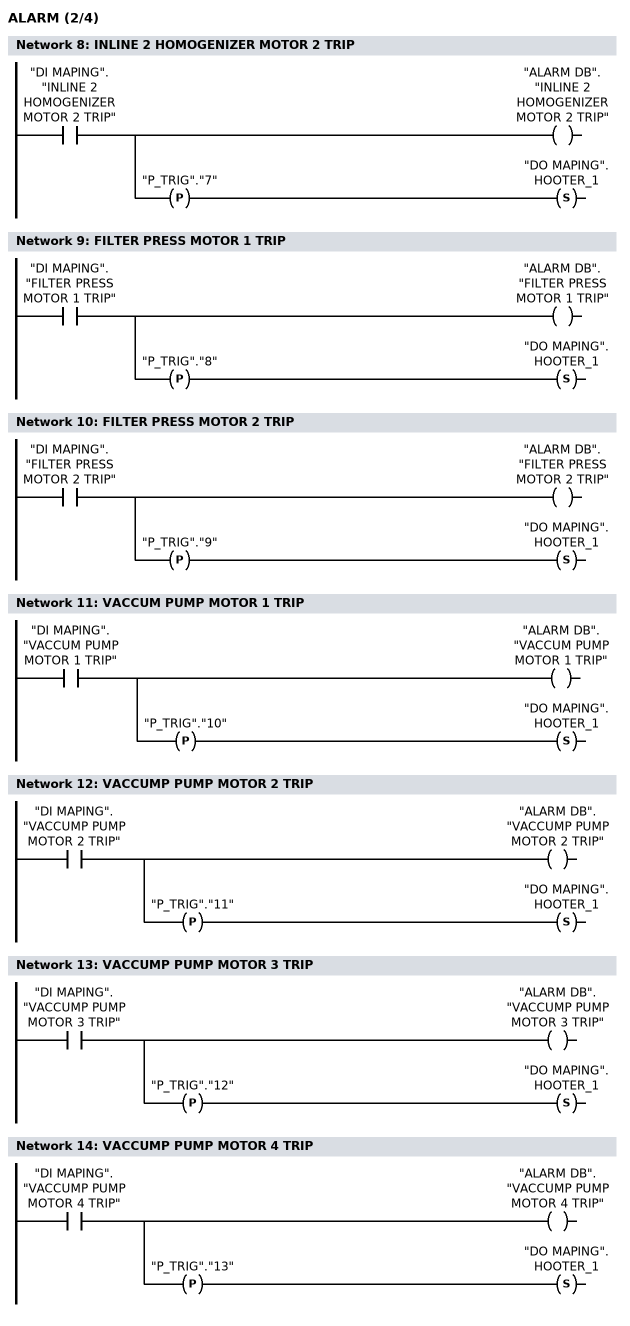
   RUNG wire#powerrail
      Contact( "DI MAPING"."INLINE 2 HOMOGENIZER MOTOR 2 TRIP" )
      wire#w1
      Coil( "ALARM DB"."INLINE 2 HOMOGENIZER MOTOR 2 TRIP" )
   END_RUNG
   RUNG wire#w1
      P_Trig( "P_TRIG"."7" )
      S_Coil( "DO MAPING".HOOTER_1 )
   END_RUNG
   // the same network as SCL:
   "ALARM DB"."INLINE 2 HOMOGENIZER MOTOR 2 TRIP" := "DI MAPING"."INLINE 2 HOMOGENIZER MOTOR 2 TRIP";
   #_w1 := "DI MAPING"."INLINE 2 HOMOGENIZER MOTOR 2 TRIP" AND NOT "P_TRIG"."7";   // rising edge
   "P_TRIG"."7" := "DI MAPING"."INLINE 2 HOMOGENIZER MOTOR 2 TRIP";
   IF #_w1 THEN "DO MAPING".HOOTER_1 := TRUE; END_IF;
END_REGION

REGION Network 9: FILTER PRESS MOTOR 1 TRIP
   RUNG wire#powerrail
      Contact( "DI MAPING"."FILTER PRESS MOTOR 1 TRIP" )
      wire#w1
      Coil( "ALARM DB"."FILTER PRESS MOTOR 1 TRIP" )
   END_RUNG
   RUNG wire#w1
      P_Trig( "P_TRIG"."8" )
      S_Coil( "DO MAPING".HOOTER_1 )
   END_RUNG
   // the same network as SCL:
   "ALARM DB"."FILTER PRESS MOTOR 1 TRIP" := "DI MAPING"."FILTER PRESS MOTOR 1 TRIP";
   #_w1 := "DI MAPING"."FILTER PRESS MOTOR 1 TRIP" AND NOT "P_TRIG"."8";   // rising edge
   "P_TRIG"."8" := "DI MAPING"."FILTER PRESS MOTOR 1 TRIP";
   IF #_w1 THEN "DO MAPING".HOOTER_1 := TRUE; END_IF;
END_REGION

REGION Network 10: FILTER PRESS MOTOR 2 TRIP
   RUNG wire#powerrail
      Contact( "DI MAPING"."FILTER PRESS MOTOR 2 TRIP" )
      wire#w1
      Coil( "ALARM DB"."FILTER PRESS MOTOR 2 TRIP" )
   END_RUNG
   RUNG wire#w1
      P_Trig( "P_TRIG"."9" )
      S_Coil( "DO MAPING".HOOTER_1 )
   END_RUNG
   // the same network as SCL:
   "ALARM DB"."FILTER PRESS MOTOR 2 TRIP" := "DI MAPING"."FILTER PRESS MOTOR 2 TRIP";
   #_w1 := "DI MAPING"."FILTER PRESS MOTOR 2 TRIP" AND NOT "P_TRIG"."9";   // rising edge
   "P_TRIG"."9" := "DI MAPING"."FILTER PRESS MOTOR 2 TRIP";
   IF #_w1 THEN "DO MAPING".HOOTER_1 := TRUE; END_IF;
END_REGION

REGION Network 11: VACCUM PUMP MOTOR 1 TRIP
   RUNG wire#powerrail
      Contact( "DI MAPING"."VACCUM PUMP MOTOR 1 TRIP" )
      wire#w1
      Coil( "ALARM DB"."VACCUM PUMP MOTOR 1 TRIP" )
   END_RUNG
   RUNG wire#w1
      P_Trig( "P_TRIG"."10" )
      S_Coil( "DO MAPING".HOOTER_1 )
   END_RUNG
   // the same network as SCL:
   "ALARM DB"."VACCUM PUMP MOTOR 1 TRIP" := "DI MAPING"."VACCUM PUMP MOTOR 1 TRIP";
   #_w1 := "DI MAPING"."VACCUM PUMP MOTOR 1 TRIP" AND NOT "P_TRIG"."10";   // rising edge
   "P_TRIG"."10" := "DI MAPING"."VACCUM PUMP MOTOR 1 TRIP";
   IF #_w1 THEN "DO MAPING".HOOTER_1 := TRUE; END_IF;
END_REGION

REGION Network 12: VACCUMP PUMP MOTOR 2 TRIP
   RUNG wire#powerrail
      Contact( "DI MAPING"."VACCUMP PUMP MOTOR 2 TRIP" )
      wire#w1
      Coil( "ALARM DB"."VACCUMP PUMP MOTOR 2 TRIP" )
   END_RUNG
   RUNG wire#w1
      P_Trig( "P_TRIG"."11" )
      S_Coil( "DO MAPING".HOOTER_1 )
   END_RUNG
   // the same network as SCL:
   "ALARM DB"."VACCUMP PUMP MOTOR 2 TRIP" := "DI MAPING"."VACCUMP PUMP MOTOR 2 TRIP";
   #_w1 := "DI MAPING"."VACCUMP PUMP MOTOR 2 TRIP" AND NOT "P_TRIG"."11";   // rising edge
   "P_TRIG"."11" := "DI MAPING"."VACCUMP PUMP MOTOR 2 TRIP";
   IF #_w1 THEN "DO MAPING".HOOTER_1 := TRUE; END_IF;
END_REGION

REGION Network 13: VACCUMP PUMP MOTOR 3 TRIP
   RUNG wire#powerrail
      Contact( "DI MAPING"."VACCUMP PUMP MOTOR 3 TRIP" )
      wire#w1
      Coil( "ALARM DB"."VACCUMP PUMP MOTOR 3 TRIP" )
   END_RUNG
   RUNG wire#w1
      P_Trig( "P_TRIG"."12" )
      S_Coil( "DO MAPING".HOOTER_1 )
   END_RUNG
   // the same network as SCL:
   "ALARM DB"."VACCUMP PUMP MOTOR 3 TRIP" := "DI MAPING"."VACCUMP PUMP MOTOR 3 TRIP";
   #_w1 := "DI MAPING"."VACCUMP PUMP MOTOR 3 TRIP" AND NOT "P_TRIG"."12";   // rising edge
   "P_TRIG"."12" := "DI MAPING"."VACCUMP PUMP MOTOR 3 TRIP";
   IF #_w1 THEN "DO MAPING".HOOTER_1 := TRUE; END_IF;
END_REGION

REGION Network 14: VACCUMP PUMP MOTOR 4 TRIP
   RUNG wire#powerrail
      Contact( "DI MAPING"."VACCUMP PUMP MOTOR 4 TRIP" )
      wire#w1
      Coil( "ALARM DB"."VACCUMP PUMP MOTOR 4 TRIP" )
   END_RUNG
   RUNG wire#w1
      P_Trig( "P_TRIG"."13" )
      S_Coil( "DO MAPING".HOOTER_1 )
   END_RUNG
   // the same network as SCL:
   "ALARM DB"."VACCUMP PUMP MOTOR 4 TRIP" := "DI MAPING"."VACCUMP PUMP MOTOR 4 TRIP";
   #_w1 := "DI MAPING"."VACCUMP PUMP MOTOR 4 TRIP" AND NOT "P_TRIG"."13";   // rising edge
   "P_TRIG"."13" := "DI MAPING"."VACCUMP PUMP MOTOR 4 TRIP";
   IF #_w1 THEN "DO MAPING".HOOTER_1 := TRUE; END_IF;
END_REGION

REGION Network 15: SUGAR VESSEL BOTTOM STERROR TRIP
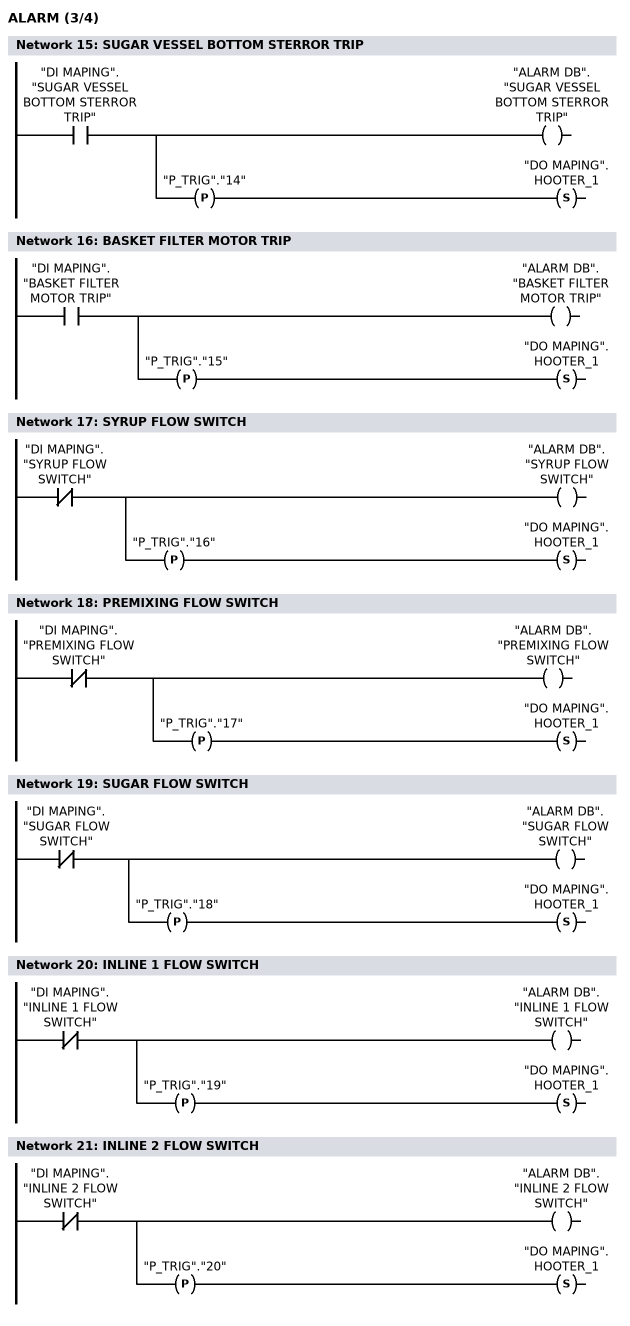
   RUNG wire#powerrail
      Contact( "DI MAPING"."SUGAR VESSEL BOTTOM STERROR TRIP" )
      wire#w1
      Coil( "ALARM DB"."SUGAR VESSEL BOTTOM STERROR TRIP" )
   END_RUNG
   RUNG wire#w1
      P_Trig( "P_TRIG"."14" )
      S_Coil( "DO MAPING".HOOTER_1 )
   END_RUNG
   // the same network as SCL:
   "ALARM DB"."SUGAR VESSEL BOTTOM STERROR TRIP" := "DI MAPING"."SUGAR VESSEL BOTTOM STERROR TRIP";
   #_w1 := "DI MAPING"."SUGAR VESSEL BOTTOM STERROR TRIP" AND NOT "P_TRIG"."14";   // rising edge
   "P_TRIG"."14" := "DI MAPING"."SUGAR VESSEL BOTTOM STERROR TRIP";
   IF #_w1 THEN "DO MAPING".HOOTER_1 := TRUE; END_IF;
END_REGION

REGION Network 16: BASKET FILTER MOTOR TRIP
   RUNG wire#powerrail
      Contact( "DI MAPING"."BASKET FILTER MOTOR TRIP" )
      wire#w1
      Coil( "ALARM DB"."BASKET FILTER MOTOR TRIP" )
   END_RUNG
   RUNG wire#w1
      P_Trig( "P_TRIG"."15" )
      S_Coil( "DO MAPING".HOOTER_1 )
   END_RUNG
   // the same network as SCL:
   "ALARM DB"."BASKET FILTER MOTOR TRIP" := "DI MAPING"."BASKET FILTER MOTOR TRIP";
   #_w1 := "DI MAPING"."BASKET FILTER MOTOR TRIP" AND NOT "P_TRIG"."15";   // rising edge
   "P_TRIG"."15" := "DI MAPING"."BASKET FILTER MOTOR TRIP";
   IF #_w1 THEN "DO MAPING".HOOTER_1 := TRUE; END_IF;
END_REGION

REGION Network 17: SYRUP FLOW SWITCH
   RUNG wire#powerrail
      I_Contact( "DI MAPING"."SYRUP FLOW SWITCH" )
      wire#w1
      Coil( "ALARM DB"."SYRUP FLOW SWITCH" )
   END_RUNG
   RUNG wire#w1
      P_Trig( "P_TRIG"."16" )
      S_Coil( "DO MAPING".HOOTER_1 )
   END_RUNG
   // the same network as SCL:
   "ALARM DB"."SYRUP FLOW SWITCH" := NOT "DI MAPING"."SYRUP FLOW SWITCH";
   #_w1 := NOT "DI MAPING"."SYRUP FLOW SWITCH" AND NOT "P_TRIG"."16";   // rising edge
   "P_TRIG"."16" := NOT "DI MAPING"."SYRUP FLOW SWITCH";
   IF #_w1 THEN "DO MAPING".HOOTER_1 := TRUE; END_IF;
END_REGION

REGION Network 18: PREMIXING FLOW SWITCH
   RUNG wire#powerrail
      I_Contact( "DI MAPING"."PREMIXING FLOW SWITCH" )
      wire#w1
      Coil( "ALARM DB"."PREMIXING FLOW SWITCH" )
   END_RUNG
   RUNG wire#w1
      P_Trig( "P_TRIG"."17" )
      S_Coil( "DO MAPING".HOOTER_1 )
   END_RUNG
   // the same network as SCL:
   "ALARM DB"."PREMIXING FLOW SWITCH" := NOT "DI MAPING"."PREMIXING FLOW SWITCH";
   #_w1 := NOT "DI MAPING"."PREMIXING FLOW SWITCH" AND NOT "P_TRIG"."17";   // rising edge
   "P_TRIG"."17" := NOT "DI MAPING"."PREMIXING FLOW SWITCH";
   IF #_w1 THEN "DO MAPING".HOOTER_1 := TRUE; END_IF;
END_REGION

REGION Network 19: SUGAR FLOW SWITCH
   RUNG wire#powerrail
      I_Contact( "DI MAPING"."SUGAR FLOW SWITCH" )
      wire#w1
      Coil( "ALARM DB"."SUGAR FLOW SWITCH" )
   END_RUNG
   RUNG wire#w1
      P_Trig( "P_TRIG"."18" )
      S_Coil( "DO MAPING".HOOTER_1 )
   END_RUNG
   // the same network as SCL:
   "ALARM DB"."SUGAR FLOW SWITCH" := NOT "DI MAPING"."SUGAR FLOW SWITCH";
   #_w1 := NOT "DI MAPING"."SUGAR FLOW SWITCH" AND NOT "P_TRIG"."18";   // rising edge
   "P_TRIG"."18" := NOT "DI MAPING"."SUGAR FLOW SWITCH";
   IF #_w1 THEN "DO MAPING".HOOTER_1 := TRUE; END_IF;
END_REGION

REGION Network 20: INLINE 1 FLOW SWITCH
   RUNG wire#powerrail
      I_Contact( "DI MAPING"."INLINE 1 FLOW SWITCH" )
      wire#w1
      Coil( "ALARM DB"."INLINE 1 FLOW SWITCH" )
   END_RUNG
   RUNG wire#w1
      P_Trig( "P_TRIG"."19" )
      S_Coil( "DO MAPING".HOOTER_1 )
   END_RUNG
   // the same network as SCL:
   "ALARM DB"."INLINE 1 FLOW SWITCH" := NOT "DI MAPING"."INLINE 1 FLOW SWITCH";
   #_w1 := NOT "DI MAPING"."INLINE 1 FLOW SWITCH" AND NOT "P_TRIG"."19";   // rising edge
   "P_TRIG"."19" := NOT "DI MAPING"."INLINE 1 FLOW SWITCH";
   IF #_w1 THEN "DO MAPING".HOOTER_1 := TRUE; END_IF;
END_REGION

REGION Network 21: INLINE 2 FLOW SWITCH
   RUNG wire#powerrail
      I_Contact( "DI MAPING"."INLINE 2 FLOW SWITCH" )
      wire#w1
      Coil( "ALARM DB"."INLINE 2 FLOW SWITCH" )
   END_RUNG
   RUNG wire#w1
      P_Trig( "P_TRIG"."20" )
      S_Coil( "DO MAPING".HOOTER_1 )
   END_RUNG
   // the same network as SCL:
   "ALARM DB"."INLINE 2 FLOW SWITCH" := NOT "DI MAPING"."INLINE 2 FLOW SWITCH";
   #_w1 := NOT "DI MAPING"."INLINE 2 FLOW SWITCH" AND NOT "P_TRIG"."20";   // rising edge
   "P_TRIG"."20" := NOT "DI MAPING"."INLINE 2 FLOW SWITCH";
   IF #_w1 THEN "DO MAPING".HOOTER_1 := TRUE; END_IF;
END_REGION

REGION Network 22: MFG TO STORAGE-1 WITH INLINE HOMOGENIZER TRANSFER COMPLETE
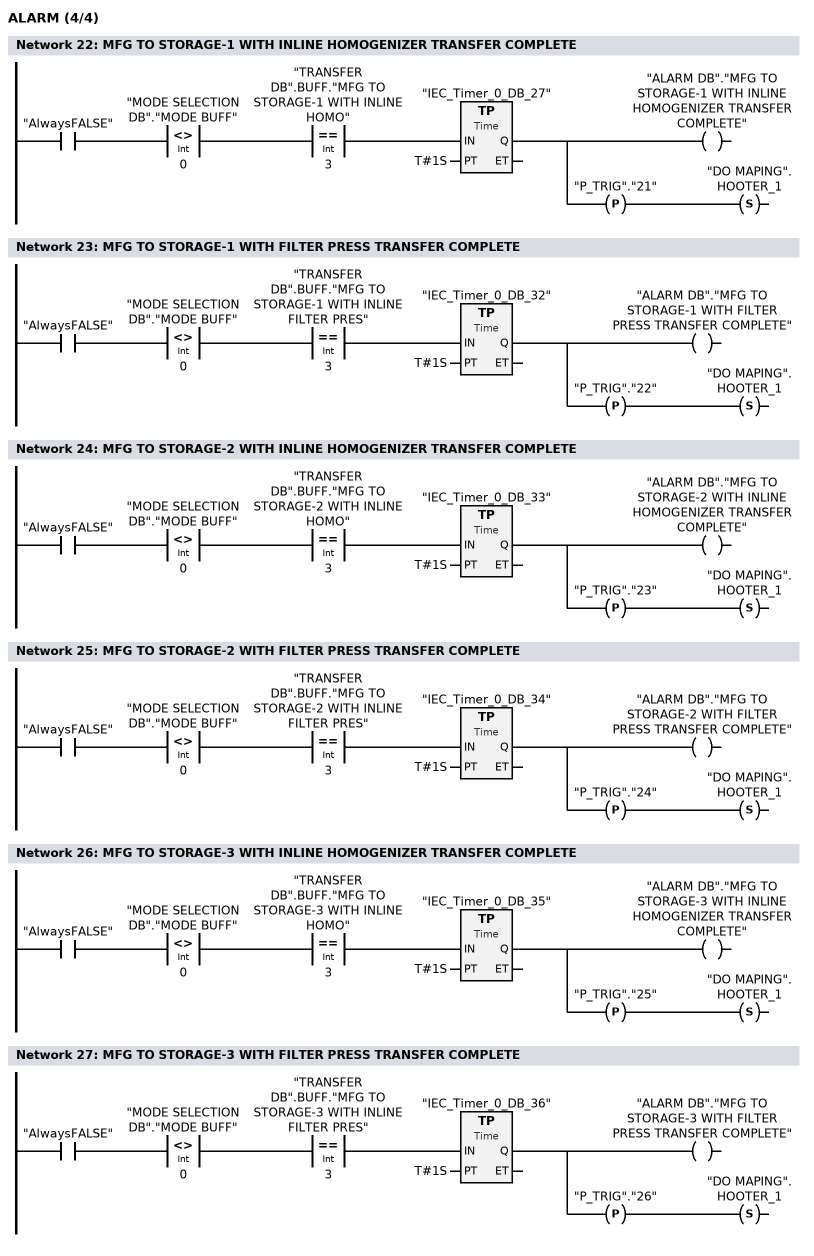
   RUNG wire#powerrail
      Contact( "AlwaysFALSE" )
      { S7_Templates := "SrcType := Int" } NE_Contact(in1 := "MODE SELECTION DB"."MODE BUFF", in2 := 0)
      { S7_Templates := "SrcType := Int" } EQ_Contact(in1 := "TRANSFER DB".BUFF."MFG TO STORAGE-1 WITH INLINE HOMO", in2 := 3)
      { S7_Templates := "time_type := Time" } "IEC_Timer_0_DB_27".TP(pt := T#1S, et =>)
      wire#w1
      Coil( "ALARM DB"."MFG TO STORAGE-1 WITH INLINE HOMOGENIZER TRANSFER COMPLETE" )
   END_RUNG
   RUNG wire#w1
      P_Trig( "P_TRIG"."21" )
      S_Coil( "DO MAPING".HOOTER_1 )
   END_RUNG
   // the same network as SCL:
   "IEC_Timer_0_DB_27".TP(IN := "AlwaysFALSE" AND ("MODE SELECTION DB"."MODE BUFF" <> 0) AND ("TRANSFER DB".BUFF."MFG TO STORAGE-1 WITH INLINE HOMO" = 3),
                          PT := T#1S);
   "ALARM DB"."MFG TO STORAGE-1 WITH INLINE HOMOGENIZER TRANSFER COMPLETE" := "IEC_Timer_0_DB_27".Q;
   #_w1 := "IEC_Timer_0_DB_27".Q AND NOT "P_TRIG"."21";   // rising edge
   "P_TRIG"."21" := "IEC_Timer_0_DB_27".Q;
   IF #_w1 THEN "DO MAPING".HOOTER_1 := TRUE; END_IF;
END_REGION

REGION Network 23: MFG TO STORAGE-1 WITH FILTER PRESS TRANSFER COMPLETE
   RUNG wire#powerrail
      Contact( "AlwaysFALSE" )
      { S7_Templates := "SrcType := Int" } NE_Contact(in1 := "MODE SELECTION DB"."MODE BUFF", in2 := 0)
      { S7_Templates := "SrcType := Int" } EQ_Contact(in1 := "TRANSFER DB".BUFF."MFG TO STORAGE-1 WITH INLINE FILTER PRES", in2 := 3)
      { S7_Templates := "time_type := Time" } "IEC_Timer_0_DB_32".TP(pt := T#1S, et =>)
      wire#w1
      Coil( "ALARM DB"."MFG TO STORAGE-1 WITH FILTER PRESS TRANSFER COMPLETE" )
   END_RUNG
   RUNG wire#w1
      P_Trig( "P_TRIG"."22" )
      S_Coil( "DO MAPING".HOOTER_1 )
   END_RUNG
   // the same network as SCL:
   "IEC_Timer_0_DB_32".TP(IN := "AlwaysFALSE" AND ("MODE SELECTION DB"."MODE BUFF" <> 0) AND ("TRANSFER DB".BUFF."MFG TO STORAGE-1 WITH INLINE FILTER PRES" = 3),
                          PT := T#1S);
   "ALARM DB"."MFG TO STORAGE-1 WITH FILTER PRESS TRANSFER COMPLETE" := "IEC_Timer_0_DB_32".Q;
   #_w1 := "IEC_Timer_0_DB_32".Q AND NOT "P_TRIG"."22";   // rising edge
   "P_TRIG"."22" := "IEC_Timer_0_DB_32".Q;
   IF #_w1 THEN "DO MAPING".HOOTER_1 := TRUE; END_IF;
END_REGION

REGION Network 24: MFG TO STORAGE-2 WITH INLINE HOMOGENIZER TRANSFER COMPLETE
   RUNG wire#powerrail
      Contact( "AlwaysFALSE" )
      { S7_Templates := "SrcType := Int" } NE_Contact(in1 := "MODE SELECTION DB"."MODE BUFF", in2 := 0)
      { S7_Templates := "SrcType := Int" } EQ_Contact(in1 := "TRANSFER DB".BUFF."MFG TO STORAGE-2 WITH INLINE HOMO", in2 := 3)
      { S7_Templates := "time_type := Time" } "IEC_Timer_0_DB_33".TP(pt := T#1S, et =>)
      wire#w1
      Coil( "ALARM DB"."MFG TO STORAGE-2 WITH INLINE HOMOGENIZER TRANSFER COMPLETE" )
   END_RUNG
   RUNG wire#w1
      P_Trig( "P_TRIG"."23" )
      S_Coil( "DO MAPING".HOOTER_1 )
   END_RUNG
   // the same network as SCL:
   "IEC_Timer_0_DB_33".TP(IN := "AlwaysFALSE" AND ("MODE SELECTION DB"."MODE BUFF" <> 0) AND ("TRANSFER DB".BUFF."MFG TO STORAGE-2 WITH INLINE HOMO" = 3),
                          PT := T#1S);
   "ALARM DB"."MFG TO STORAGE-2 WITH INLINE HOMOGENIZER TRANSFER COMPLETE" := "IEC_Timer_0_DB_33".Q;
   #_w1 := "IEC_Timer_0_DB_33".Q AND NOT "P_TRIG"."23";   // rising edge
   "P_TRIG"."23" := "IEC_Timer_0_DB_33".Q;
   IF #_w1 THEN "DO MAPING".HOOTER_1 := TRUE; END_IF;
END_REGION

REGION Network 25: MFG TO STORAGE-2 WITH FILTER PRESS TRANSFER COMPLETE
   RUNG wire#powerrail
      Contact( "AlwaysFALSE" )
      { S7_Templates := "SrcType := Int" } NE_Contact(in1 := "MODE SELECTION DB"."MODE BUFF", in2 := 0)
      { S7_Templates := "SrcType := Int" } EQ_Contact(in1 := "TRANSFER DB".BUFF."MFG TO STORAGE-2 WITH INLINE FILTER PRES", in2 := 3)
      { S7_Templates := "time_type := Time" } "IEC_Timer_0_DB_34".TP(pt := T#1S, et =>)
      wire#w1
      Coil( "ALARM DB"."MFG TO STORAGE-2 WITH FILTER PRESS TRANSFER COMPLETE" )
   END_RUNG
   RUNG wire#w1
      P_Trig( "P_TRIG"."24" )
      S_Coil( "DO MAPING".HOOTER_1 )
   END_RUNG
   // the same network as SCL:
   "IEC_Timer_0_DB_34".TP(IN := "AlwaysFALSE" AND ("MODE SELECTION DB"."MODE BUFF" <> 0) AND ("TRANSFER DB".BUFF."MFG TO STORAGE-2 WITH INLINE FILTER PRES" = 3),
                          PT := T#1S);
   "ALARM DB"."MFG TO STORAGE-2 WITH FILTER PRESS TRANSFER COMPLETE" := "IEC_Timer_0_DB_34".Q;
   #_w1 := "IEC_Timer_0_DB_34".Q AND NOT "P_TRIG"."24";   // rising edge
   "P_TRIG"."24" := "IEC_Timer_0_DB_34".Q;
   IF #_w1 THEN "DO MAPING".HOOTER_1 := TRUE; END_IF;
END_REGION

REGION Network 26: MFG TO STORAGE-3 WITH INLINE HOMOGENIZER TRANSFER COMPLETE
   RUNG wire#powerrail
      Contact( "AlwaysFALSE" )
      { S7_Templates := "SrcType := Int" } NE_Contact(in1 := "MODE SELECTION DB"."MODE BUFF", in2 := 0)
      { S7_Templates := "SrcType := Int" } EQ_Contact(in1 := "TRANSFER DB".BUFF."MFG TO STORAGE-3 WITH INLINE HOMO", in2 := 3)
      { S7_Templates := "time_type := Time" } "IEC_Timer_0_DB_35".TP(pt := T#1S, et =>)
      wire#w1
      Coil( "ALARM DB"."MFG TO STORAGE-3 WITH INLINE HOMOGENIZER TRANSFER COMPLETE" )
   END_RUNG
   RUNG wire#w1
      P_Trig( "P_TRIG"."25" )
      S_Coil( "DO MAPING".HOOTER_1 )
   END_RUNG
   // the same network as SCL:
   "IEC_Timer_0_DB_35".TP(IN := "AlwaysFALSE" AND ("MODE SELECTION DB"."MODE BUFF" <> 0) AND ("TRANSFER DB".BUFF."MFG TO STORAGE-3 WITH INLINE HOMO" = 3),
                          PT := T#1S);
   "ALARM DB"."MFG TO STORAGE-3 WITH INLINE HOMOGENIZER TRANSFER COMPLETE" := "IEC_Timer_0_DB_35".Q;
   #_w1 := "IEC_Timer_0_DB_35".Q AND NOT "P_TRIG"."25";   // rising edge
   "P_TRIG"."25" := "IEC_Timer_0_DB_35".Q;
   IF #_w1 THEN "DO MAPING".HOOTER_1 := TRUE; END_IF;
END_REGION

REGION Network 27: MFG TO STORAGE-3 WITH FILTER PRESS TRANSFER COMPLETE
   RUNG wire#powerrail
      Contact( "AlwaysFALSE" )
      { S7_Templates := "SrcType := Int" } NE_Contact(in1 := "MODE SELECTION DB"."MODE BUFF", in2 := 0)
      { S7_Templates := "SrcType := Int" } EQ_Contact(in1 := "TRANSFER DB".BUFF."MFG TO STORAGE-3 WITH INLINE FILTER PRES", in2 := 3)
      { S7_Templates := "time_type := Time" } "IEC_Timer_0_DB_36".TP(pt := T#1S, et =>)
      wire#w1
      Coil( "ALARM DB"."MFG TO STORAGE-3 WITH FILTER PRESS TRANSFER COMPLETE" )
   END_RUNG
   RUNG wire#w1
      P_Trig( "P_TRIG"."26" )
      S_Coil( "DO MAPING".HOOTER_1 )
   END_RUNG
   // the same network as SCL:
   "IEC_Timer_0_DB_36".TP(IN := "AlwaysFALSE" AND ("MODE SELECTION DB"."MODE BUFF" <> 0) AND ("TRANSFER DB".BUFF."MFG TO STORAGE-3 WITH INLINE FILTER PRES" = 3),
                          PT := T#1S);
   "ALARM DB"."MFG TO STORAGE-3 WITH FILTER PRESS TRANSFER COMPLETE" := "IEC_Timer_0_DB_36".Q;
   #_w1 := "IEC_Timer_0_DB_36".Q AND NOT "P_TRIG"."26";   // rising edge
   "P_TRIG"."26" := "IEC_Timer_0_DB_36".Q;
   IF #_w1 THEN "DO MAPING".HOOTER_1 := TRUE; END_IF;
END_REGION
END_FUNCTION

FUNCTION "AUTO ALARM" : Void   // FC17, LAD
{ S7_Optimized_Access := 'TRUE' }
// stored: SetENOAutomatically false
BEGIN

REGION Network 1: ///////////////////////////////MFG PUPUP/////////////////////////////////////
END_REGION

REGION Network 2: PURIFIED WATER PROCESS SELECT
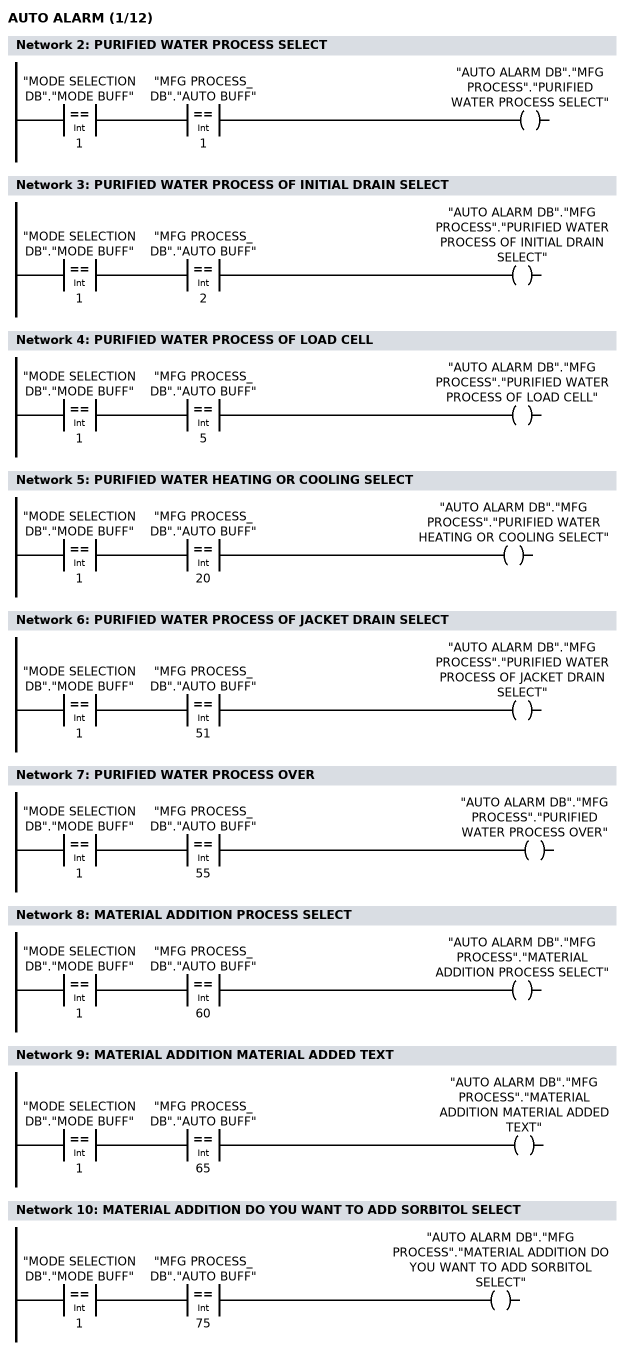
   RUNG wire#powerrail
      { S7_Templates := "SrcType := Int" } EQ_Contact(in1 := "MODE SELECTION DB"."MODE BUFF", in2 := 1)
      { S7_Templates := "SrcType := Int" } EQ_Contact(in1 := "MFG PROCESS_DB"."AUTO BUFF", in2 := 1)
      Coil( "AUTO ALARM DB"."MFG PROCESS"."PURIFIED WATER PROCESS SELECT" )
   END_RUNG
   // the same network as SCL:
   "AUTO ALARM DB"."MFG PROCESS"."PURIFIED WATER PROCESS SELECT" := ("MODE SELECTION DB"."MODE BUFF" = 1) AND ("MFG PROCESS_DB"."AUTO BUFF" = 1);
END_REGION

REGION Network 3: PURIFIED WATER PROCESS OF INITIAL DRAIN SELECT
   RUNG wire#powerrail
      { S7_Templates := "SrcType := Int" } EQ_Contact(in1 := "MODE SELECTION DB"."MODE BUFF", in2 := 1)
      { S7_Templates := "SrcType := Int" } EQ_Contact(in1 := "MFG PROCESS_DB"."AUTO BUFF", in2 := 2)
      Coil( "AUTO ALARM DB"."MFG PROCESS"."PURIFIED WATER PROCESS OF INITIAL DRAIN SELECT" )
   END_RUNG
   // the same network as SCL:
   "AUTO ALARM DB"."MFG PROCESS"."PURIFIED WATER PROCESS OF INITIAL DRAIN SELECT" := ("MODE SELECTION DB"."MODE BUFF" = 1) AND ("MFG PROCESS_DB"."AUTO BUFF" = 2);
END_REGION

REGION Network 4: PURIFIED WATER PROCESS OF LOAD CELL
   RUNG wire#powerrail
      { S7_Templates := "SrcType := Int" } EQ_Contact(in1 := "MODE SELECTION DB"."MODE BUFF", in2 := 1)
      { S7_Templates := "SrcType := Int" } EQ_Contact(in1 := "MFG PROCESS_DB"."AUTO BUFF", in2 := 5)
      Coil( "AUTO ALARM DB"."MFG PROCESS"."PURIFIED WATER PROCESS OF LOAD CELL" )
   END_RUNG
   // the same network as SCL:
   "AUTO ALARM DB"."MFG PROCESS"."PURIFIED WATER PROCESS OF LOAD CELL" := ("MODE SELECTION DB"."MODE BUFF" = 1) AND ("MFG PROCESS_DB"."AUTO BUFF" = 5);
END_REGION

REGION Network 5: PURIFIED WATER HEATING OR COOLING SELECT
   RUNG wire#powerrail
      { S7_Templates := "SrcType := Int" } EQ_Contact(in1 := "MODE SELECTION DB"."MODE BUFF", in2 := 1)
      { S7_Templates := "SrcType := Int" } EQ_Contact(in1 := "MFG PROCESS_DB"."AUTO BUFF", in2 := 20)
      Coil( "AUTO ALARM DB"."MFG PROCESS"."PURIFIED WATER HEATING OR COOLING SELECT" )
   END_RUNG
   // the same network as SCL:
   "AUTO ALARM DB"."MFG PROCESS"."PURIFIED WATER HEATING OR COOLING SELECT" := ("MODE SELECTION DB"."MODE BUFF" = 1) AND ("MFG PROCESS_DB"."AUTO BUFF" = 20);
END_REGION

REGION Network 6: PURIFIED WATER PROCESS OF JACKET DRAIN SELECT
   RUNG wire#powerrail
      { S7_Templates := "SrcType := Int" } EQ_Contact(in1 := "MODE SELECTION DB"."MODE BUFF", in2 := 1)
      { S7_Templates := "SrcType := Int" } EQ_Contact(in1 := "MFG PROCESS_DB"."AUTO BUFF", in2 := 51)
      Coil( "AUTO ALARM DB"."MFG PROCESS"."PURIFIED WATER PROCESS OF JACKET DRAIN SELECT" )
   END_RUNG
   // the same network as SCL:
   "AUTO ALARM DB"."MFG PROCESS"."PURIFIED WATER PROCESS OF JACKET DRAIN SELECT" := ("MODE SELECTION DB"."MODE BUFF" = 1) AND ("MFG PROCESS_DB"."AUTO BUFF" = 51);
END_REGION

REGION Network 7: PURIFIED WATER PROCESS OVER
   RUNG wire#powerrail
      { S7_Templates := "SrcType := Int" } EQ_Contact(in1 := "MODE SELECTION DB"."MODE BUFF", in2 := 1)
      { S7_Templates := "SrcType := Int" } EQ_Contact(in1 := "MFG PROCESS_DB"."AUTO BUFF", in2 := 55)
      Coil( "AUTO ALARM DB"."MFG PROCESS"."PURIFIED WATER PROCESS OVER" )
   END_RUNG
   // the same network as SCL:
   "AUTO ALARM DB"."MFG PROCESS"."PURIFIED WATER PROCESS OVER" := ("MODE SELECTION DB"."MODE BUFF" = 1) AND ("MFG PROCESS_DB"."AUTO BUFF" = 55);
END_REGION

